// TIA Portal project "ContadoresHMI4" (V16)

(* hardware
DEVICE "S71500/ET200MP station_1"  S7-1500 station
   slot 0: "Rail_0"  Rack  6ES7 590-1***0-0AA0
   slot 1: "PLC_1"  CPU 1516-3 PN/DP  6ES7 516-3AN00-0AB0  V1.8
      slot 3: "CPU display_1"  6ES7591-1BA00-0AA0
      slot 32768: "PROFINET interface_1"  X1
         slot 32769: "Port_1"  X1 P1
         slot 32770: "Port_2"  X1 P2
      slot 33024: "PROFINET interface_2"  X2
         slot 33025: "Port_1"  X2 P1
      slot 33280: "DP interface_1"  X3
DEVICE "HMI_1"  TP700 Comfort
   slot 0: "HMI_1"  TP700 Comfort  6AV2 124-0GC01-0AX0  16.0.0.0
   slot 1: "HMI_RT_1"  TP700 Comfort  6AV2 124-0GC01-0AX0  16.0.0.0
   slot 5: "HMI_1.IE_CP_1"  PROFINET Interface  16.0.0.0
      slot 1: "PROFINET Interface_1"  PROFINET Interface
         slot 1: "Port_1"  Port
         slot 2: "Port_2"  Port
   slot 7: "HMI_1.MPI/DP_CP_1"  MPI/DP Interface  16.0.0.0
*)

// ===== PLC "PLC_1"  CPU 1516-3 PN/DP =====

VAR_GLOBAL   // PLC tag table "Default tag table"
   "ReiniciarJuego" AT %M6.0 : Bool;
   "CodigoS0J1" AT %M6.1 : Bool;
   "CodigoS1J1" AT %M6.2 : Bool;
   "CodigoS2J1" AT %M6.3 : Bool;
   "CodigoS3J1" AT %M6.4 : Bool;
   "CodigoO0J1" AT %M6.5 : Bool;
   "CodigoO1J1" AT %M6.6 : Bool;
   "CodigoO2J1" AT %M6.7 : Bool;
   "CodigoO3J1" AT %M7.0 : Bool;
   "CodigoS0J2" AT %M7.1 : Bool;
   "CodigoS1J2" AT %M7.2 : Bool;
   "CodigoS2J2" AT %M7.3 : Bool;
   "CodigoS3J2" AT %M7.4 : Bool;
   "CodigoO0J2" AT %M7.5 : Bool;
   "CodigoO1J2" AT %M7.6 : Bool;
   "CodigoO2J2" AT %M7.7 : Bool;
   "CodigoO3J2" AT %M8.0 : Bool;
   "Intento0J1" AT %M8.1 : Bool;
   "Intento1J1" AT %M8.2 : Bool;
   "Intento2J1" AT %M8.3 : Bool;
   "Intento3J1" AT %M8.4 : Bool;
   "Intento0J2" AT %M8.5 : Bool;
   "Intento1J2" AT %M8.6 : Bool;
   "Intento2J2" AT %M8.7 : Bool;
   "Intento3J2" AT %M9.0 : Bool;
   "IntentoCompletoJ1" AT %MW2 : UInt;
   "IntentoCompletoJ2" AT %MW4 : UInt;
   "Timer" AT %M9.3 : Bool;
   "Repetido" AT %M9.4 : Bool;
   "Panel1CafeJ1" AT %M9.5 : Bool;
   "Panel1RosaJ1" AT %M9.6 : Bool;
   "Panel1MoradoJ1" AT %M9.7 : Bool;
   "Panel1RojoJ1" AT %M10.0 : Bool;
   "Panel1AzulJ1" AT %M10.1 : Bool;
   "Panel1VerdeJ1" AT %M10.2 : Bool;
   "Panel1AmarilloJ1" AT %M10.3 : Bool;
   "Panel2CafeJ1" AT %M10.4 : Bool;
   "Panel2RosaJ1" AT %M10.5 : Bool;
   "Panel2MoradoJ1" AT %M10.6 : Bool;
   "Panel2RojoJ1" AT %M10.7 : Bool;
   "Panel2AzulJ1" AT %M11.0 : Bool;
   "Panel2VerdeJ1" AT %M11.1 : Bool;
   "Panel2AmarilloJ1" AT %M11.2 : Bool;
   "Panel1CafeJ2" AT %M11.3 : Bool;
   "Panel1RosaJ2" AT %M11.4 : Bool;
   "Panel1MoradoJ2" AT %M11.5 : Bool;
   "Panel1RojoJ2" AT %M11.6 : Bool;
   "Panel1AzulJ2" AT %M11.7 : Bool;
   "Panel1VerdeJ2" AT %M12.0 : Bool;
   "Panel1AmarilloJ2" AT %M12.1 : Bool;
   "Panel2CafeJ2" AT %M12.2 : Bool;
   "Panel2RosaJ2" AT %M12.3 : Bool;
   "Panel2MoradoJ2" AT %M12.4 : Bool;
   "Panel2RojoJ2" AT %M12.5 : Bool;
   "Panel2AzulJ2" AT %M12.6 : Bool;
   "Panel2VerdeJ2" AT %M12.7 : Bool;
   "Panel2AmarilloJ2" AT %M13.0 : Bool;
   "Panel1J1Activado" AT %M13.1 : Bool;
   "Panel2J1Activado" AT %M13.2 : Bool;
   "Panel1J2Activado" AT %M13.3 : Bool;
   "Panel2J2Activado" AT %M13.4 : Bool;
   "ReinicioCorrecto" AT %M13.5 : Bool;
   "Bounce1" AT %M13.6 : Bool;
   "Bounce2" AT %M13.7 : Bool;
   "Bounce3" AT %M14.0 : Bool;
   "Bounce5" AT %M14.1 : Bool;
   "Bounce6" AT %M14.2 : Bool;
   "Bounce7" AT %M14.3 : Bool;
   "Bounce8" AT %M14.4 : Bool;
   "Bounce10" AT %M14.5 : Bool;
   "MensajeCorrecto" AT %M14.6 : Bool;
   "Bounce4" AT %M14.7 : Bool;
   "Bounce9" AT %M15.0 : Bool;
   "ReiniciarContadorJ1" AT %M15.1 : Bool;
   "ReiniciarContadorJ2" AT %M15.2 : Bool;
   "ChecarIntento1J1" AT %M15.3 : Bool;
   "ChecarIntento2J1" AT %M15.4 : Bool;
   "ChecarIntento3J1" AT %M15.5 : Bool;
   "ChecarIntento4J1" AT %M15.6 : Bool;
   "ChecarIntento1J2" AT %M15.7 : Bool;
   "ChecarIntento2J2" AT %M16.0 : Bool;
   "ChecarIntento3J2" AT %M16.1 : Bool;
   "ChecarIntento4J2" AT %M16.2 : Bool;
   "ContadorCorr" AT %MW17 : UInt;
   "ContadorSimi" AT %MW20 : UInt;
   "ContadorError" AT %MW22 : UInt;
   "ContadorCorrTemp" AT %MW24 : UInt;
   "ContadorSimiTemp" AT %MW26 : UInt;
   "ReiniciarChecarCorr" AT %M28.0 : Bool;
   "ReiniciarChecarSimi" AT %M28.1 : Bool;
   "ReiniciarChecarError" AT %M28.2 : Bool;
   "ChecarIntentoCorrecto" AT %M28.3 : Bool;
   "ChecarIntento1SJ1" AT %M28.4 : Bool;
   "ChecarIntento2SJ1" AT %M28.5 : Bool;
   "ChecarIntento3SJ1" AT %M28.6 : Bool;
   "ChecarIntento4SJ1" AT %M28.7 : Bool;
   "ChecarIntento1SJ2" AT %M29.0 : Bool;
   "ChecarIntento2SJ2" AT %M29.1 : Bool;
   "ChecarIntento3SJ2" AT %M29.2 : Bool;
   "ChecarIntento4SJ2" AT %M29.3 : Bool;
   "CorrectasSimilares" AT %M29.4 : Bool;
   "IntentoCompletoCORR" AT %MW31 : UInt;
   "ReiniciarCorrSimiDisp" AT %M34.0 : Bool;
   "CondicionGanasteJ1" AT %M34.1 : Bool;
   "CondicionPerdisteJ1" AT %M34.2 : Bool;
   "CondicionGanasteJ2" AT %M34.3 : Bool;
   "CondicionPerdisteJ2" AT %M34.4 : Bool;
   "BloqueoSimilares1" AT %M34.5 : Bool;
   "BloqueoSimilares2" AT %M34.6 : Bool;
   "BloqueoSimilares3" AT %M34.7 : Bool;
   "BloqueoSimilares4" AT %M35.0 : Bool;
END_VAR

DATA_BLOCK "Var"   // DB3
{ S7_Optimized_Access := 'TRUE' }
VERSION : 0.1
   VAR
      V1 : Array[0..10, 0..10] of Int;
      CodigoSJ1 : Array[0..3] of Int;
      CodigoOJ1 : Array[0..3] of Int;
      CodigoSJ2 : Array[0..3] of Int;
      CodigoOJ2 : Array[0..3] of Int;
      VectorPrincipalJ1 : Array[0..7, 0..3] of Int;
      VectorSecundarioJ1 : Array[0..7, 0..3] of Int;
      VectorPrincipalJ2 : Array[0..7, 0..3] of Int;
      VectorSecundarioJ2 : Array[0..7, 0..3] of Int;
      VectorMensajes : Array[0..10] of Int;
      VectorMensajesReset : Array[0..10] of Int;
      VectorMensajesJ2 : Array[0..10] of Int;
      VectorMensajesResetJ2 : Array[0..10] of Int;
      VectorCorrectas : Array[0..7, 0..3] of Int;
      VectorCorrectasReset : Array[0..7, 0..3] of Int;
      CodigoSimilaresJ1 : Array[0..3] of Int;
      CodigoSimilaresJ1Temp : Array[0..3] of Int;
   END_VAR
BEGIN
END_DATA_BLOCK

// folder: System blocks/Program resources

DATA_BLOCK "ContadorCorrectas"   // DB1
{ S7_Optimized_Access := 'TRUE' }
AUTHOR : Simatic
FAMILY : IEC
NAME : UCNTR
VERSION : 1.2
// stored: InstanceOfName IEC_UCOUNTER
"IEC_UCOUNTER"
BEGIN
END_DATA_BLOCK

DATA_BLOCK "IEC_Counter_0_DB_1"   // DB2
{ S7_Optimized_Access := 'TRUE' }
AUTHOR : Simatic
FAMILY : IEC
NAME : UCNTR
VERSION : 1.2
// stored: InstanceOfName IEC_UCOUNTER
"IEC_UCOUNTER"
BEGIN
END_DATA_BLOCK

DATA_BLOCK "IEC_Timer_1_DB"   // DB4
{ S7_Optimized_Access := 'TRUE' }
AUTHOR : Simatic
FAMILY : IEC
NAME : IEC_TMR
VERSION : 1.0
// stored: InstanceOfName IEC_TIMER
"IEC_TIMER"
BEGIN
END_DATA_BLOCK

DATA_BLOCK "IEC_Timer_0_DB_1"   // DB5
{ S7_Optimized_Access := 'TRUE' }
AUTHOR : Simatic
FAMILY : IEC
NAME : IEC_TMR
VERSION : 1.0
// stored: InstanceOfName IEC_TIMER
"IEC_TIMER"
BEGIN
END_DATA_BLOCK

DATA_BLOCK "IEC_Timer_2_DB"   // DB6
{ S7_Optimized_Access := 'TRUE' }
AUTHOR : Simatic
FAMILY : IEC
NAME : IEC_TMR
VERSION : 1.0
// stored: InstanceOfName IEC_TIMER
"IEC_TIMER"
BEGIN
END_DATA_BLOCK

DATA_BLOCK "IEC_Timer_3_DB"   // DB7
{ S7_Optimized_Access := 'TRUE' }
AUTHOR : Simatic
FAMILY : IEC
NAME : IEC_TMR
VERSION : 1.0
// stored: InstanceOfName IEC_TIMER
"IEC_TIMER"
BEGIN
END_DATA_BLOCK

DATA_BLOCK "IEC_Timer_4_DB"   // DB8
{ S7_Optimized_Access := 'TRUE' }
AUTHOR : Simatic
FAMILY : IEC
NAME : IEC_TMR
VERSION : 1.0
// stored: InstanceOfName IEC_TIMER
"IEC_TIMER"
BEGIN
END_DATA_BLOCK

DATA_BLOCK "IEC_Timer_5_DB"   // DB9
{ S7_Optimized_Access := 'TRUE' }
AUTHOR : Simatic
FAMILY : IEC
NAME : IEC_TMR
VERSION : 1.0
// stored: InstanceOfName IEC_TIMER
"IEC_TIMER"
BEGIN
END_DATA_BLOCK

DATA_BLOCK "ContadorSimilares"   // DB10
{ S7_Optimized_Access := 'TRUE' }
AUTHOR : Simatic
FAMILY : IEC
NAME : UCNTR
VERSION : 1.2
// stored: InstanceOfName IEC_UCOUNTER
"IEC_UCOUNTER"
BEGIN
END_DATA_BLOCK

// folder: (top level)

ORGANIZATION_BLOCK "Main"   // OB1, LAD, ProgramCycle
TITLE = "Main Program Sweep (Cycle)"
{ S7_Optimized_Access := 'TRUE' }
VERSION : 0.1
   VAR_INPUT
      Initial_Call : Bool;   // Initial call of this OB
      Remanence : Bool;   // =True, if remanent data are available
   END_VAR
   VAR_TEMP   // added for the SCL form of the ladder/FBD networks
      _w1 : Bool;
      _w2 : Bool;
      _w3 : Bool;
      _w4 : Bool;
      _w5 : Bool;
      _w6 : Bool;
      _w7 : Bool;
      _w8 : Bool;
      _w9 : Bool;
      _w10 : Bool;
      _w11 : Bool;
      _w12 : Bool;
      _w13 : Bool;
      _w14 : Bool;
      _w15 : Bool;
      _w16 : Bool;
      _w17 : Bool;
      _w18 : Bool;
      _w19 : Bool;
      _w20 : Bool;
      _w21 : Bool;
      _w22 : Bool;
      _w23 : Bool;
      _w24 : Bool;
      _w25 : Bool;
      _w26 : Bool;
      _w27 : Bool;
      _w28 : Bool;
      _w29 : Bool;
      _w30 : Bool;
      _w31 : Bool;
      _w32 : Bool;
      _w33 : Bool;
      _w34 : Bool;
      _w35 : Bool;
      _w36 : Bool;
      _w37 : Bool;
   END_VAR
BEGIN

REGION Network 1: Reiniciar Juego
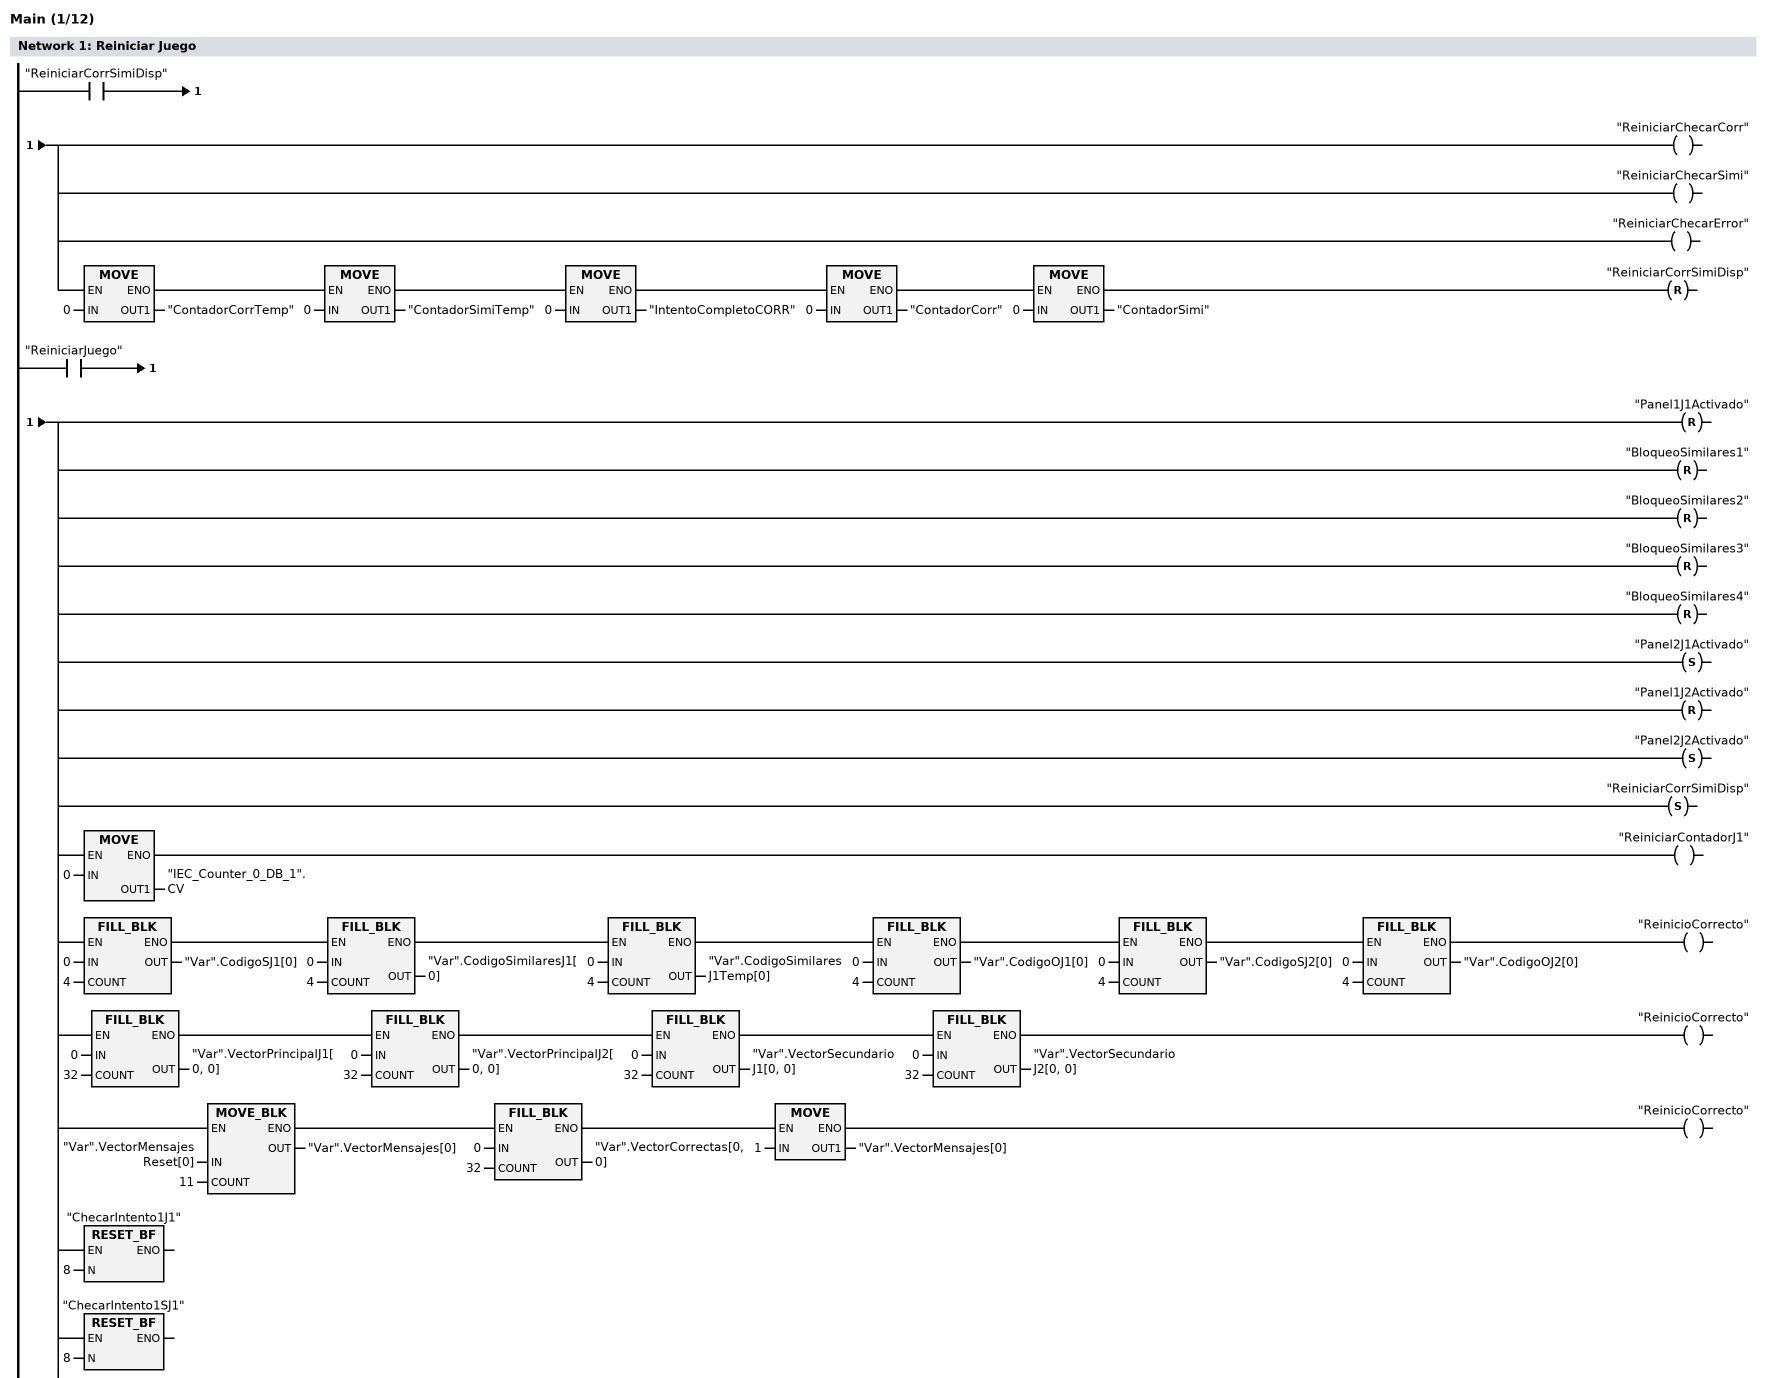
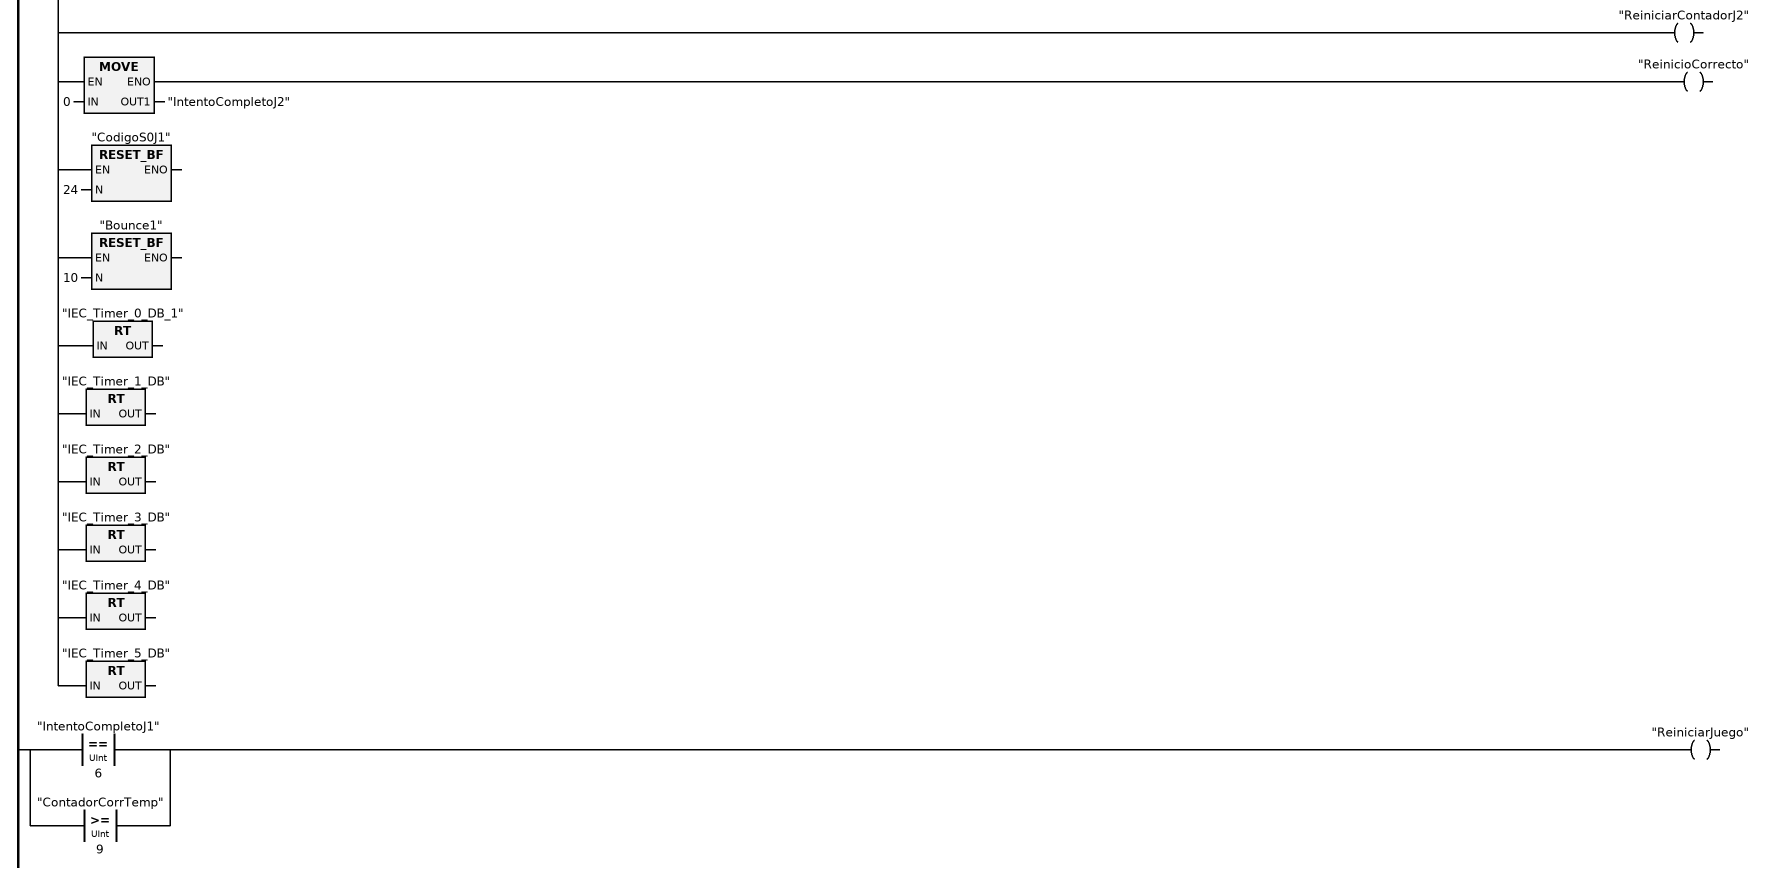
   // no SCL statement known for RBitfield: written as a call
   "ReiniciarChecarCorr" := "ReiniciarCorrSimiDisp";
   "ReiniciarChecarSimi" := "ReiniciarCorrSimiDisp";
   "ReiniciarChecarError" := "ReiniciarCorrSimiDisp";
   IF "ReiniciarCorrSimiDisp" THEN
       "ContadorCorrTemp" := 0;
       "ContadorSimiTemp" := 0;
       "IntentoCompletoCORR" := 0;
       "ContadorCorr" := 0;
       "ContadorSimi" := 0;
       "ReiniciarCorrSimiDisp" := FALSE;
   END_IF;
   IF "ReiniciarJuego" THEN
       "Panel1J1Activado" := FALSE;
       "BloqueoSimilares1" := FALSE;
       "BloqueoSimilares2" := FALSE;
       "BloqueoSimilares3" := FALSE;
       "BloqueoSimilares4" := FALSE;
       "Panel2J1Activado" := TRUE;
       "Panel1J2Activado" := FALSE;
       "Panel2J2Activado" := TRUE;
       "ReiniciarCorrSimiDisp" := TRUE;
       "IEC_Counter_0_DB_1".CV := 0;
   END_IF;
   "ReiniciarContadorJ1" := "ReiniciarJuego";
   #_w1 := "ReiniciarJuego";
   #_w2 := "ReiniciarJuego";
   IF #_w2 THEN
       FILL_BLK(IN := 0, COUNT := 4, OUT => "Var".CodigoSJ1[0]);
       FILL_BLK(IN := 0, COUNT := 4, OUT => "Var".CodigoSimilaresJ1[0]);
       FILL_BLK(IN := 0, COUNT := 4, OUT => "Var".CodigoSimilaresJ1Temp[0]);
       FILL_BLK(IN := 0, COUNT := 4, OUT => "Var".CodigoOJ1[0]);
       FILL_BLK(IN := 0, COUNT := 4, OUT => "Var".CodigoSJ2[0]);
       FILL_BLK(IN := 0, COUNT := 4, OUT => "Var".CodigoOJ2[0]);
   END_IF;
   "ReinicioCorrecto" := #_w2;
   IF #_w1 THEN
       FILL_BLK(IN := 0, COUNT := 32, OUT => "Var".VectorPrincipalJ1[0, 0]);
       FILL_BLK(IN := 0, COUNT := 32, OUT => "Var".VectorPrincipalJ2[0, 0]);
       FILL_BLK(IN := 0, COUNT := 32, OUT => "Var".VectorSecundarioJ1[0, 0]);
       FILL_BLK(IN := 0, COUNT := 32, OUT => "Var".VectorSecundarioJ2[0, 0]);
   END_IF;
   "ReinicioCorrecto" := #_w1;
   IF #_w1 THEN
       MOVE_BLK(IN := "Var".VectorMensajesReset[0], COUNT := 11, OUT => "Var".VectorMensajes[0]);
       FILL_BLK(IN := 0, COUNT := 32, OUT => "Var".VectorCorrectas[0, 0]);
       "Var".VectorMensajes[0] := 1;
   END_IF;
   "ReinicioCorrecto" := #_w1;
   IF #_w1 THEN
       RESET_BF(operand := "ChecarIntento1J1", n := 8);
       RESET_BF(operand := "ChecarIntento1SJ1", n := 8);
   END_IF;
   "ReiniciarContadorJ2" := #_w1;
   IF #_w1 THEN "IntentoCompletoJ2" := 0; END_IF;
   "ReinicioCorrecto" := #_w1;
   IF #_w1 THEN
       RESET_BF(operand := "CodigoS0J1", n := 24);
       RESET_BF(operand := "Bounce1", n := 10);
       RESET_TIMER("IEC_Timer_0_DB_1");
       RESET_TIMER("IEC_Timer_1_DB");
       RESET_TIMER("IEC_Timer_2_DB");
       RESET_TIMER("IEC_Timer_3_DB");
       RESET_TIMER("IEC_Timer_4_DB");
       RESET_TIMER("IEC_Timer_5_DB");
   END_IF;
   "ReiniciarJuego" := ("IntentoCompletoJ1" = 6) OR ("ContadorCorrTemp" >= 9);
END_REGION

REGION Network 2: Seleccionar Codigo
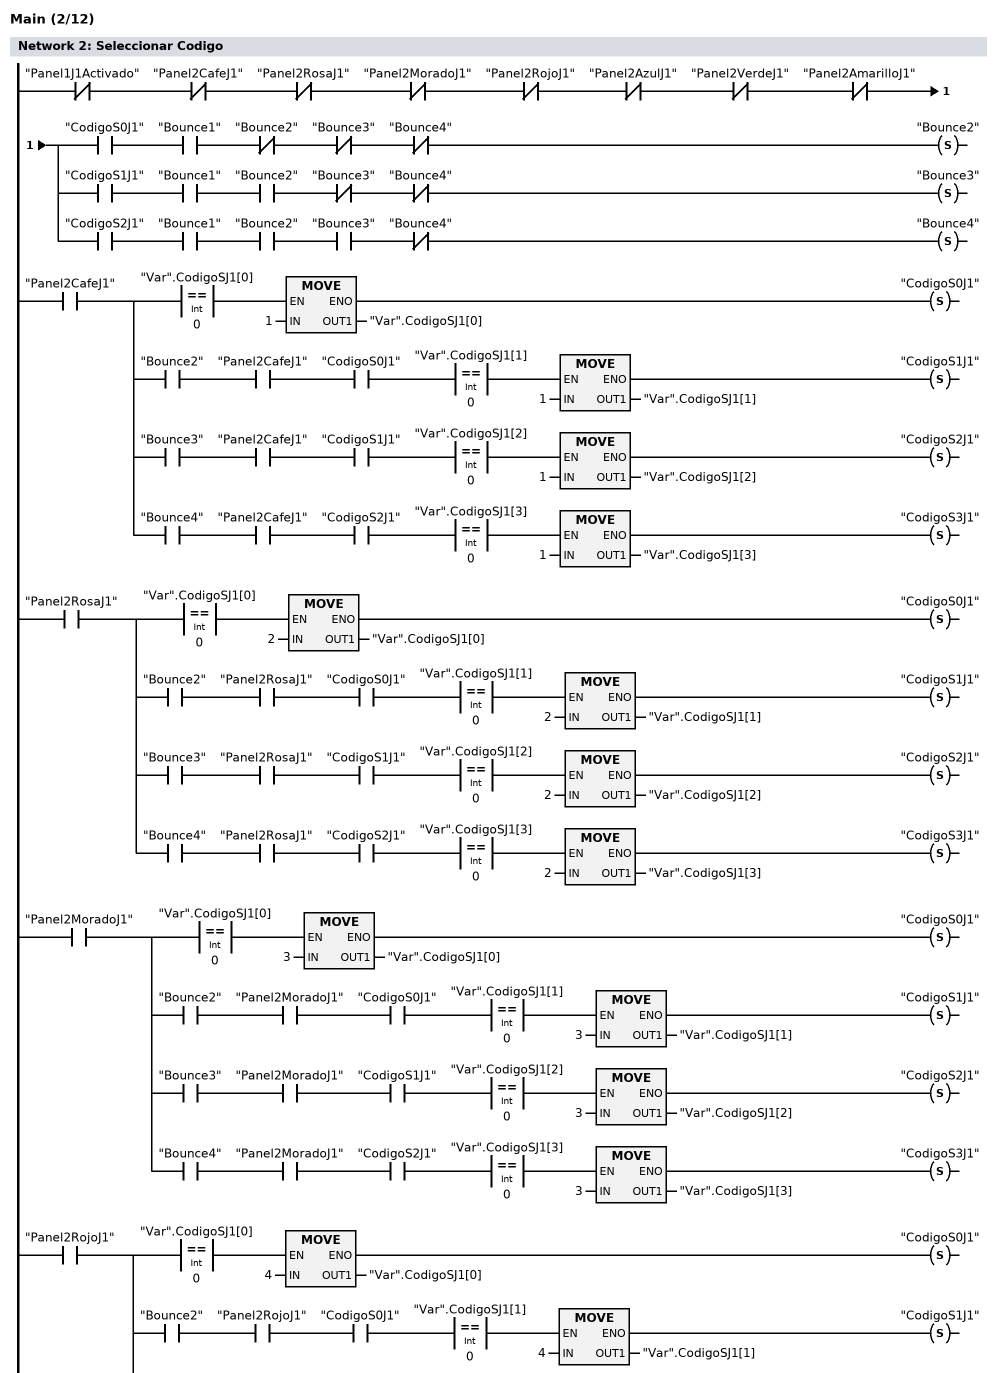
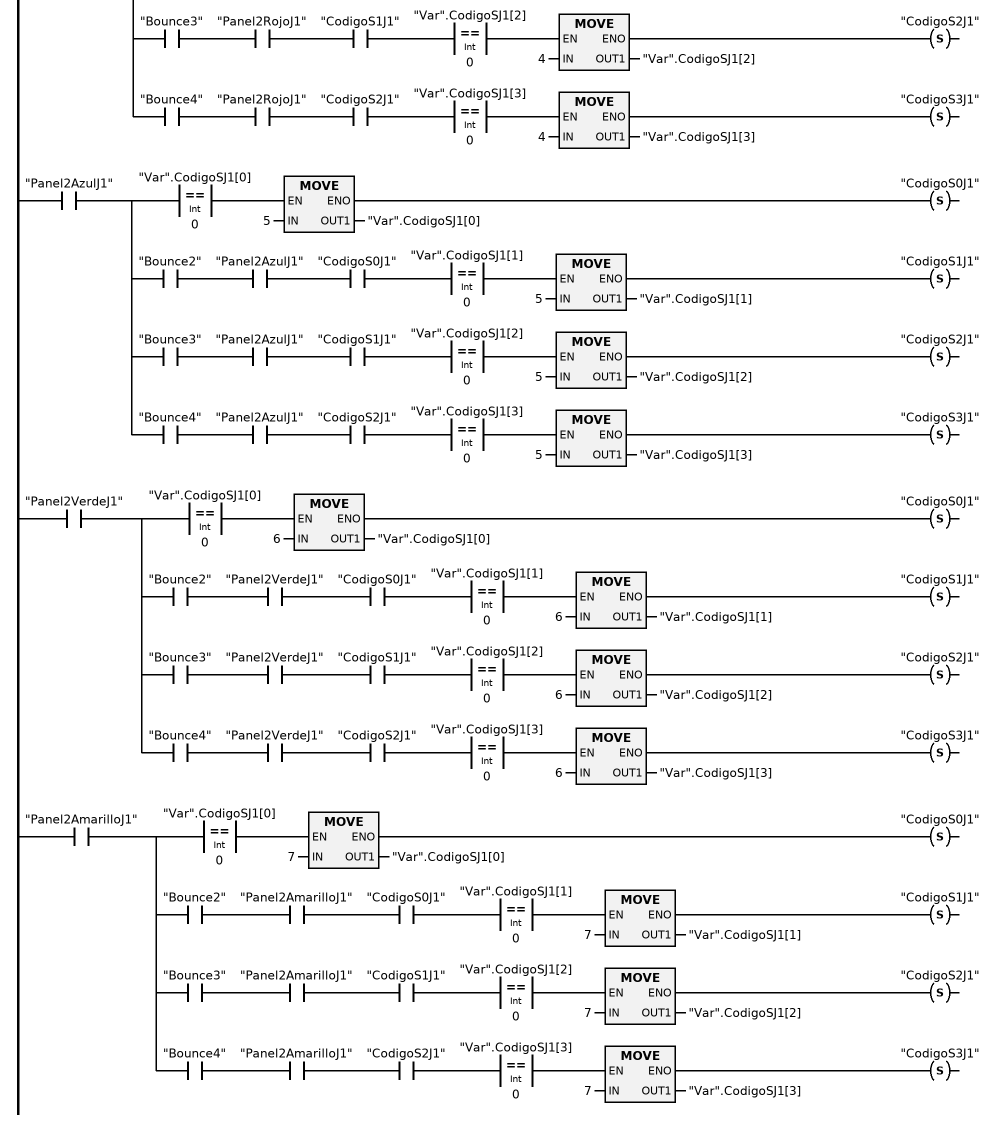
   RUNG wire#powerrail
      I_Contact( "Panel1J1Activado" )
      I_Contact( "Panel2CafeJ1" )
      I_Contact( "Panel2RosaJ1" )
      I_Contact( "Panel2MoradoJ1" )
      I_Contact( "Panel2RojoJ1" )
      I_Contact( "Panel2AzulJ1" )
      I_Contact( "Panel2VerdeJ1" )
      I_Contact( "Panel2AmarilloJ1" )
      wire#w1
      Contact( "CodigoS0J1" )
      Contact( "Bounce1" )
      I_Contact( "Bounce2" )
      I_Contact( "Bounce3" )
      I_Contact( "Bounce4" )
      S_Coil( "Bounce2" )
   END_RUNG
   RUNG wire#w1
      Contact( "CodigoS1J1" )
      Contact( "Bounce1" )
      Contact( "Bounce2" )
      I_Contact( "Bounce3" )
      I_Contact( "Bounce4" )
      S_Coil( "Bounce3" )
   END_RUNG
   RUNG wire#w1
      Contact( "CodigoS2J1" )
      Contact( "Bounce1" )
      Contact( "Bounce2" )
      Contact( "Bounce3" )
      I_Contact( "Bounce4" )
      S_Coil( "Bounce4" )
   END_RUNG
   RUNG wire#powerrail
      Contact( "Panel2CafeJ1" )
      wire#w2
      { S7_Templates := "SrcType := Int" } EQ_Contact(in1 := "Var".CodigoSJ1[0], in2 := 0)
      Move(in := 1, out1 => "Var".CodigoSJ1[0])
      S_Coil( "CodigoS0J1" )
   END_RUNG
   RUNG wire#w2
      Contact( "Bounce2" )
      Contact( "Panel2CafeJ1" )
      Contact( "CodigoS0J1" )
      { S7_Templates := "SrcType := Int" } EQ_Contact(in1 := "Var".CodigoSJ1[1], in2 := 0)
      Move(in := 1, out1 => "Var".CodigoSJ1[1])
      S_Coil( "CodigoS1J1" )
   END_RUNG
   RUNG wire#w2
      Contact( "Bounce3" )
      Contact( "Panel2CafeJ1" )
      Contact( "CodigoS1J1" )
      { S7_Templates := "SrcType := Int" } EQ_Contact(in1 := "Var".CodigoSJ1[2], in2 := 0)
      Move(in := 1, out1 => "Var".CodigoSJ1[2])
      S_Coil( "CodigoS2J1" )
   END_RUNG
   RUNG wire#w2
      Contact( "Bounce4" )
      Contact( "Panel2CafeJ1" )
      Contact( "CodigoS2J1" )
      { S7_Templates := "SrcType := Int" } EQ_Contact(in1 := "Var".CodigoSJ1[3], in2 := 0)
      Move(in := 1, out1 => "Var".CodigoSJ1[3])
      S_Coil( "CodigoS3J1" )
   END_RUNG
   RUNG wire#powerrail
      Contact( "Panel2RosaJ1" )
      wire#w3
      { S7_Templates := "SrcType := Int" } EQ_Contact(in1 := "Var".CodigoSJ1[0], in2 := 0)
      Move(in := 2, out1 => "Var".CodigoSJ1[0])
      S_Coil( "CodigoS0J1" )
   END_RUNG
   RUNG wire#w3
      Contact( "Bounce2" )
      Contact( "Panel2RosaJ1" )
      Contact( "CodigoS0J1" )
      { S7_Templates := "SrcType := Int" } EQ_Contact(in1 := "Var".CodigoSJ1[1], in2 := 0)
      Move(in := 2, out1 => "Var".CodigoSJ1[1])
      S_Coil( "CodigoS1J1" )
   END_RUNG
   RUNG wire#w3
      Contact( "Bounce3" )
      Contact( "Panel2RosaJ1" )
      Contact( "CodigoS1J1" )
      { S7_Templates := "SrcType := Int" } EQ_Contact(in1 := "Var".CodigoSJ1[2], in2 := 0)
      Move(in := 2, out1 => "Var".CodigoSJ1[2])
      S_Coil( "CodigoS2J1" )
   END_RUNG
   RUNG wire#w3
      Contact( "Bounce4" )
      Contact( "Panel2RosaJ1" )
      Contact( "CodigoS2J1" )
      { S7_Templates := "SrcType := Int" } EQ_Contact(in1 := "Var".CodigoSJ1[3], in2 := 0)
      Move(in := 2, out1 => "Var".CodigoSJ1[3])
      S_Coil( "CodigoS3J1" )
   END_RUNG
   RUNG wire#powerrail
      Contact( "Panel2MoradoJ1" )
      wire#w4
      { S7_Templates := "SrcType := Int" } EQ_Contact(in1 := "Var".CodigoSJ1[0], in2 := 0)
      Move(in := 3, out1 => "Var".CodigoSJ1[0])
      S_Coil( "CodigoS0J1" )
   END_RUNG
   RUNG wire#w4
      Contact( "Bounce2" )
      Contact( "Panel2MoradoJ1" )
      Contact( "CodigoS0J1" )
      { S7_Templates := "SrcType := Int" } EQ_Contact(in1 := "Var".CodigoSJ1[1], in2 := 0)
      Move(in := 3, out1 => "Var".CodigoSJ1[1])
      S_Coil( "CodigoS1J1" )
   END_RUNG
   RUNG wire#w4
      Contact( "Bounce3" )
      Contact( "Panel2MoradoJ1" )
      Contact( "CodigoS1J1" )
      { S7_Templates := "SrcType := Int" } EQ_Contact(in1 := "Var".CodigoSJ1[2], in2 := 0)
      Move(in := 3, out1 => "Var".CodigoSJ1[2])
      S_Coil( "CodigoS2J1" )
   END_RUNG
   RUNG wire#w4
      Contact( "Bounce4" )
      Contact( "Panel2MoradoJ1" )
      Contact( "CodigoS2J1" )
      { S7_Templates := "SrcType := Int" } EQ_Contact(in1 := "Var".CodigoSJ1[3], in2 := 0)
      Move(in := 3, out1 => "Var".CodigoSJ1[3])
      S_Coil( "CodigoS3J1" )
   END_RUNG
   RUNG wire#powerrail
      Contact( "Panel2RojoJ1" )
      wire#w5
      { S7_Templates := "SrcType := Int" } EQ_Contact(in1 := "Var".CodigoSJ1[0], in2 := 0)
      Move(in := 4, out1 => "Var".CodigoSJ1[0])
      S_Coil( "CodigoS0J1" )
   END_RUNG
   RUNG wire#w5
      Contact( "Bounce2" )
      Contact( "Panel2RojoJ1" )
      Contact( "CodigoS0J1" )
      { S7_Templates := "SrcType := Int" } EQ_Contact(in1 := "Var".CodigoSJ1[1], in2 := 0)
      Move(in := 4, out1 => "Var".CodigoSJ1[1])
      S_Coil( "CodigoS1J1" )
   END_RUNG
   RUNG wire#w5
      Contact( "Bounce3" )
      Contact( "Panel2RojoJ1" )
      Contact( "CodigoS1J1" )
      { S7_Templates := "SrcType := Int" } EQ_Contact(in1 := "Var".CodigoSJ1[2], in2 := 0)
      Move(in := 4, out1 => "Var".CodigoSJ1[2])
      S_Coil( "CodigoS2J1" )
   END_RUNG
   RUNG wire#w5
      Contact( "Bounce4" )
      Contact( "Panel2RojoJ1" )
      Contact( "CodigoS2J1" )
      { S7_Templates := "SrcType := Int" } EQ_Contact(in1 := "Var".CodigoSJ1[3], in2 := 0)
      Move(in := 4, out1 => "Var".CodigoSJ1[3])
      S_Coil( "CodigoS3J1" )
   END_RUNG
   RUNG wire#powerrail
      Contact( "Panel2AzulJ1" )
      wire#w6
      { S7_Templates := "SrcType := Int" } EQ_Contact(in1 := "Var".CodigoSJ1[0], in2 := 0)
      Move(in := 5, out1 => "Var".CodigoSJ1[0])
      S_Coil( "CodigoS0J1" )
   END_RUNG
   RUNG wire#w6
      Contact( "Bounce2" )
      Contact( "Panel2AzulJ1" )
      Contact( "CodigoS0J1" )
      { S7_Templates := "SrcType := Int" } EQ_Contact(in1 := "Var".CodigoSJ1[1], in2 := 0)
      Move(in := 5, out1 => "Var".CodigoSJ1[1])
      S_Coil( "CodigoS1J1" )
   END_RUNG
   RUNG wire#w6
      Contact( "Bounce3" )
      Contact( "Panel2AzulJ1" )
      Contact( "CodigoS1J1" )
      { S7_Templates := "SrcType := Int" } EQ_Contact(in1 := "Var".CodigoSJ1[2], in2 := 0)
      Move(in := 5, out1 => "Var".CodigoSJ1[2])
      S_Coil( "CodigoS2J1" )
   END_RUNG
   RUNG wire#w6
      Contact( "Bounce4" )
      Contact( "Panel2AzulJ1" )
      Contact( "CodigoS2J1" )
      { S7_Templates := "SrcType := Int" } EQ_Contact(in1 := "Var".CodigoSJ1[3], in2 := 0)
      Move(in := 5, out1 => "Var".CodigoSJ1[3])
      S_Coil( "CodigoS3J1" )
   END_RUNG
   RUNG wire#powerrail
      Contact( "Panel2VerdeJ1" )
      wire#w7
      { S7_Templates := "SrcType := Int" } EQ_Contact(in1 := "Var".CodigoSJ1[0], in2 := 0)
      Move(in := 6, out1 => "Var".CodigoSJ1[0])
      S_Coil( "CodigoS0J1" )
   END_RUNG
   RUNG wire#w7
      Contact( "Bounce2" )
      Contact( "Panel2VerdeJ1" )
      Contact( "CodigoS0J1" )
      { S7_Templates := "SrcType := Int" } EQ_Contact(in1 := "Var".CodigoSJ1[1], in2 := 0)
      Move(in := 6, out1 => "Var".CodigoSJ1[1])
      S_Coil( "CodigoS1J1" )
   END_RUNG
   RUNG wire#w7
      Contact( "Bounce3" )
      Contact( "Panel2VerdeJ1" )
      Contact( "CodigoS1J1" )
      { S7_Templates := "SrcType := Int" } EQ_Contact(in1 := "Var".CodigoSJ1[2], in2 := 0)
      Move(in := 6, out1 => "Var".CodigoSJ1[2])
      S_Coil( "CodigoS2J1" )
   END_RUNG
   RUNG wire#w7
      Contact( "Bounce4" )
      Contact( "Panel2VerdeJ1" )
      Contact( "CodigoS2J1" )
      { S7_Templates := "SrcType := Int" } EQ_Contact(in1 := "Var".CodigoSJ1[3], in2 := 0)
      Move(in := 6, out1 => "Var".CodigoSJ1[3])
      S_Coil( "CodigoS3J1" )
   END_RUNG
   RUNG wire#powerrail
      Contact( "Panel2AmarilloJ1" )
      wire#w8
      { S7_Templates := "SrcType := Int" } EQ_Contact(in1 := "Var".CodigoSJ1[0], in2 := 0)
      Move(in := 7, out1 => "Var".CodigoSJ1[0])
      S_Coil( "CodigoS0J1" )
   END_RUNG
   RUNG wire#w8
      Contact( "Bounce2" )
      Contact( "Panel2AmarilloJ1" )
      Contact( "CodigoS0J1" )
      { S7_Templates := "SrcType := Int" } EQ_Contact(in1 := "Var".CodigoSJ1[1], in2 := 0)
      Move(in := 7, out1 => "Var".CodigoSJ1[1])
      S_Coil( "CodigoS1J1" )
   END_RUNG
   RUNG wire#w8
      Contact( "Bounce3" )
      Contact( "Panel2AmarilloJ1" )
      Contact( "CodigoS1J1" )
      { S7_Templates := "SrcType := Int" } EQ_Contact(in1 := "Var".CodigoSJ1[2], in2 := 0)
      Move(in := 7, out1 => "Var".CodigoSJ1[2])
      S_Coil( "CodigoS2J1" )
   END_RUNG
   RUNG wire#w8
      Contact( "Bounce4" )
      Contact( "Panel2AmarilloJ1" )
      Contact( "CodigoS2J1" )
      { S7_Templates := "SrcType := Int" } EQ_Contact(in1 := "Var".CodigoSJ1[3], in2 := 0)
      Move(in := 7, out1 => "Var".CodigoSJ1[3])
      S_Coil( "CodigoS3J1" )
   END_RUNG
   // the same network as SCL:
   #_w1 := NOT "Panel1J1Activado" AND NOT "Panel2CafeJ1" AND NOT "Panel2RosaJ1" AND NOT "Panel2MoradoJ1" AND NOT "Panel2RojoJ1" AND NOT "Panel2AzulJ1" AND NOT "Panel2VerdeJ1" AND NOT "Panel2AmarilloJ1";
   IF #_w1 AND "CodigoS0J1" AND "Bounce1" AND NOT "Bounce2" AND NOT "Bounce3" AND NOT "Bounce4" THEN
       "Bounce2" := TRUE;
   END_IF;
   IF #_w1 AND "CodigoS1J1" AND "Bounce1" AND "Bounce2" AND NOT "Bounce3" AND NOT "Bounce4" THEN
       "Bounce3" := TRUE;
   END_IF;
   IF #_w1 AND "CodigoS2J1" AND "Bounce1" AND "Bounce2" AND "Bounce3" AND NOT "Bounce4" THEN
       "Bounce4" := TRUE;
   END_IF;
   #_w2 := "Panel2CafeJ1" AND ("Var".CodigoSJ1[0] = 0);
   IF #_w2 THEN
       "Var".CodigoSJ1[0] := 1;
       "CodigoS0J1" := TRUE;
   END_IF;
   #_w3 := "Panel2CafeJ1" AND "Bounce2" AND "Panel2CafeJ1" AND "CodigoS0J1" AND ("Var".CodigoSJ1[1] = 0);
   IF #_w3 THEN
       "Var".CodigoSJ1[1] := 1;
       "CodigoS1J1" := TRUE;
   END_IF;
   #_w4 := "Panel2CafeJ1" AND "Bounce3" AND "Panel2CafeJ1" AND "CodigoS1J1" AND ("Var".CodigoSJ1[2] = 0);
   IF #_w4 THEN
       "Var".CodigoSJ1[2] := 1;
       "CodigoS2J1" := TRUE;
   END_IF;
   #_w5 := "Panel2CafeJ1" AND "Bounce4" AND "Panel2CafeJ1" AND "CodigoS2J1" AND ("Var".CodigoSJ1[3] = 0);
   IF #_w5 THEN
       "Var".CodigoSJ1[3] := 1;
       "CodigoS3J1" := TRUE;
   END_IF;
   #_w6 := "Panel2RosaJ1" AND ("Var".CodigoSJ1[0] = 0);
   IF #_w6 THEN
       "Var".CodigoSJ1[0] := 2;
       "CodigoS0J1" := TRUE;
   END_IF;
   #_w7 := "Panel2RosaJ1" AND "Bounce2" AND "Panel2RosaJ1" AND "CodigoS0J1" AND ("Var".CodigoSJ1[1] = 0);
   IF #_w7 THEN
       "Var".CodigoSJ1[1] := 2;
       "CodigoS1J1" := TRUE;
   END_IF;
   #_w8 := "Panel2RosaJ1" AND "Bounce3" AND "Panel2RosaJ1" AND "CodigoS1J1" AND ("Var".CodigoSJ1[2] = 0);
   IF #_w8 THEN
       "Var".CodigoSJ1[2] := 2;
       "CodigoS2J1" := TRUE;
   END_IF;
   #_w9 := "Panel2RosaJ1" AND "Bounce4" AND "Panel2RosaJ1" AND "CodigoS2J1" AND ("Var".CodigoSJ1[3] = 0);
   IF #_w9 THEN
       "Var".CodigoSJ1[3] := 2;
       "CodigoS3J1" := TRUE;
   END_IF;
   #_w10 := "Panel2MoradoJ1" AND ("Var".CodigoSJ1[0] = 0);
   IF #_w10 THEN
       "Var".CodigoSJ1[0] := 3;
       "CodigoS0J1" := TRUE;
   END_IF;
   #_w11 := "Panel2MoradoJ1" AND "Bounce2" AND "Panel2MoradoJ1" AND "CodigoS0J1" AND ("Var".CodigoSJ1[1] = 0);
   IF #_w11 THEN
       "Var".CodigoSJ1[1] := 3;
       "CodigoS1J1" := TRUE;
   END_IF;
   #_w12 := "Panel2MoradoJ1" AND "Bounce3" AND "Panel2MoradoJ1" AND "CodigoS1J1" AND ("Var".CodigoSJ1[2] = 0);
   IF #_w12 THEN
       "Var".CodigoSJ1[2] := 3;
       "CodigoS2J1" := TRUE;
   END_IF;
   #_w13 := "Panel2MoradoJ1" AND "Bounce4" AND "Panel2MoradoJ1" AND "CodigoS2J1" AND ("Var".CodigoSJ1[3] = 0);
   IF #_w13 THEN
       "Var".CodigoSJ1[3] := 3;
       "CodigoS3J1" := TRUE;
   END_IF;
   #_w14 := "Panel2RojoJ1" AND ("Var".CodigoSJ1[0] = 0);
   IF #_w14 THEN
       "Var".CodigoSJ1[0] := 4;
       "CodigoS0J1" := TRUE;
   END_IF;
   #_w15 := "Panel2RojoJ1" AND "Bounce2" AND "Panel2RojoJ1" AND "CodigoS0J1" AND ("Var".CodigoSJ1[1] = 0);
   IF #_w15 THEN
       "Var".CodigoSJ1[1] := 4;
       "CodigoS1J1" := TRUE;
   END_IF;
   #_w16 := "Panel2RojoJ1" AND "Bounce3" AND "Panel2RojoJ1" AND "CodigoS1J1" AND ("Var".CodigoSJ1[2] = 0);
   IF #_w16 THEN
       "Var".CodigoSJ1[2] := 4;
       "CodigoS2J1" := TRUE;
   END_IF;
   #_w17 := "Panel2RojoJ1" AND "Bounce4" AND "Panel2RojoJ1" AND "CodigoS2J1" AND ("Var".CodigoSJ1[3] = 0);
   IF #_w17 THEN
       "Var".CodigoSJ1[3] := 4;
       "CodigoS3J1" := TRUE;
   END_IF;
   #_w18 := "Panel2AzulJ1" AND ("Var".CodigoSJ1[0] = 0);
   IF #_w18 THEN
       "Var".CodigoSJ1[0] := 5;
       "CodigoS0J1" := TRUE;
   END_IF;
   #_w19 := "Panel2AzulJ1" AND "Bounce2" AND "Panel2AzulJ1" AND "CodigoS0J1" AND ("Var".CodigoSJ1[1] = 0);
   IF #_w19 THEN
       "Var".CodigoSJ1[1] := 5;
       "CodigoS1J1" := TRUE;
   END_IF;
   #_w20 := "Panel2AzulJ1" AND "Bounce3" AND "Panel2AzulJ1" AND "CodigoS1J1" AND ("Var".CodigoSJ1[2] = 0);
   IF #_w20 THEN
       "Var".CodigoSJ1[2] := 5;
       "CodigoS2J1" := TRUE;
   END_IF;
   #_w21 := "Panel2AzulJ1" AND "Bounce4" AND "Panel2AzulJ1" AND "CodigoS2J1" AND ("Var".CodigoSJ1[3] = 0);
   IF #_w21 THEN
       "Var".CodigoSJ1[3] := 5;
       "CodigoS3J1" := TRUE;
   END_IF;
   #_w22 := "Panel2VerdeJ1" AND ("Var".CodigoSJ1[0] = 0);
   IF #_w22 THEN
       "Var".CodigoSJ1[0] := 6;
       "CodigoS0J1" := TRUE;
   END_IF;
   #_w23 := "Panel2VerdeJ1" AND "Bounce2" AND "Panel2VerdeJ1" AND "CodigoS0J1" AND ("Var".CodigoSJ1[1] = 0);
   IF #_w23 THEN
       "Var".CodigoSJ1[1] := 6;
       "CodigoS1J1" := TRUE;
   END_IF;
   #_w24 := "Panel2VerdeJ1" AND "Bounce3" AND "Panel2VerdeJ1" AND "CodigoS1J1" AND ("Var".CodigoSJ1[2] = 0);
   IF #_w24 THEN
       "Var".CodigoSJ1[2] := 6;
       "CodigoS2J1" := TRUE;
   END_IF;
   #_w25 := "Panel2VerdeJ1" AND "Bounce4" AND "Panel2VerdeJ1" AND "CodigoS2J1" AND ("Var".CodigoSJ1[3] = 0);
   IF #_w25 THEN
       "Var".CodigoSJ1[3] := 6;
       "CodigoS3J1" := TRUE;
   END_IF;
   #_w26 := "Panel2AmarilloJ1" AND ("Var".CodigoSJ1[0] = 0);
   IF #_w26 THEN
       "Var".CodigoSJ1[0] := 7;
       "CodigoS0J1" := TRUE;
   END_IF;
   #_w27 := "Panel2AmarilloJ1" AND "Bounce2" AND "Panel2AmarilloJ1" AND "CodigoS0J1" AND ("Var".CodigoSJ1[1] = 0);
   IF #_w27 THEN
       "Var".CodigoSJ1[1] := 7;
       "CodigoS1J1" := TRUE;
   END_IF;
   #_w28 := "Panel2AmarilloJ1" AND "Bounce3" AND "Panel2AmarilloJ1" AND "CodigoS1J1" AND ("Var".CodigoSJ1[2] = 0);
   IF #_w28 THEN
       "Var".CodigoSJ1[2] := 7;
       "CodigoS2J1" := TRUE;
   END_IF;
   #_w29 := "Panel2AmarilloJ1" AND "Bounce4" AND "Panel2AmarilloJ1" AND "CodigoS2J1" AND ("Var".CodigoSJ1[3] = 0);
   IF #_w29 THEN
       "Var".CodigoSJ1[3] := 7;
       "CodigoS3J1" := TRUE;
   END_IF;
END_REGION

REGION Network 3: Clave Secreta
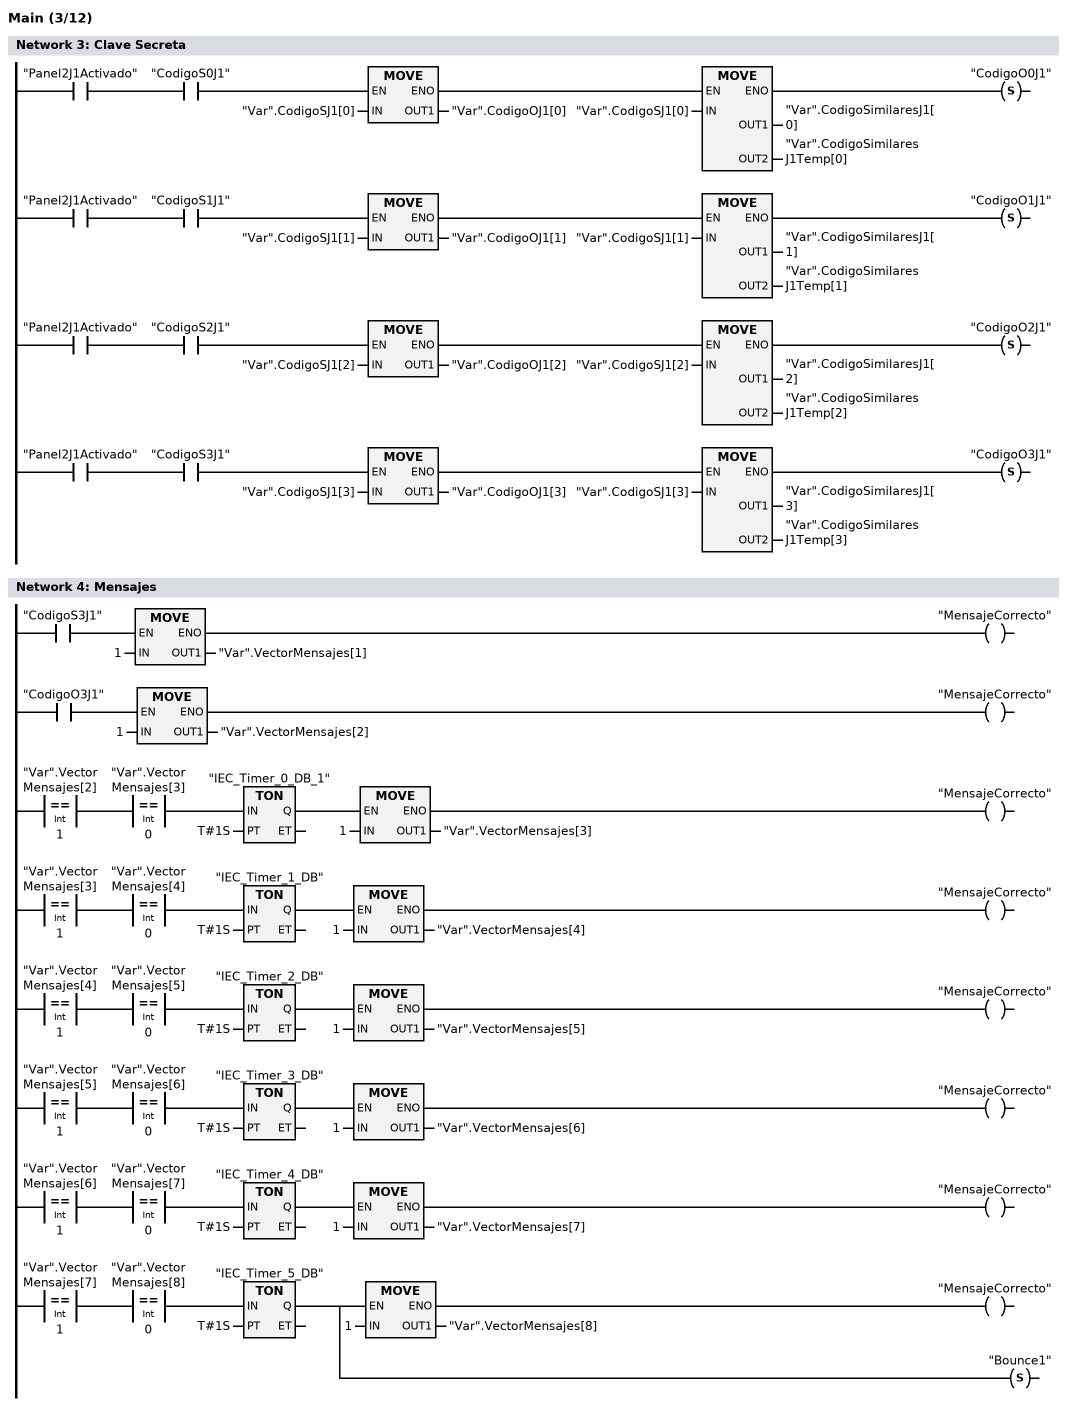
   RUNG wire#powerrail
      Contact( "Panel2J1Activado" )
      Contact( "CodigoS0J1" )
      Move(in := "Var".CodigoSJ1[0], out1 => "Var".CodigoOJ1[0])
      Move(in := "Var".CodigoSJ1[0], out1 => "Var".CodigoSimilaresJ1[0], out2 => "Var".CodigoSimilaresJ1Temp[0])
      S_Coil( "CodigoO0J1" )
   END_RUNG
   RUNG wire#powerrail
      Contact( "Panel2J1Activado" )
      Contact( "CodigoS1J1" )
      Move(in := "Var".CodigoSJ1[1], out1 => "Var".CodigoOJ1[1])
      Move(in := "Var".CodigoSJ1[1], out1 => "Var".CodigoSimilaresJ1[1], out2 => "Var".CodigoSimilaresJ1Temp[1])
      S_Coil( "CodigoO1J1" )
   END_RUNG
   RUNG wire#powerrail
      Contact( "Panel2J1Activado" )
      Contact( "CodigoS2J1" )
      Move(in := "Var".CodigoSJ1[2], out1 => "Var".CodigoOJ1[2])
      Move(in := "Var".CodigoSJ1[2], out1 => "Var".CodigoSimilaresJ1[2], out2 => "Var".CodigoSimilaresJ1Temp[2])
      S_Coil( "CodigoO2J1" )
   END_RUNG
   RUNG wire#powerrail
      Contact( "Panel2J1Activado" )
      Contact( "CodigoS3J1" )
      Move(in := "Var".CodigoSJ1[3], out1 => "Var".CodigoOJ1[3])
      Move(in := "Var".CodigoSJ1[3], out1 => "Var".CodigoSimilaresJ1[3], out2 => "Var".CodigoSimilaresJ1Temp[3])
      S_Coil( "CodigoO3J1" )
   END_RUNG
   // the same network as SCL:
   IF "Panel2J1Activado" AND "CodigoS0J1" THEN
       "Var".CodigoOJ1[0] := "Var".CodigoSJ1[0];
       "Var".CodigoSimilaresJ1[0] := "Var".CodigoSJ1[0];
       "Var".CodigoSimilaresJ1Temp[0] := "Var".CodigoSJ1[0];
       "CodigoO0J1" := TRUE;
   END_IF;
   IF "Panel2J1Activado" AND "CodigoS1J1" THEN
       "Var".CodigoOJ1[1] := "Var".CodigoSJ1[1];
       "Var".CodigoSimilaresJ1[1] := "Var".CodigoSJ1[1];
       "Var".CodigoSimilaresJ1Temp[1] := "Var".CodigoSJ1[1];
       "CodigoO1J1" := TRUE;
   END_IF;
   IF "Panel2J1Activado" AND "CodigoS2J1" THEN
       "Var".CodigoOJ1[2] := "Var".CodigoSJ1[2];
       "Var".CodigoSimilaresJ1[2] := "Var".CodigoSJ1[2];
       "Var".CodigoSimilaresJ1Temp[2] := "Var".CodigoSJ1[2];
       "CodigoO2J1" := TRUE;
   END_IF;
   IF "Panel2J1Activado" AND "CodigoS3J1" THEN
       "Var".CodigoOJ1[3] := "Var".CodigoSJ1[3];
       "Var".CodigoSimilaresJ1[3] := "Var".CodigoSJ1[3];
       "Var".CodigoSimilaresJ1Temp[3] := "Var".CodigoSJ1[3];
       "CodigoO3J1" := TRUE;
   END_IF;
END_REGION

REGION Network 4: Mensajes
   IF "CodigoS3J1" THEN "Var".VectorMensajes[1] := 1; END_IF;
   "MensajeCorrecto" := "CodigoS3J1";
   IF "CodigoO3J1" THEN "Var".VectorMensajes[2] := 1; END_IF;
   "MensajeCorrecto" := "CodigoO3J1";
   "IEC_Timer_0_DB_1".TON(IN := ("Var".VectorMensajes[2] = 1) AND ("Var".VectorMensajes[3] = 0), PT := T#1S);
   IF "IEC_Timer_0_DB_1".Q THEN "Var".VectorMensajes[3] := 1; END_IF;
   "MensajeCorrecto" := "IEC_Timer_0_DB_1".Q;
   "IEC_Timer_1_DB".TON(IN := ("Var".VectorMensajes[3] = 1) AND ("Var".VectorMensajes[4] = 0), PT := T#1S);
   IF "IEC_Timer_1_DB".Q THEN "Var".VectorMensajes[4] := 1; END_IF;
   "MensajeCorrecto" := "IEC_Timer_1_DB".Q;
   "IEC_Timer_2_DB".TON(IN := ("Var".VectorMensajes[4] = 1) AND ("Var".VectorMensajes[5] = 0), PT := T#1S);
   IF "IEC_Timer_2_DB".Q THEN "Var".VectorMensajes[5] := 1; END_IF;
   "MensajeCorrecto" := "IEC_Timer_2_DB".Q;
   "IEC_Timer_3_DB".TON(IN := ("Var".VectorMensajes[5] = 1) AND ("Var".VectorMensajes[6] = 0), PT := T#1S);
   IF "IEC_Timer_3_DB".Q THEN "Var".VectorMensajes[6] := 1; END_IF;
   "MensajeCorrecto" := "IEC_Timer_3_DB".Q;
   "IEC_Timer_4_DB".TON(IN := ("Var".VectorMensajes[6] = 1) AND ("Var".VectorMensajes[7] = 0), PT := T#1S);
   IF "IEC_Timer_4_DB".Q THEN "Var".VectorMensajes[7] := 1; END_IF;
   "MensajeCorrecto" := "IEC_Timer_4_DB".Q;
   "IEC_Timer_5_DB".TON(IN := ("Var".VectorMensajes[7] = 1) AND ("Var".VectorMensajes[8] = 0), PT := T#1S);
   IF "IEC_Timer_5_DB".Q THEN "Var".VectorMensajes[8] := 1; END_IF;
   "MensajeCorrecto" := "IEC_Timer_5_DB".Q;
   IF "IEC_Timer_5_DB".Q THEN "Bounce1" := TRUE; END_IF;
END_REGION

REGION Network 5: ActivarOtroPanel
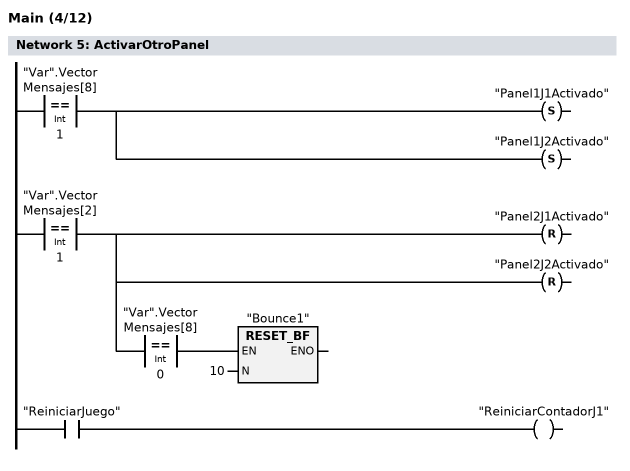
   // no SCL statement known for RBitfield: written as a call
   IF "Var".VectorMensajes[8] = 1 THEN
       "Panel1J1Activado" := TRUE;
       "Panel1J2Activado" := TRUE;
   END_IF;
   #_w1 := "Var".VectorMensajes[2] = 1;
   IF #_w1 THEN
       "Panel2J1Activado" := FALSE;
       "Panel2J2Activado" := FALSE;
   END_IF;
   IF #_w1 AND ("Var".VectorMensajes[8] = 0) THEN RESET_BF(operand := "Bounce1", n := 10); END_IF;
   "ReiniciarContadorJ1" := "ReiniciarJuego";
END_REGION

REGION Network 6: Seleccionar Intentos
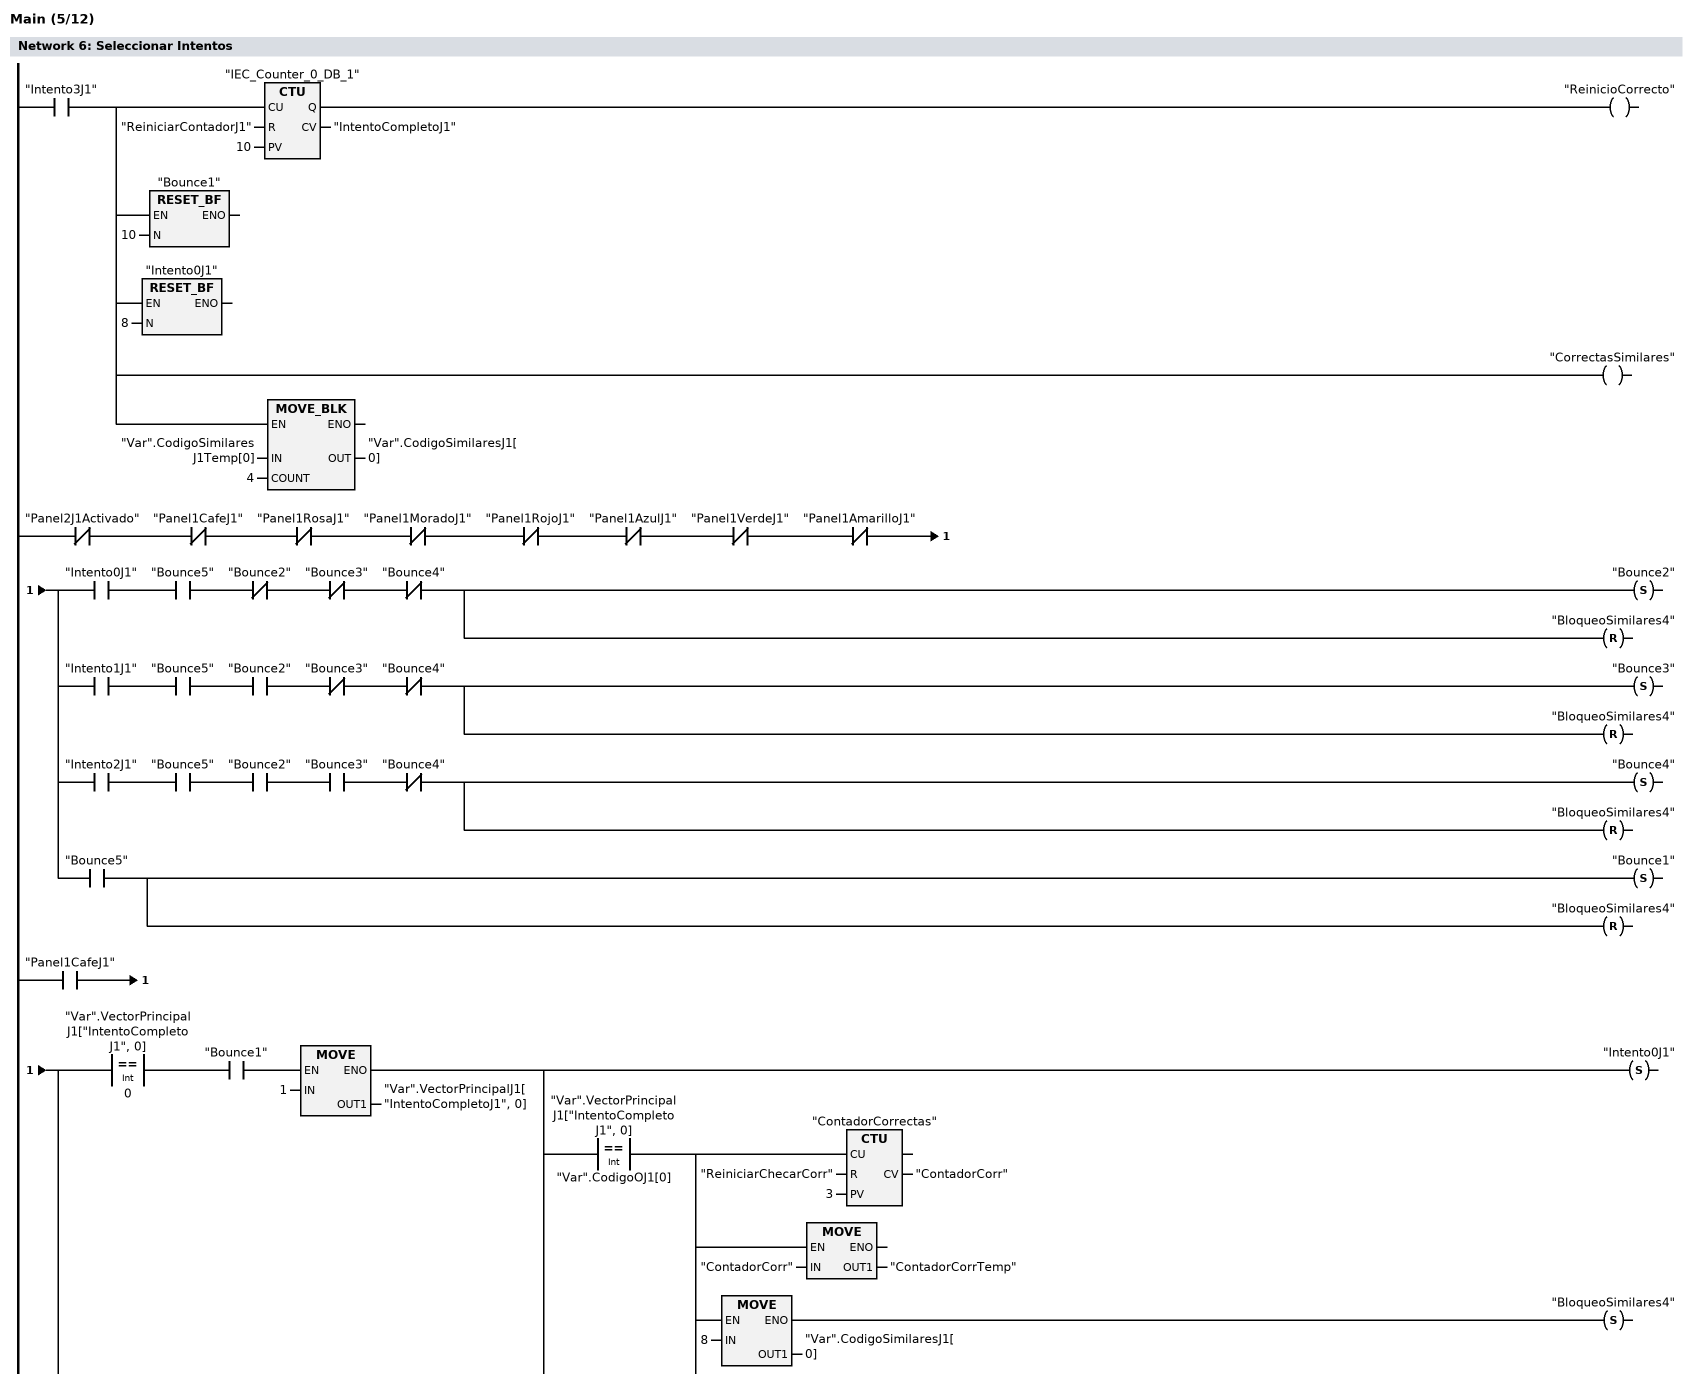
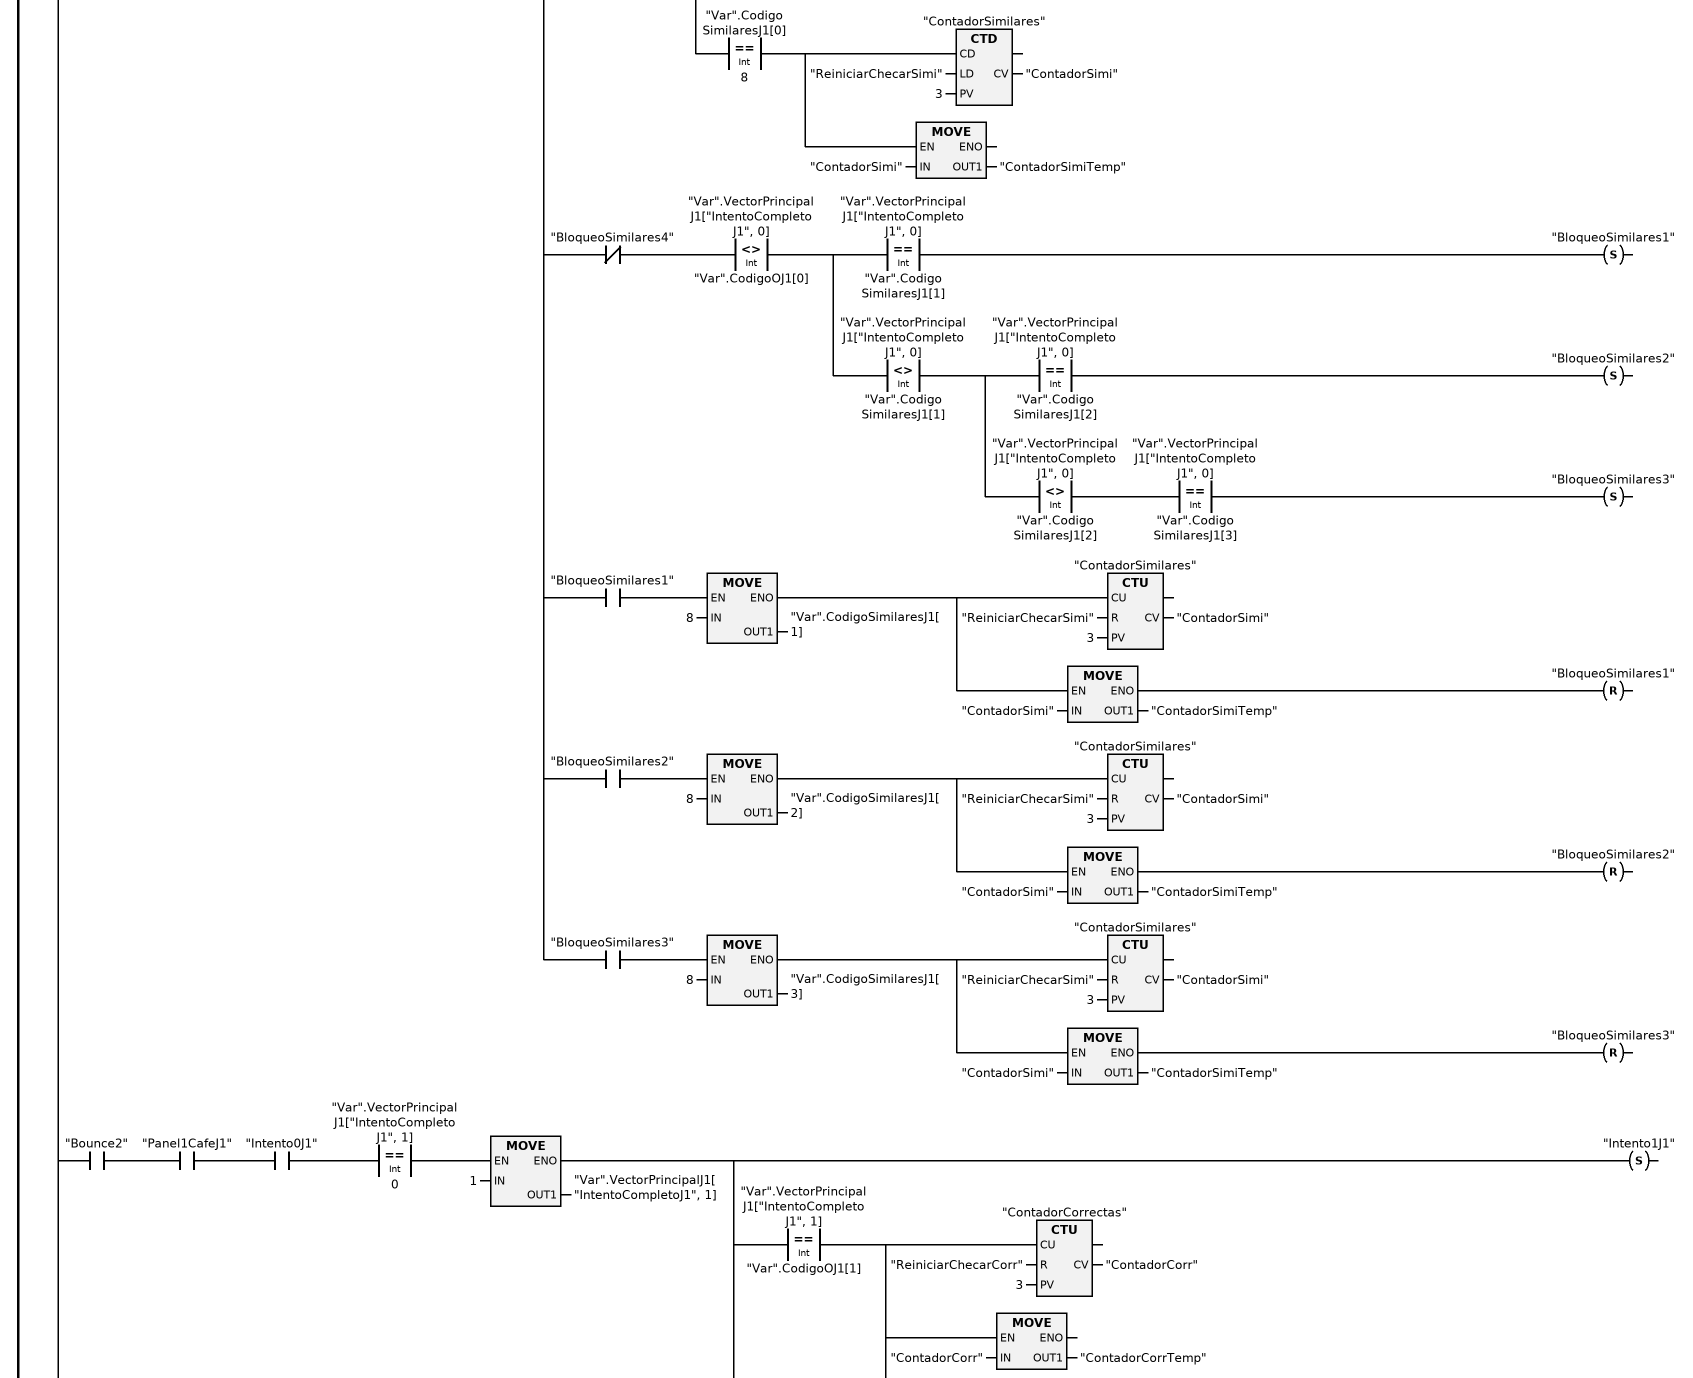
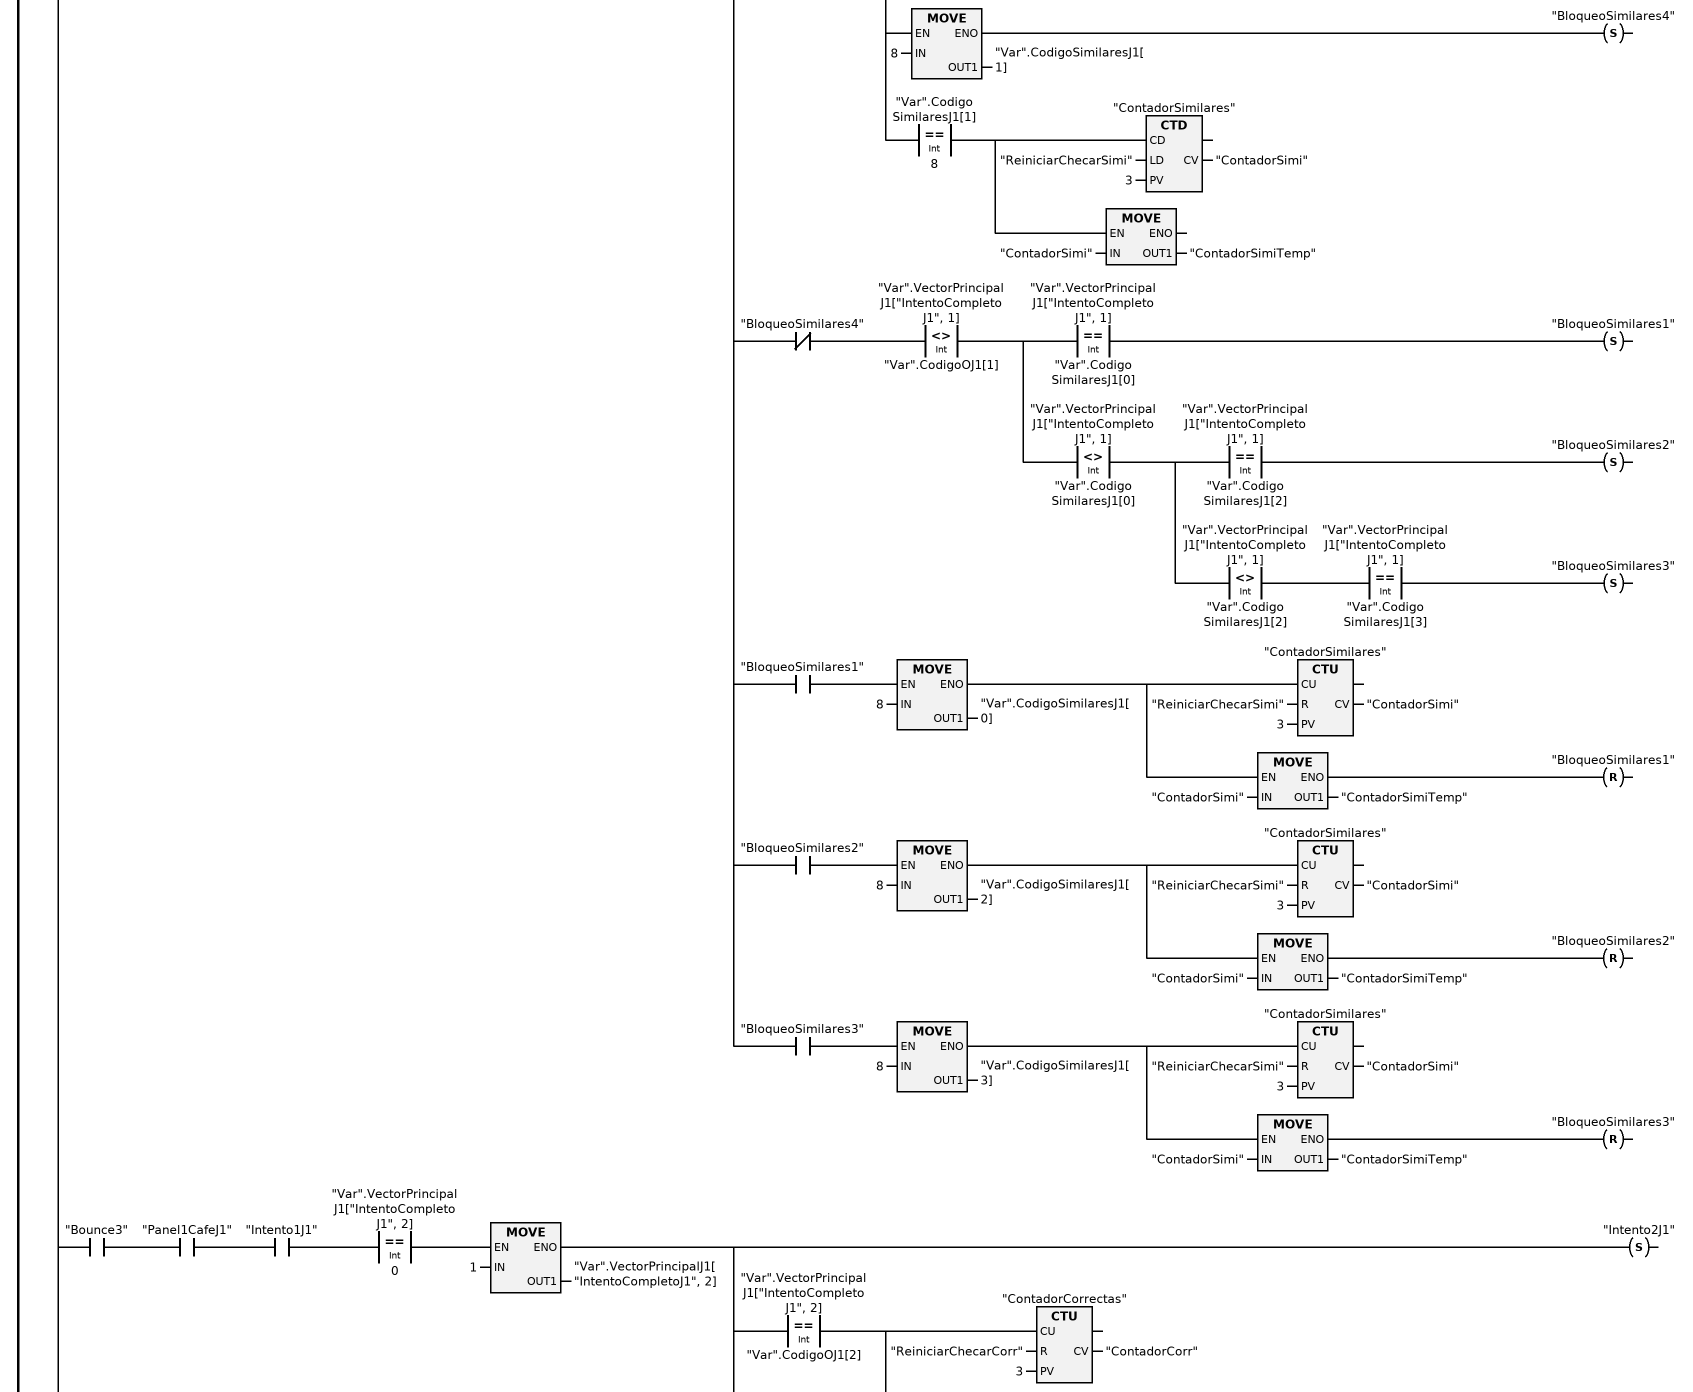
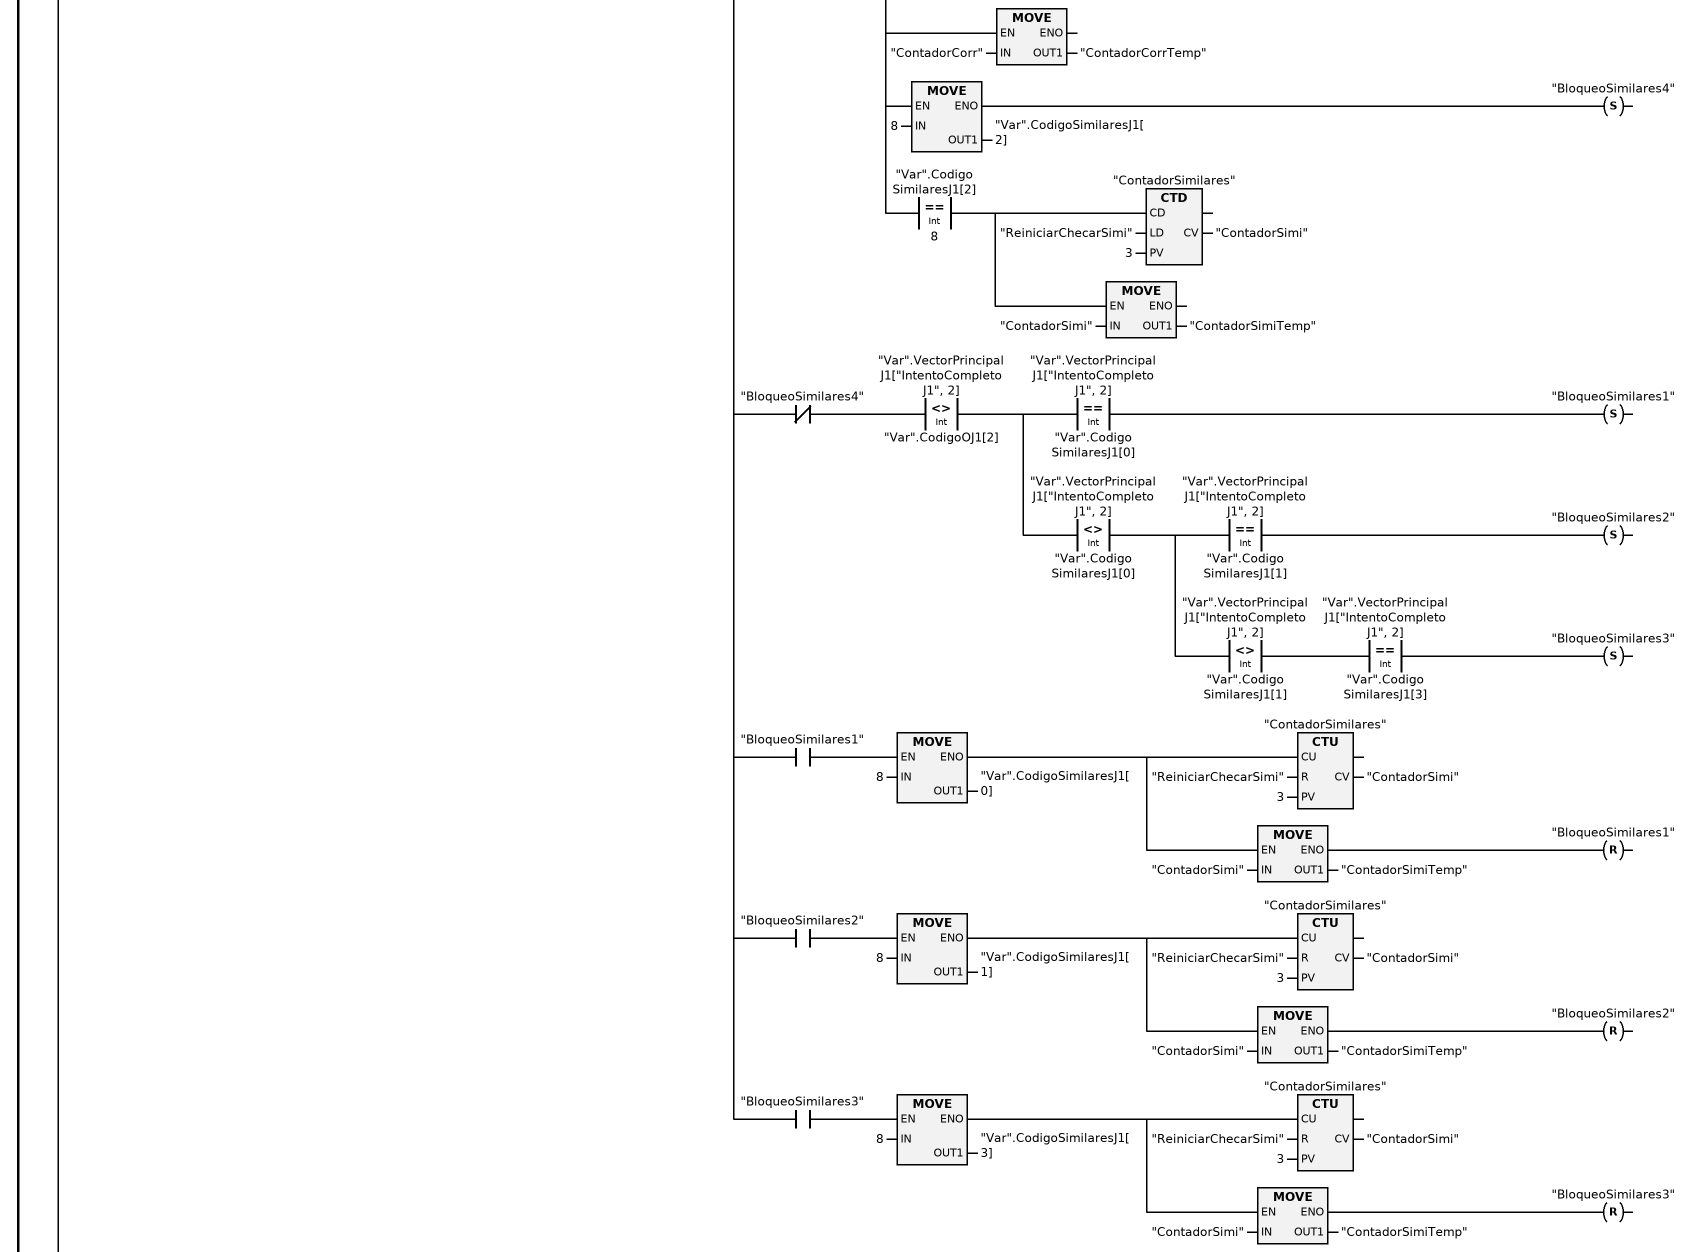
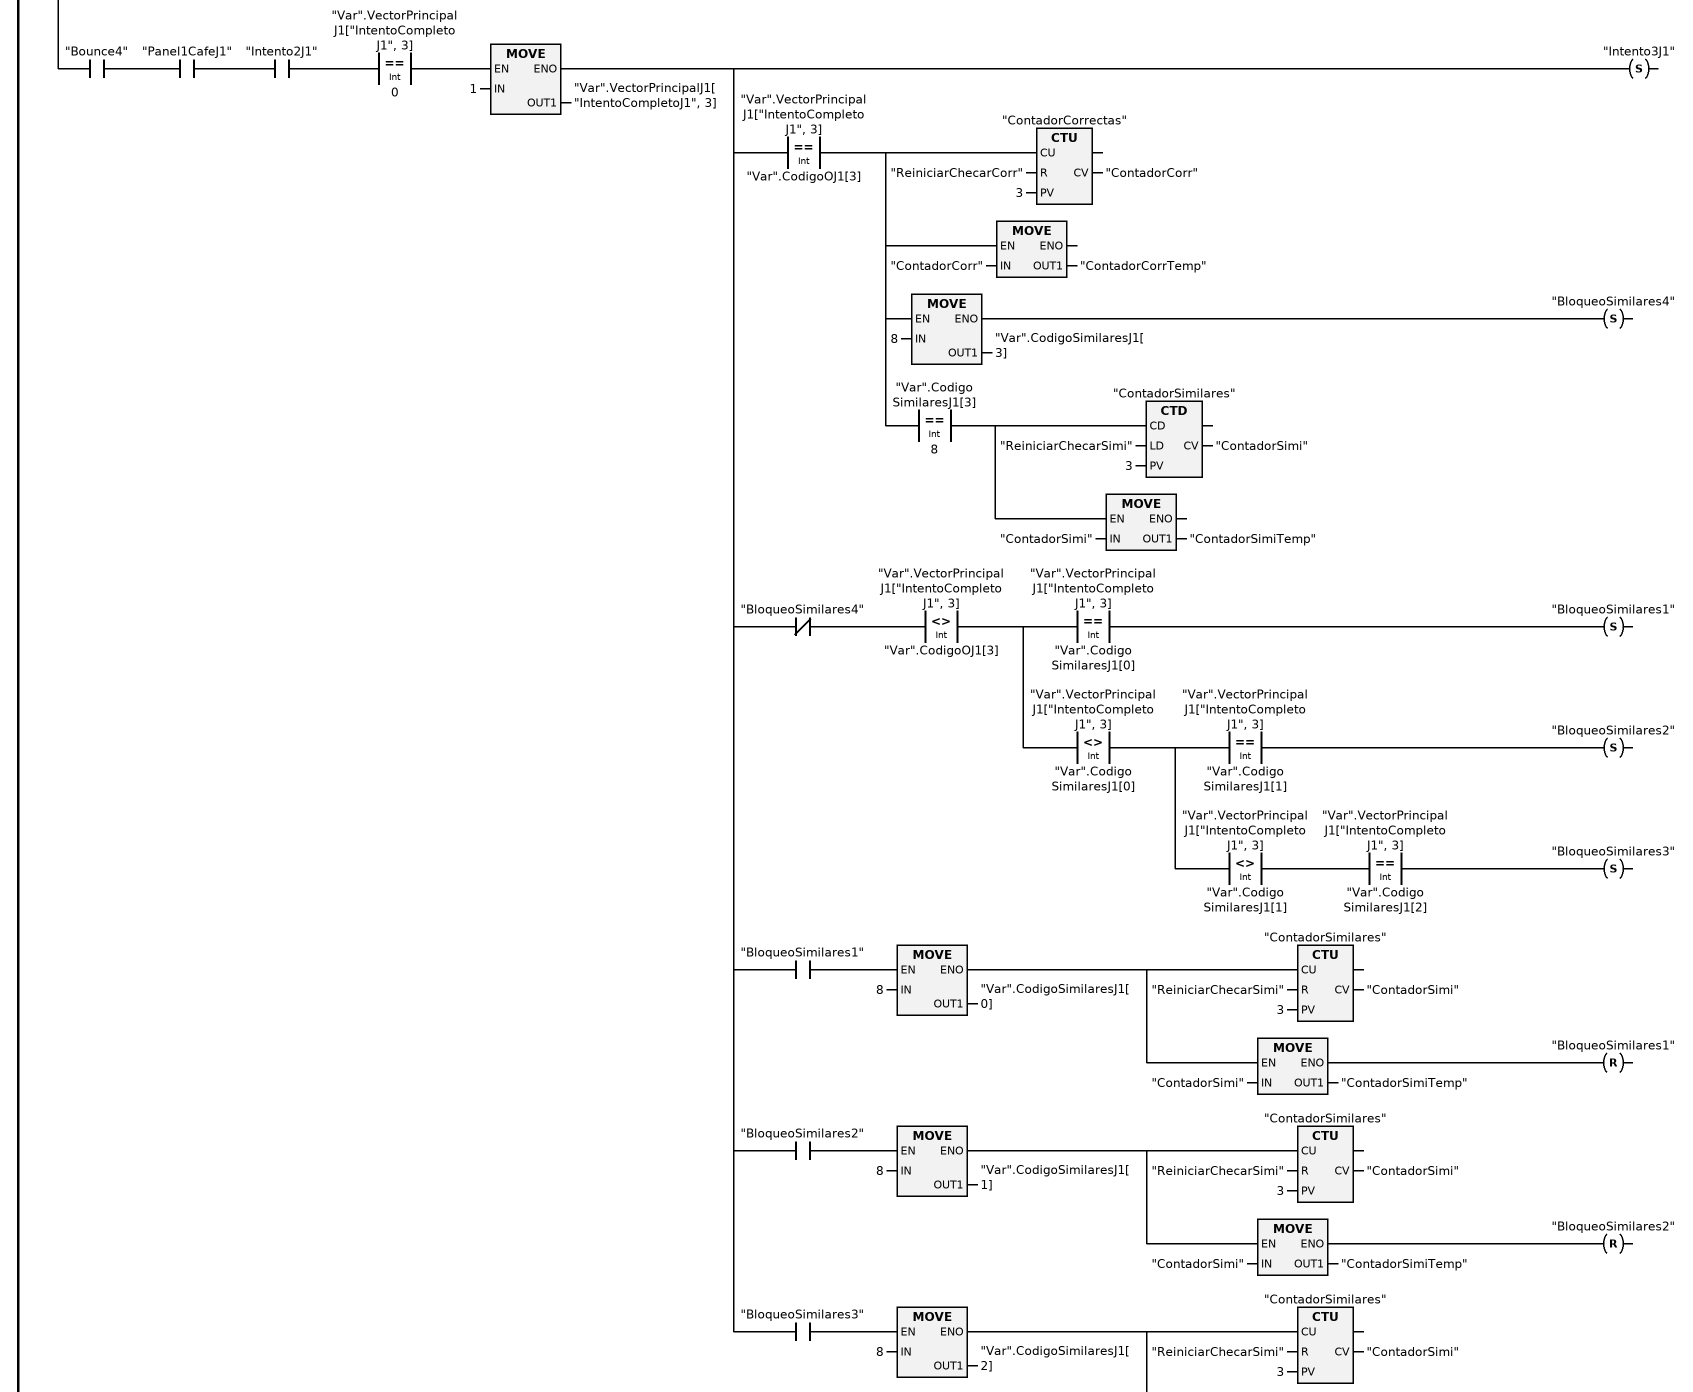
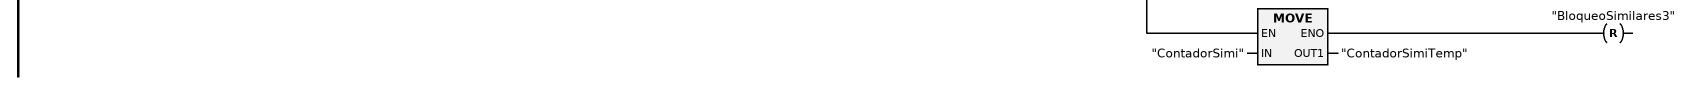
   // no SCL statement known for RBitfield: written as a call
   "IEC_Counter_0_DB_1".CTU(CU := "Intento3J1", R := "ReiniciarContadorJ1", PV := 10, CV => "IntentoCompletoJ1");
   "ReinicioCorrecto" := "IEC_Counter_0_DB_1".Q;
   #_w1 := "Intento3J1";
   IF #_w1 THEN
       RESET_BF(operand := "Bounce1", n := 10);
       RESET_BF(operand := "Intento0J1", n := 8);
   END_IF;
   "CorrectasSimilares" := #_w1;
   IF #_w1 THEN
       MOVE_BLK(IN := "Var".CodigoSimilaresJ1Temp[0], COUNT := 4, OUT => "Var".CodigoSimilaresJ1[0]);
   END_IF;
   #_w2 := NOT "Panel2J1Activado" AND NOT "Panel1CafeJ1" AND NOT "Panel1RosaJ1" AND NOT "Panel1MoradoJ1" AND NOT "Panel1RojoJ1" AND NOT "Panel1AzulJ1" AND NOT "Panel1VerdeJ1" AND NOT "Panel1AmarilloJ1";
   #_w3 := #_w2 AND "Intento0J1" AND "Bounce5" AND NOT "Bounce2" AND NOT "Bounce3" AND NOT "Bounce4";
   IF #_w3 THEN
       "Bounce2" := TRUE;
       "BloqueoSimilares4" := FALSE;
   END_IF;
   #_w4 := #_w2 AND "Intento1J1" AND "Bounce5" AND "Bounce2" AND NOT "Bounce3" AND NOT "Bounce4";
   IF #_w4 THEN
       "Bounce3" := TRUE;
       "BloqueoSimilares4" := FALSE;
   END_IF;
   #_w5 := #_w2 AND "Intento2J1" AND "Bounce5" AND "Bounce2" AND "Bounce3" AND NOT "Bounce4";
   IF #_w5 THEN
       "Bounce4" := TRUE;
       "BloqueoSimilares4" := FALSE;
   END_IF;
   IF #_w2 AND "Bounce5" THEN
       "Bounce1" := TRUE;
       "BloqueoSimilares4" := FALSE;
   END_IF;
   #_w6 := "Panel1CafeJ1" AND ("Var".VectorPrincipalJ1["IntentoCompletoJ1", 0] = 0) AND "Bounce1";
   IF #_w6 THEN
       "Var".VectorPrincipalJ1["IntentoCompletoJ1", 0] := 1;
       "Intento0J1" := TRUE;
   END_IF;
   #_w7 := #_w6 AND ("Var".VectorPrincipalJ1["IntentoCompletoJ1", 0] = "Var".CodigoOJ1[0]);
   "ContadorCorrectas".CTU(CU := #_w7, R := "ReiniciarChecarCorr", PV := 3, CV => "ContadorCorr");
   IF #_w7 THEN
       "ContadorCorrTemp" := "ContadorCorr";
       "Var".CodigoSimilaresJ1[0] := 8;
       "BloqueoSimilares4" := TRUE;
   END_IF;
   #_w8 := #_w7 AND ("Var".CodigoSimilaresJ1[0] = 8);
   "ContadorSimilares".CTD(CD := #_w8, LD := "ReiniciarChecarSimi", PV := 3, CV => "ContadorSimi");
   IF #_w8 THEN "ContadorSimiTemp" := "ContadorSimi"; END_IF;
   #_w9 := #_w6 AND NOT "BloqueoSimilares4" AND ("Var".VectorPrincipalJ1["IntentoCompletoJ1", 0] <> "Var".CodigoOJ1[0]);
   IF #_w9 AND ("Var".VectorPrincipalJ1["IntentoCompletoJ1", 0] = "Var".CodigoSimilaresJ1[1]) THEN
       "BloqueoSimilares1" := TRUE;
   END_IF;
   #_w10 := #_w9 AND ("Var".VectorPrincipalJ1["IntentoCompletoJ1", 0] <> "Var".CodigoSimilaresJ1[1]);
   IF #_w10 AND ("Var".VectorPrincipalJ1["IntentoCompletoJ1", 0] = "Var".CodigoSimilaresJ1[2]) THEN
       "BloqueoSimilares2" := TRUE;
   END_IF;
   IF #_w10 AND ("Var".VectorPrincipalJ1["IntentoCompletoJ1", 0] <> "Var".CodigoSimilaresJ1[2]) AND ("Var".VectorPrincipalJ1["IntentoCompletoJ1", 0] = "Var".CodigoSimilaresJ1[3]) THEN
       "BloqueoSimilares3" := TRUE;
   END_IF;
   #_w11 := #_w6 AND "BloqueoSimilares1";
   IF #_w11 THEN "Var".CodigoSimilaresJ1[1] := 8; END_IF;
   "ContadorSimilares".CTU(CU := #_w11, R := "ReiniciarChecarSimi", PV := 3, CV => "ContadorSimi");
   IF #_w11 THEN
       "ContadorSimiTemp" := "ContadorSimi";
       "BloqueoSimilares1" := FALSE;
   END_IF;
   #_w12 := #_w6 AND "BloqueoSimilares2";
   IF #_w12 THEN "Var".CodigoSimilaresJ1[2] := 8; END_IF;
   "ContadorSimilares".CTU(CU := #_w12, R := "ReiniciarChecarSimi", PV := 3, CV => "ContadorSimi");
   IF #_w12 THEN
       "ContadorSimiTemp" := "ContadorSimi";
       "BloqueoSimilares2" := FALSE;
   END_IF;
   #_w13 := #_w6 AND "BloqueoSimilares3";
   IF #_w13 THEN "Var".CodigoSimilaresJ1[3] := 8; END_IF;
   "ContadorSimilares".CTU(CU := #_w13, R := "ReiniciarChecarSimi", PV := 3, CV => "ContadorSimi");
   IF #_w13 THEN
       "ContadorSimiTemp" := "ContadorSimi";
       "BloqueoSimilares3" := FALSE;
   END_IF;
   #_w14 := "Panel1CafeJ1" AND "Bounce2" AND "Panel1CafeJ1" AND "Intento0J1" AND ("Var".VectorPrincipalJ1["IntentoCompletoJ1", 1] = 0);
   IF #_w14 THEN
       "Var".VectorPrincipalJ1["IntentoCompletoJ1", 1] := 1;
       "Intento1J1" := TRUE;
   END_IF;
   #_w15 := #_w14 AND ("Var".VectorPrincipalJ1["IntentoCompletoJ1", 1] = "Var".CodigoOJ1[1]);
   "ContadorCorrectas".CTU(CU := #_w15, R := "ReiniciarChecarCorr", PV := 3, CV => "ContadorCorr");
   IF #_w15 THEN
       "ContadorCorrTemp" := "ContadorCorr";
       "Var".CodigoSimilaresJ1[1] := 8;
       "BloqueoSimilares4" := TRUE;
   END_IF;
   #_w16 := #_w15 AND ("Var".CodigoSimilaresJ1[1] = 8);
   "ContadorSimilares".CTD(CD := #_w16, LD := "ReiniciarChecarSimi", PV := 3, CV => "ContadorSimi");
   IF #_w16 THEN "ContadorSimiTemp" := "ContadorSimi"; END_IF;
   #_w17 := #_w14 AND NOT "BloqueoSimilares4" AND ("Var".VectorPrincipalJ1["IntentoCompletoJ1", 1] <> "Var".CodigoOJ1[1]);
   IF #_w17 AND ("Var".VectorPrincipalJ1["IntentoCompletoJ1", 1] = "Var".CodigoSimilaresJ1[0]) THEN
       "BloqueoSimilares1" := TRUE;
   END_IF;
   #_w18 := #_w17 AND ("Var".VectorPrincipalJ1["IntentoCompletoJ1", 1] <> "Var".CodigoSimilaresJ1[0]);
   IF #_w18 AND ("Var".VectorPrincipalJ1["IntentoCompletoJ1", 1] = "Var".CodigoSimilaresJ1[2]) THEN
       "BloqueoSimilares2" := TRUE;
   END_IF;
   IF #_w18 AND ("Var".VectorPrincipalJ1["IntentoCompletoJ1", 1] <> "Var".CodigoSimilaresJ1[2]) AND ("Var".VectorPrincipalJ1["IntentoCompletoJ1", 1] = "Var".CodigoSimilaresJ1[3]) THEN
       "BloqueoSimilares3" := TRUE;
   END_IF;
   #_w19 := #_w14 AND "BloqueoSimilares1";
   IF #_w19 THEN "Var".CodigoSimilaresJ1[0] := 8; END_IF;
   "ContadorSimilares".CTU(CU := #_w19, R := "ReiniciarChecarSimi", PV := 3, CV => "ContadorSimi");
   IF #_w19 THEN
       "ContadorSimiTemp" := "ContadorSimi";
       "BloqueoSimilares1" := FALSE;
   END_IF;
   #_w20 := #_w14 AND "BloqueoSimilares2";
   IF #_w20 THEN "Var".CodigoSimilaresJ1[2] := 8; END_IF;
   "ContadorSimilares".CTU(CU := #_w20, R := "ReiniciarChecarSimi", PV := 3, CV => "ContadorSimi");
   IF #_w20 THEN
       "ContadorSimiTemp" := "ContadorSimi";
       "BloqueoSimilares2" := FALSE;
   END_IF;
   #_w21 := #_w14 AND "BloqueoSimilares3";
   IF #_w21 THEN "Var".CodigoSimilaresJ1[3] := 8; END_IF;
   "ContadorSimilares".CTU(CU := #_w21, R := "ReiniciarChecarSimi", PV := 3, CV => "ContadorSimi");
   IF #_w21 THEN
       "ContadorSimiTemp" := "ContadorSimi";
       "BloqueoSimilares3" := FALSE;
   END_IF;
   #_w22 := "Panel1CafeJ1" AND "Bounce3" AND "Panel1CafeJ1" AND "Intento1J1" AND ("Var".VectorPrincipalJ1["IntentoCompletoJ1", 2] = 0);
   IF #_w22 THEN
       "Var".VectorPrincipalJ1["IntentoCompletoJ1", 2] := 1;
       "Intento2J1" := TRUE;
   END_IF;
   #_w23 := #_w22 AND ("Var".VectorPrincipalJ1["IntentoCompletoJ1", 2] = "Var".CodigoOJ1[2]);
   "ContadorCorrectas".CTU(CU := #_w23, R := "ReiniciarChecarCorr", PV := 3, CV => "ContadorCorr");
   IF #_w23 THEN
       "ContadorCorrTemp" := "ContadorCorr";
       "Var".CodigoSimilaresJ1[2] := 8;
       "BloqueoSimilares4" := TRUE;
   END_IF;
   #_w24 := #_w23 AND ("Var".CodigoSimilaresJ1[2] = 8);
   "ContadorSimilares".CTD(CD := #_w24, LD := "ReiniciarChecarSimi", PV := 3, CV => "ContadorSimi");
   IF #_w24 THEN "ContadorSimiTemp" := "ContadorSimi"; END_IF;
   #_w25 := #_w22 AND NOT "BloqueoSimilares4" AND ("Var".VectorPrincipalJ1["IntentoCompletoJ1", 2] <> "Var".CodigoOJ1[2]);
   IF #_w25 AND ("Var".VectorPrincipalJ1["IntentoCompletoJ1", 2] = "Var".CodigoSimilaresJ1[0]) THEN
       "BloqueoSimilares1" := TRUE;
   END_IF;
   #_w26 := #_w25 AND ("Var".VectorPrincipalJ1["IntentoCompletoJ1", 2] <> "Var".CodigoSimilaresJ1[0]);
   IF #_w26 AND ("Var".VectorPrincipalJ1["IntentoCompletoJ1", 2] = "Var".CodigoSimilaresJ1[1]) THEN
       "BloqueoSimilares2" := TRUE;
   END_IF;
   IF #_w26 AND ("Var".VectorPrincipalJ1["IntentoCompletoJ1", 2] <> "Var".CodigoSimilaresJ1[1]) AND ("Var".VectorPrincipalJ1["IntentoCompletoJ1", 2] = "Var".CodigoSimilaresJ1[3]) THEN
       "BloqueoSimilares3" := TRUE;
   END_IF;
   #_w27 := #_w22 AND "BloqueoSimilares1";
   IF #_w27 THEN "Var".CodigoSimilaresJ1[0] := 8; END_IF;
   "ContadorSimilares".CTU(CU := #_w27, R := "ReiniciarChecarSimi", PV := 3, CV => "ContadorSimi");
   IF #_w27 THEN
       "ContadorSimiTemp" := "ContadorSimi";
       "BloqueoSimilares1" := FALSE;
   END_IF;
   #_w28 := #_w22 AND "BloqueoSimilares2";
   IF #_w28 THEN "Var".CodigoSimilaresJ1[1] := 8; END_IF;
   "ContadorSimilares".CTU(CU := #_w28, R := "ReiniciarChecarSimi", PV := 3, CV => "ContadorSimi");
   IF #_w28 THEN
       "ContadorSimiTemp" := "ContadorSimi";
       "BloqueoSimilares2" := FALSE;
   END_IF;
   #_w29 := #_w22 AND "BloqueoSimilares3";
   IF #_w29 THEN "Var".CodigoSimilaresJ1[3] := 8; END_IF;
   "ContadorSimilares".CTU(CU := #_w29, R := "ReiniciarChecarSimi", PV := 3, CV => "ContadorSimi");
   IF #_w29 THEN
       "ContadorSimiTemp" := "ContadorSimi";
       "BloqueoSimilares3" := FALSE;
   END_IF;
   #_w30 := "Panel1CafeJ1" AND "Bounce4" AND "Panel1CafeJ1" AND "Intento2J1" AND ("Var".VectorPrincipalJ1["IntentoCompletoJ1", 3] = 0);
   IF #_w30 THEN
       "Var".VectorPrincipalJ1["IntentoCompletoJ1", 3] := 1;
       "Intento3J1" := TRUE;
   END_IF;
   #_w31 := #_w30 AND ("Var".VectorPrincipalJ1["IntentoCompletoJ1", 3] = "Var".CodigoOJ1[3]);
   "ContadorCorrectas".CTU(CU := #_w31, R := "ReiniciarChecarCorr", PV := 3, CV => "ContadorCorr");
   IF #_w31 THEN
       "ContadorCorrTemp" := "ContadorCorr";
       "Var".CodigoSimilaresJ1[3] := 8;
       "BloqueoSimilares4" := TRUE;
   END_IF;
   #_w32 := #_w31 AND ("Var".CodigoSimilaresJ1[3] = 8);
   "ContadorSimilares".CTD(CD := #_w32, LD := "ReiniciarChecarSimi", PV := 3, CV => "ContadorSimi");
   IF #_w32 THEN "ContadorSimiTemp" := "ContadorSimi"; END_IF;
   #_w33 := #_w30 AND NOT "BloqueoSimilares4" AND ("Var".VectorPrincipalJ1["IntentoCompletoJ1", 3] <> "Var".CodigoOJ1[3]);
   IF #_w33 AND ("Var".VectorPrincipalJ1["IntentoCompletoJ1", 3] = "Var".CodigoSimilaresJ1[0]) THEN
       "BloqueoSimilares1" := TRUE;
   END_IF;
   #_w34 := #_w33 AND ("Var".VectorPrincipalJ1["IntentoCompletoJ1", 3] <> "Var".CodigoSimilaresJ1[0]);
   IF #_w34 AND ("Var".VectorPrincipalJ1["IntentoCompletoJ1", 3] = "Var".CodigoSimilaresJ1[1]) THEN
       "BloqueoSimilares2" := TRUE;
   END_IF;
   IF #_w34 AND ("Var".VectorPrincipalJ1["IntentoCompletoJ1", 3] <> "Var".CodigoSimilaresJ1[1]) AND ("Var".VectorPrincipalJ1["IntentoCompletoJ1", 3] = "Var".CodigoSimilaresJ1[2]) THEN
       "BloqueoSimilares3" := TRUE;
   END_IF;
   #_w35 := #_w30 AND "BloqueoSimilares1";
   IF #_w35 THEN "Var".CodigoSimilaresJ1[0] := 8; END_IF;
   "ContadorSimilares".CTU(CU := #_w35, R := "ReiniciarChecarSimi", PV := 3, CV => "ContadorSimi");
   IF #_w35 THEN
       "ContadorSimiTemp" := "ContadorSimi";
       "BloqueoSimilares1" := FALSE;
   END_IF;
   #_w36 := #_w30 AND "BloqueoSimilares2";
   IF #_w36 THEN "Var".CodigoSimilaresJ1[1] := 8; END_IF;
   "ContadorSimilares".CTU(CU := #_w36, R := "ReiniciarChecarSimi", PV := 3, CV => "ContadorSimi");
   IF #_w36 THEN
       "ContadorSimiTemp" := "ContadorSimi";
       "BloqueoSimilares2" := FALSE;
   END_IF;
   #_w37 := #_w30 AND "BloqueoSimilares3";
   IF #_w37 THEN "Var".CodigoSimilaresJ1[2] := 8; END_IF;
   "ContadorSimilares".CTU(CU := #_w37, R := "ReiniciarChecarSimi", PV := 3, CV => "ContadorSimi");
   IF #_w37 THEN
       "ContadorSimiTemp" := "ContadorSimi";
       "BloqueoSimilares3" := FALSE;
   END_IF;
END_REGION

REGION Network 7: Rosa
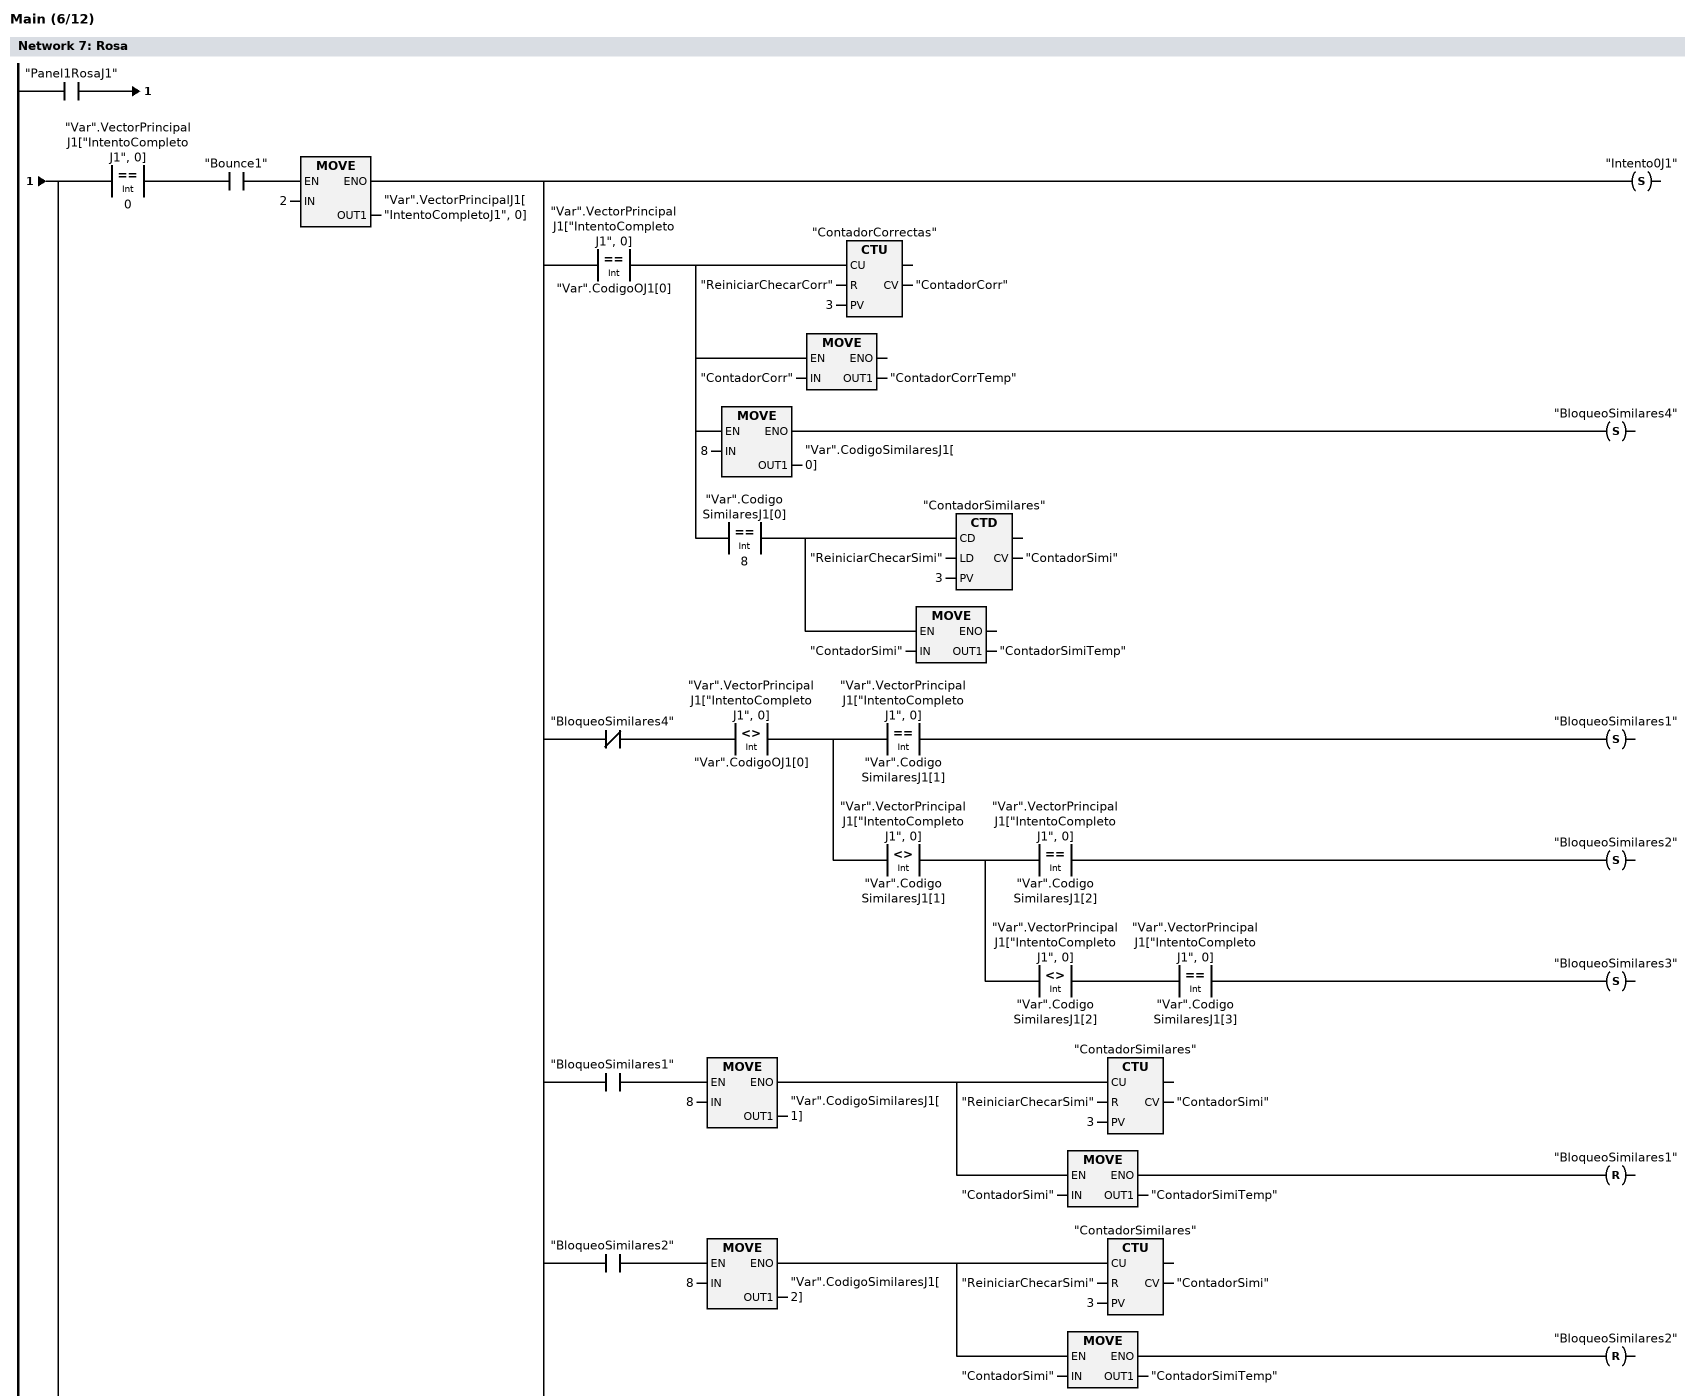
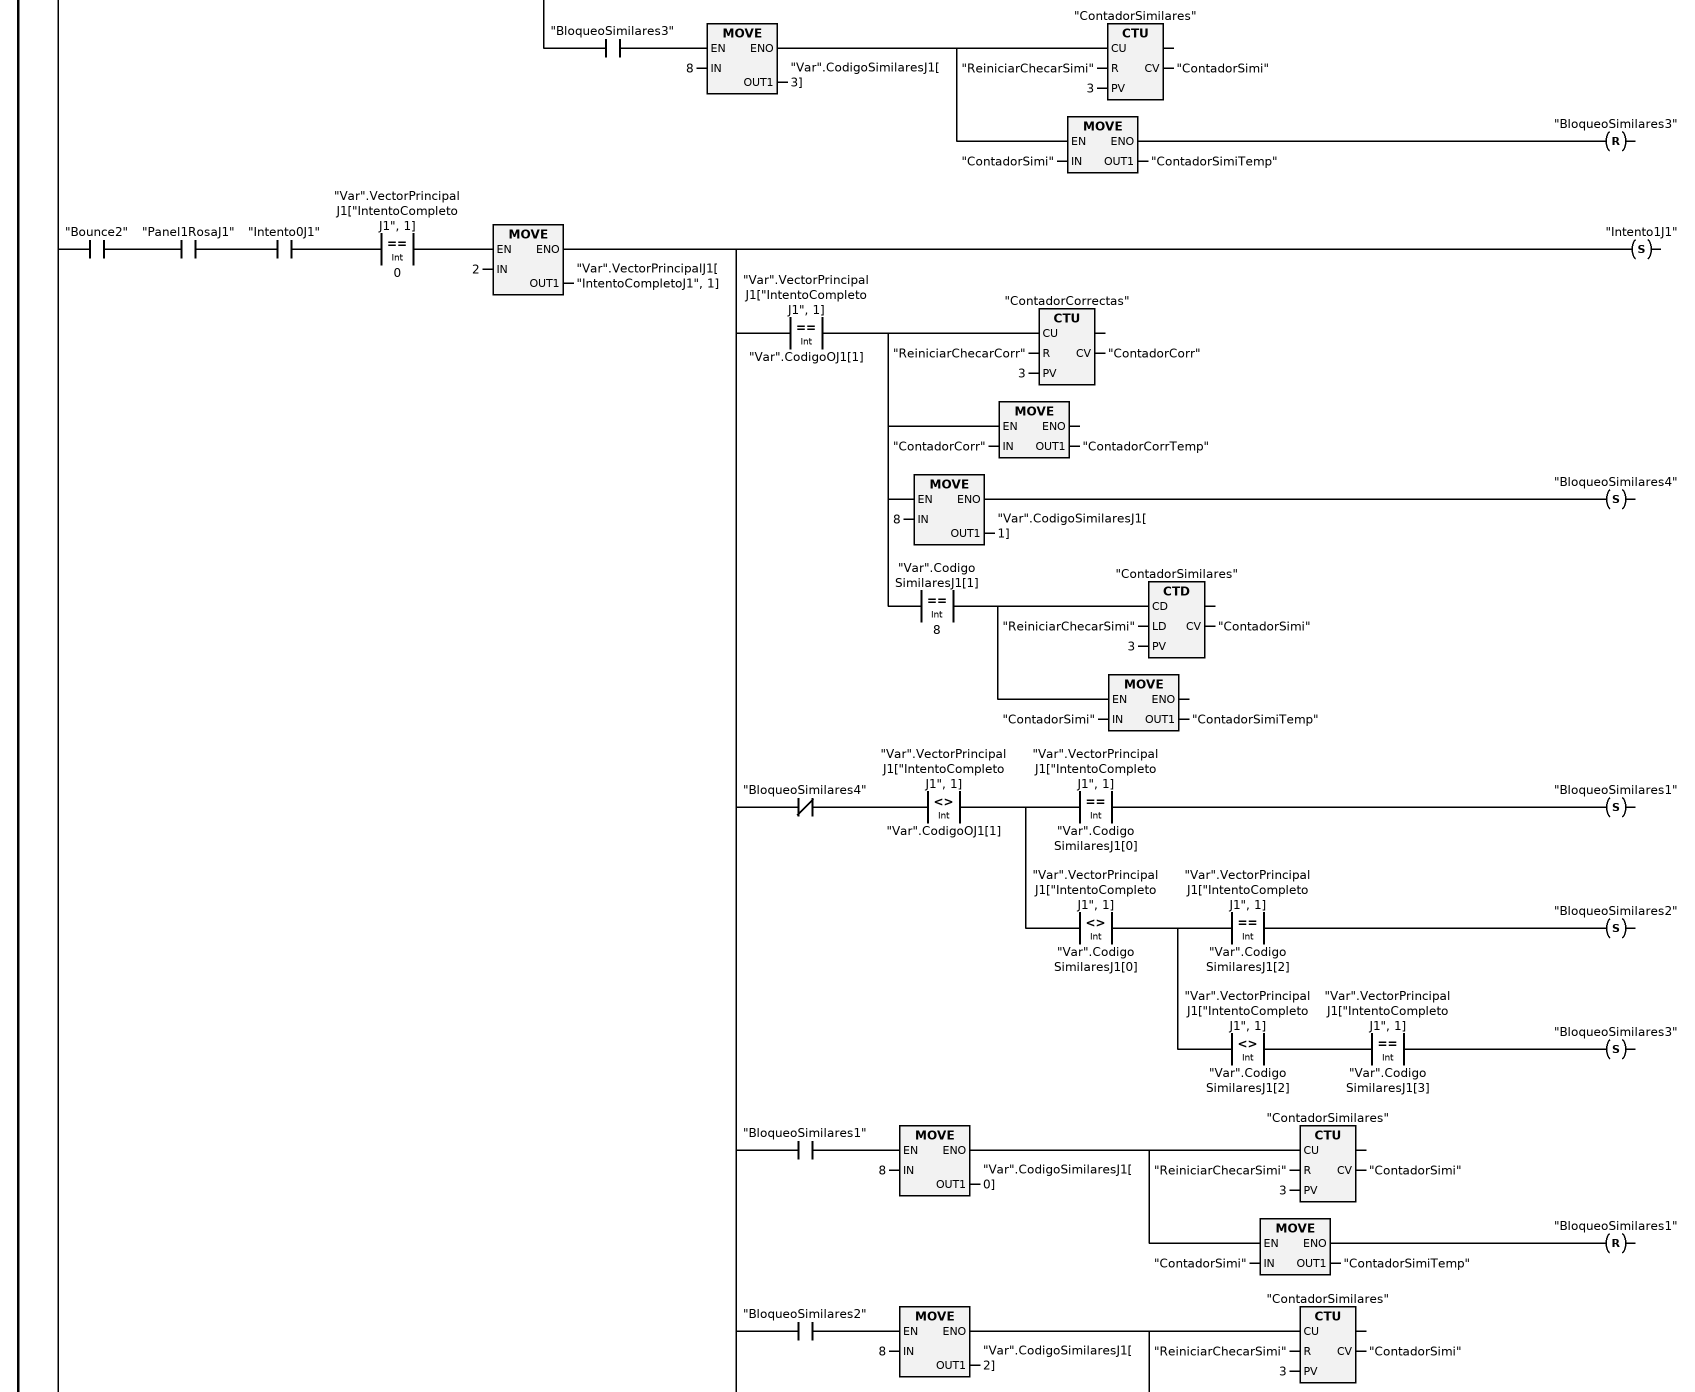
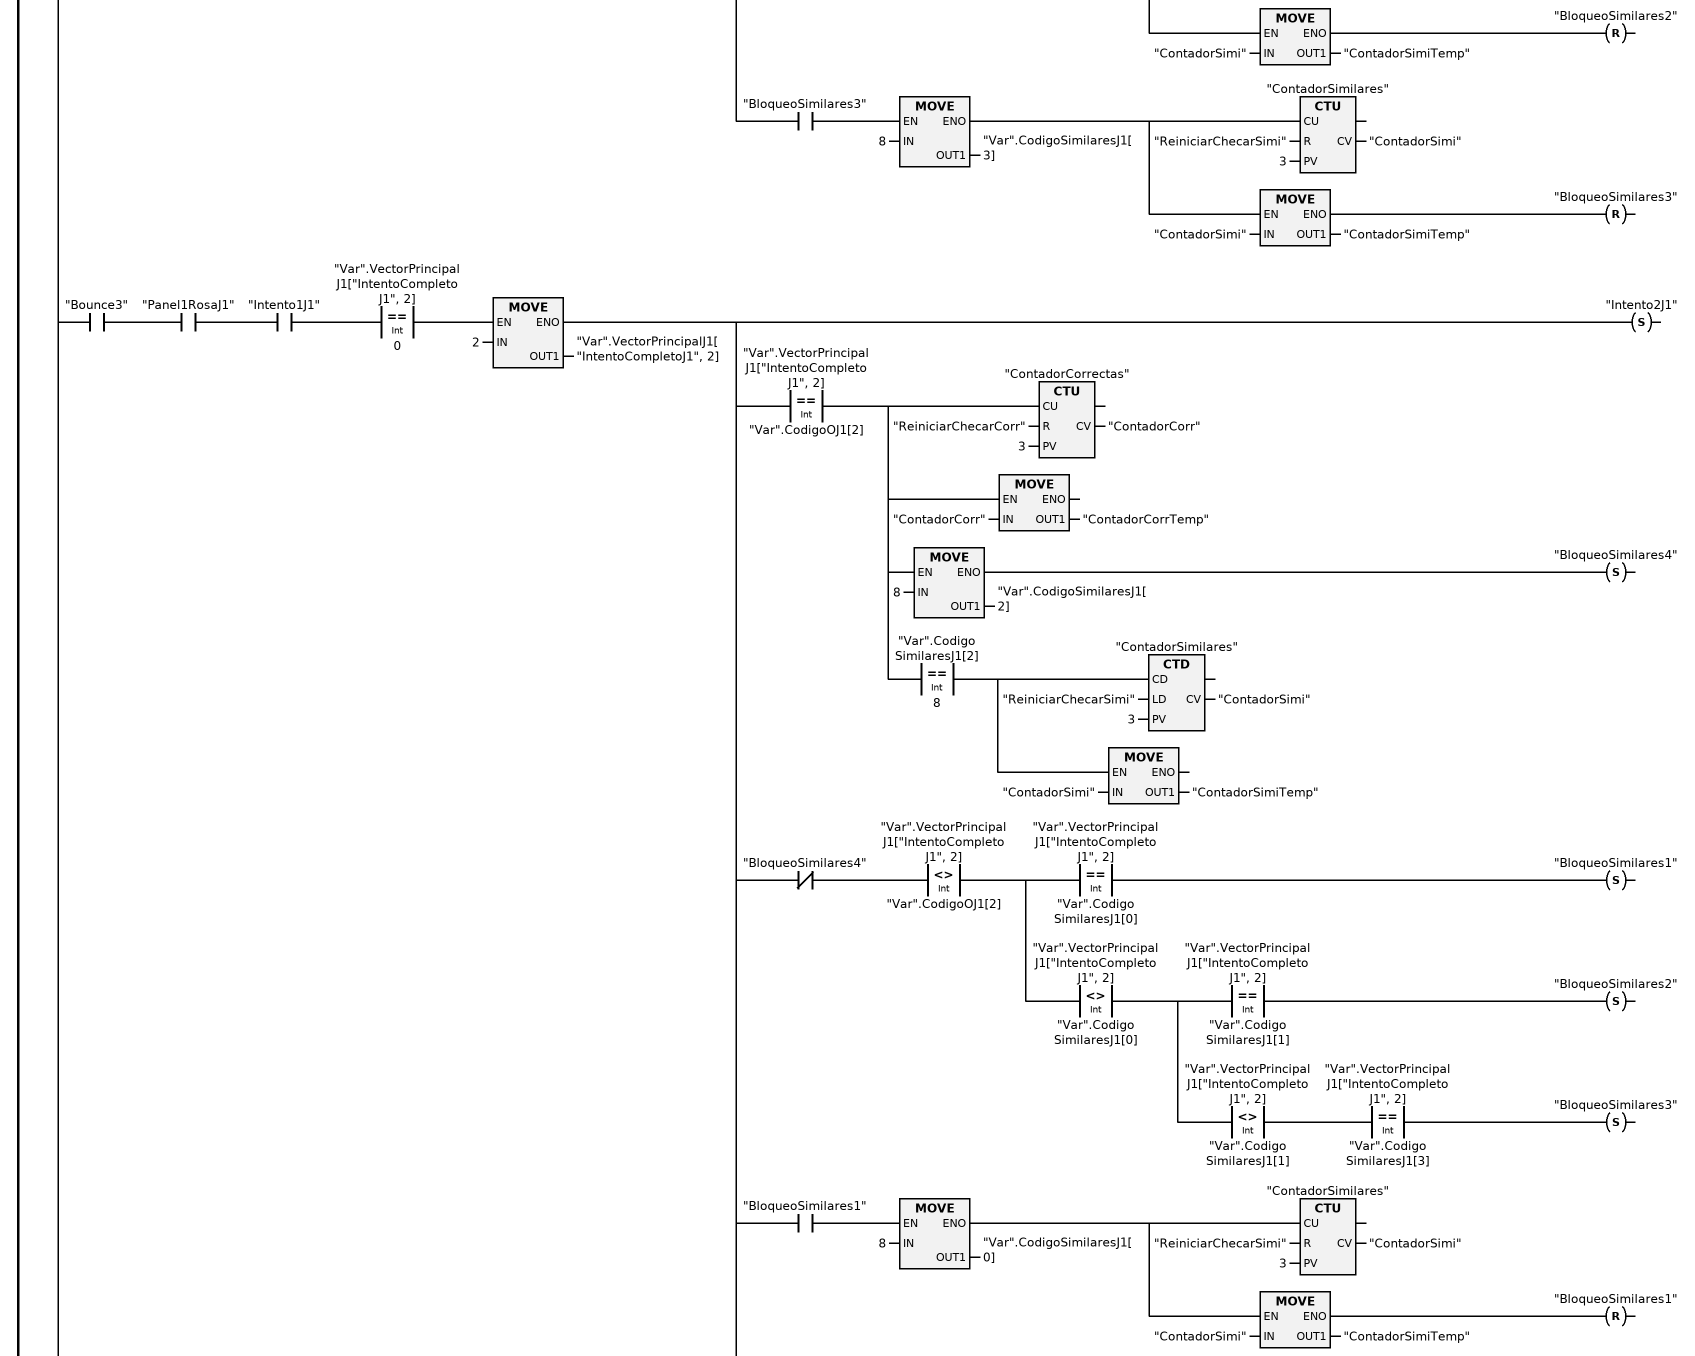
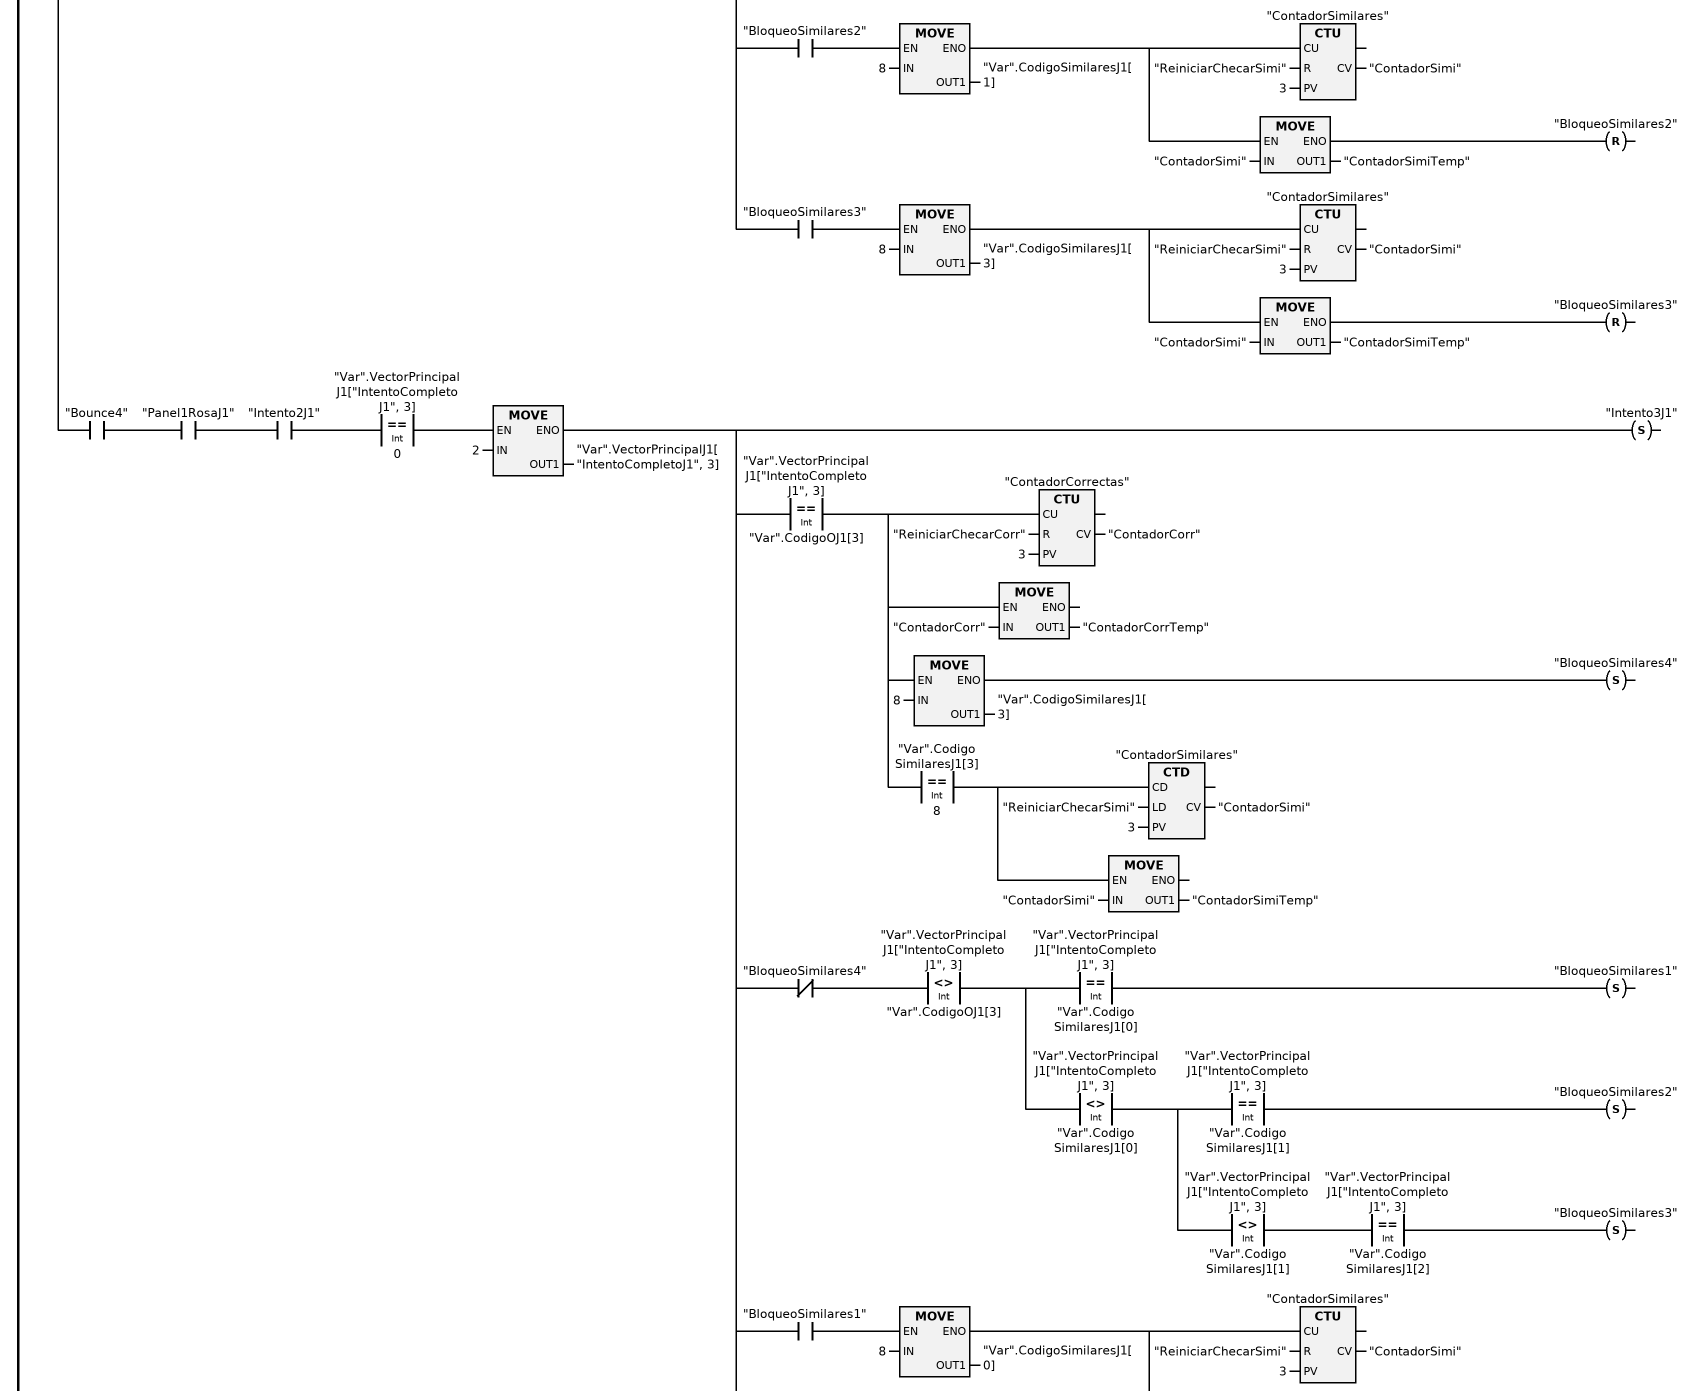
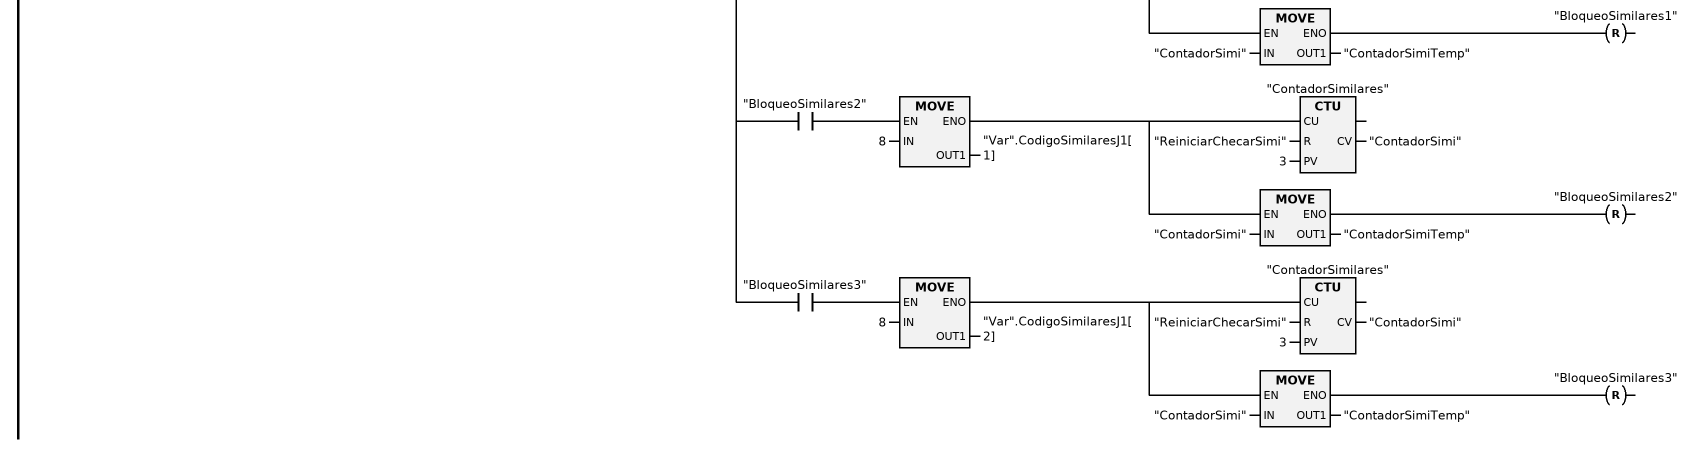
   #_w1 := "Panel1RosaJ1" AND ("Var".VectorPrincipalJ1["IntentoCompletoJ1", 0] = 0) AND "Bounce1";
   IF #_w1 THEN
       "Var".VectorPrincipalJ1["IntentoCompletoJ1", 0] := 2;
       "Intento0J1" := TRUE;
   END_IF;
   #_w2 := #_w1 AND ("Var".VectorPrincipalJ1["IntentoCompletoJ1", 0] = "Var".CodigoOJ1[0]);
   "ContadorCorrectas".CTU(CU := #_w2, R := "ReiniciarChecarCorr", PV := 3, CV => "ContadorCorr");
   IF #_w2 THEN
       "ContadorCorrTemp" := "ContadorCorr";
       "Var".CodigoSimilaresJ1[0] := 8;
       "BloqueoSimilares4" := TRUE;
   END_IF;
   #_w3 := #_w2 AND ("Var".CodigoSimilaresJ1[0] = 8);
   "ContadorSimilares".CTD(CD := #_w3, LD := "ReiniciarChecarSimi", PV := 3, CV => "ContadorSimi");
   IF #_w3 THEN "ContadorSimiTemp" := "ContadorSimi"; END_IF;
   #_w4 := #_w1 AND NOT "BloqueoSimilares4" AND ("Var".VectorPrincipalJ1["IntentoCompletoJ1", 0] <> "Var".CodigoOJ1[0]);
   IF #_w4 AND ("Var".VectorPrincipalJ1["IntentoCompletoJ1", 0] = "Var".CodigoSimilaresJ1[1]) THEN
       "BloqueoSimilares1" := TRUE;
   END_IF;
   #_w5 := #_w4 AND ("Var".VectorPrincipalJ1["IntentoCompletoJ1", 0] <> "Var".CodigoSimilaresJ1[1]);
   IF #_w5 AND ("Var".VectorPrincipalJ1["IntentoCompletoJ1", 0] = "Var".CodigoSimilaresJ1[2]) THEN
       "BloqueoSimilares2" := TRUE;
   END_IF;
   IF #_w5 AND ("Var".VectorPrincipalJ1["IntentoCompletoJ1", 0] <> "Var".CodigoSimilaresJ1[2]) AND ("Var".VectorPrincipalJ1["IntentoCompletoJ1", 0] = "Var".CodigoSimilaresJ1[3]) THEN
       "BloqueoSimilares3" := TRUE;
   END_IF;
   #_w6 := #_w1 AND "BloqueoSimilares1";
   IF #_w6 THEN "Var".CodigoSimilaresJ1[1] := 8; END_IF;
   "ContadorSimilares".CTU(CU := #_w6, R := "ReiniciarChecarSimi", PV := 3, CV => "ContadorSimi");
   IF #_w6 THEN
       "ContadorSimiTemp" := "ContadorSimi";
       "BloqueoSimilares1" := FALSE;
   END_IF;
   #_w7 := #_w1 AND "BloqueoSimilares2";
   IF #_w7 THEN "Var".CodigoSimilaresJ1[2] := 8; END_IF;
   "ContadorSimilares".CTU(CU := #_w7, R := "ReiniciarChecarSimi", PV := 3, CV => "ContadorSimi");
   IF #_w7 THEN
       "ContadorSimiTemp" := "ContadorSimi";
       "BloqueoSimilares2" := FALSE;
   END_IF;
   #_w8 := #_w1 AND "BloqueoSimilares3";
   IF #_w8 THEN "Var".CodigoSimilaresJ1[3] := 8; END_IF;
   "ContadorSimilares".CTU(CU := #_w8, R := "ReiniciarChecarSimi", PV := 3, CV => "ContadorSimi");
   IF #_w8 THEN
       "ContadorSimiTemp" := "ContadorSimi";
       "BloqueoSimilares3" := FALSE;
   END_IF;
   #_w9 := "Panel1RosaJ1" AND "Bounce2" AND "Panel1RosaJ1" AND "Intento0J1" AND ("Var".VectorPrincipalJ1["IntentoCompletoJ1", 1] = 0);
   IF #_w9 THEN
       "Var".VectorPrincipalJ1["IntentoCompletoJ1", 1] := 2;
       "Intento1J1" := TRUE;
   END_IF;
   #_w10 := #_w9 AND ("Var".VectorPrincipalJ1["IntentoCompletoJ1", 1] = "Var".CodigoOJ1[1]);
   "ContadorCorrectas".CTU(CU := #_w10, R := "ReiniciarChecarCorr", PV := 3, CV => "ContadorCorr");
   IF #_w10 THEN
       "ContadorCorrTemp" := "ContadorCorr";
       "Var".CodigoSimilaresJ1[1] := 8;
       "BloqueoSimilares4" := TRUE;
   END_IF;
   #_w11 := #_w10 AND ("Var".CodigoSimilaresJ1[1] = 8);
   "ContadorSimilares".CTD(CD := #_w11, LD := "ReiniciarChecarSimi", PV := 3, CV => "ContadorSimi");
   IF #_w11 THEN "ContadorSimiTemp" := "ContadorSimi"; END_IF;
   #_w12 := #_w9 AND NOT "BloqueoSimilares4" AND ("Var".VectorPrincipalJ1["IntentoCompletoJ1", 1] <> "Var".CodigoOJ1[1]);
   IF #_w12 AND ("Var".VectorPrincipalJ1["IntentoCompletoJ1", 1] = "Var".CodigoSimilaresJ1[0]) THEN
       "BloqueoSimilares1" := TRUE;
   END_IF;
   #_w13 := #_w12 AND ("Var".VectorPrincipalJ1["IntentoCompletoJ1", 1] <> "Var".CodigoSimilaresJ1[0]);
   IF #_w13 AND ("Var".VectorPrincipalJ1["IntentoCompletoJ1", 1] = "Var".CodigoSimilaresJ1[2]) THEN
       "BloqueoSimilares2" := TRUE;
   END_IF;
   IF #_w13 AND ("Var".VectorPrincipalJ1["IntentoCompletoJ1", 1] <> "Var".CodigoSimilaresJ1[2]) AND ("Var".VectorPrincipalJ1["IntentoCompletoJ1", 1] = "Var".CodigoSimilaresJ1[3]) THEN
       "BloqueoSimilares3" := TRUE;
   END_IF;
   #_w14 := #_w9 AND "BloqueoSimilares1";
   IF #_w14 THEN "Var".CodigoSimilaresJ1[0] := 8; END_IF;
   "ContadorSimilares".CTU(CU := #_w14, R := "ReiniciarChecarSimi", PV := 3, CV => "ContadorSimi");
   IF #_w14 THEN
       "ContadorSimiTemp" := "ContadorSimi";
       "BloqueoSimilares1" := FALSE;
   END_IF;
   #_w15 := #_w9 AND "BloqueoSimilares2";
   IF #_w15 THEN "Var".CodigoSimilaresJ1[2] := 8; END_IF;
   "ContadorSimilares".CTU(CU := #_w15, R := "ReiniciarChecarSimi", PV := 3, CV => "ContadorSimi");
   IF #_w15 THEN
       "ContadorSimiTemp" := "ContadorSimi";
       "BloqueoSimilares2" := FALSE;
   END_IF;
   #_w16 := #_w9 AND "BloqueoSimilares3";
   IF #_w16 THEN "Var".CodigoSimilaresJ1[3] := 8; END_IF;
   "ContadorSimilares".CTU(CU := #_w16, R := "ReiniciarChecarSimi", PV := 3, CV => "ContadorSimi");
   IF #_w16 THEN
       "ContadorSimiTemp" := "ContadorSimi";
       "BloqueoSimilares3" := FALSE;
   END_IF;
   #_w17 := "Panel1RosaJ1" AND "Bounce3" AND "Panel1RosaJ1" AND "Intento1J1" AND ("Var".VectorPrincipalJ1["IntentoCompletoJ1", 2] = 0);
   IF #_w17 THEN
       "Var".VectorPrincipalJ1["IntentoCompletoJ1", 2] := 2;
       "Intento2J1" := TRUE;
   END_IF;
   #_w18 := #_w17 AND ("Var".VectorPrincipalJ1["IntentoCompletoJ1", 2] = "Var".CodigoOJ1[2]);
   "ContadorCorrectas".CTU(CU := #_w18, R := "ReiniciarChecarCorr", PV := 3, CV => "ContadorCorr");
   IF #_w18 THEN
       "ContadorCorrTemp" := "ContadorCorr";
       "Var".CodigoSimilaresJ1[2] := 8;
       "BloqueoSimilares4" := TRUE;
   END_IF;
   #_w19 := #_w18 AND ("Var".CodigoSimilaresJ1[2] = 8);
   "ContadorSimilares".CTD(CD := #_w19, LD := "ReiniciarChecarSimi", PV := 3, CV => "ContadorSimi");
   IF #_w19 THEN "ContadorSimiTemp" := "ContadorSimi"; END_IF;
   #_w20 := #_w17 AND NOT "BloqueoSimilares4" AND ("Var".VectorPrincipalJ1["IntentoCompletoJ1", 2] <> "Var".CodigoOJ1[2]);
   IF #_w20 AND ("Var".VectorPrincipalJ1["IntentoCompletoJ1", 2] = "Var".CodigoSimilaresJ1[0]) THEN
       "BloqueoSimilares1" := TRUE;
   END_IF;
   #_w21 := #_w20 AND ("Var".VectorPrincipalJ1["IntentoCompletoJ1", 2] <> "Var".CodigoSimilaresJ1[0]);
   IF #_w21 AND ("Var".VectorPrincipalJ1["IntentoCompletoJ1", 2] = "Var".CodigoSimilaresJ1[1]) THEN
       "BloqueoSimilares2" := TRUE;
   END_IF;
   IF #_w21 AND ("Var".VectorPrincipalJ1["IntentoCompletoJ1", 2] <> "Var".CodigoSimilaresJ1[1]) AND ("Var".VectorPrincipalJ1["IntentoCompletoJ1", 2] = "Var".CodigoSimilaresJ1[3]) THEN
       "BloqueoSimilares3" := TRUE;
   END_IF;
   #_w22 := #_w17 AND "BloqueoSimilares1";
   IF #_w22 THEN "Var".CodigoSimilaresJ1[0] := 8; END_IF;
   "ContadorSimilares".CTU(CU := #_w22, R := "ReiniciarChecarSimi", PV := 3, CV => "ContadorSimi");
   IF #_w22 THEN
       "ContadorSimiTemp" := "ContadorSimi";
       "BloqueoSimilares1" := FALSE;
   END_IF;
   #_w23 := #_w17 AND "BloqueoSimilares2";
   IF #_w23 THEN "Var".CodigoSimilaresJ1[1] := 8; END_IF;
   "ContadorSimilares".CTU(CU := #_w23, R := "ReiniciarChecarSimi", PV := 3, CV => "ContadorSimi");
   IF #_w23 THEN
       "ContadorSimiTemp" := "ContadorSimi";
       "BloqueoSimilares2" := FALSE;
   END_IF;
   #_w24 := #_w17 AND "BloqueoSimilares3";
   IF #_w24 THEN "Var".CodigoSimilaresJ1[3] := 8; END_IF;
   "ContadorSimilares".CTU(CU := #_w24, R := "ReiniciarChecarSimi", PV := 3, CV => "ContadorSimi");
   IF #_w24 THEN
       "ContadorSimiTemp" := "ContadorSimi";
       "BloqueoSimilares3" := FALSE;
   END_IF;
   #_w25 := "Panel1RosaJ1" AND "Bounce4" AND "Panel1RosaJ1" AND "Intento2J1" AND ("Var".VectorPrincipalJ1["IntentoCompletoJ1", 3] = 0);
   IF #_w25 THEN
       "Var".VectorPrincipalJ1["IntentoCompletoJ1", 3] := 2;
       "Intento3J1" := TRUE;
   END_IF;
   #_w26 := #_w25 AND ("Var".VectorPrincipalJ1["IntentoCompletoJ1", 3] = "Var".CodigoOJ1[3]);
   "ContadorCorrectas".CTU(CU := #_w26, R := "ReiniciarChecarCorr", PV := 3, CV => "ContadorCorr");
   IF #_w26 THEN
       "ContadorCorrTemp" := "ContadorCorr";
       "Var".CodigoSimilaresJ1[3] := 8;
       "BloqueoSimilares4" := TRUE;
   END_IF;
   #_w27 := #_w26 AND ("Var".CodigoSimilaresJ1[3] = 8);
   "ContadorSimilares".CTD(CD := #_w27, LD := "ReiniciarChecarSimi", PV := 3, CV => "ContadorSimi");
   IF #_w27 THEN "ContadorSimiTemp" := "ContadorSimi"; END_IF;
   #_w28 := #_w25 AND NOT "BloqueoSimilares4" AND ("Var".VectorPrincipalJ1["IntentoCompletoJ1", 3] <> "Var".CodigoOJ1[3]);
   IF #_w28 AND ("Var".VectorPrincipalJ1["IntentoCompletoJ1", 3] = "Var".CodigoSimilaresJ1[0]) THEN
       "BloqueoSimilares1" := TRUE;
   END_IF;
   #_w29 := #_w28 AND ("Var".VectorPrincipalJ1["IntentoCompletoJ1", 3] <> "Var".CodigoSimilaresJ1[0]);
   IF #_w29 AND ("Var".VectorPrincipalJ1["IntentoCompletoJ1", 3] = "Var".CodigoSimilaresJ1[1]) THEN
       "BloqueoSimilares2" := TRUE;
   END_IF;
   IF #_w29 AND ("Var".VectorPrincipalJ1["IntentoCompletoJ1", 3] <> "Var".CodigoSimilaresJ1[1]) AND ("Var".VectorPrincipalJ1["IntentoCompletoJ1", 3] = "Var".CodigoSimilaresJ1[2]) THEN
       "BloqueoSimilares3" := TRUE;
   END_IF;
   #_w30 := #_w25 AND "BloqueoSimilares1";
   IF #_w30 THEN "Var".CodigoSimilaresJ1[0] := 8; END_IF;
   "ContadorSimilares".CTU(CU := #_w30, R := "ReiniciarChecarSimi", PV := 3, CV => "ContadorSimi");
   IF #_w30 THEN
       "ContadorSimiTemp" := "ContadorSimi";
       "BloqueoSimilares1" := FALSE;
   END_IF;
   #_w31 := #_w25 AND "BloqueoSimilares2";
   IF #_w31 THEN "Var".CodigoSimilaresJ1[1] := 8; END_IF;
   "ContadorSimilares".CTU(CU := #_w31, R := "ReiniciarChecarSimi", PV := 3, CV => "ContadorSimi");
   IF #_w31 THEN
       "ContadorSimiTemp" := "ContadorSimi";
       "BloqueoSimilares2" := FALSE;
   END_IF;
   #_w32 := #_w25 AND "BloqueoSimilares3";
   IF #_w32 THEN "Var".CodigoSimilaresJ1[2] := 8; END_IF;
   "ContadorSimilares".CTU(CU := #_w32, R := "ReiniciarChecarSimi", PV := 3, CV => "ContadorSimi");
   IF #_w32 THEN
       "ContadorSimiTemp" := "ContadorSimi";
       "BloqueoSimilares3" := FALSE;
   END_IF;
END_REGION

REGION Network 8: Morado
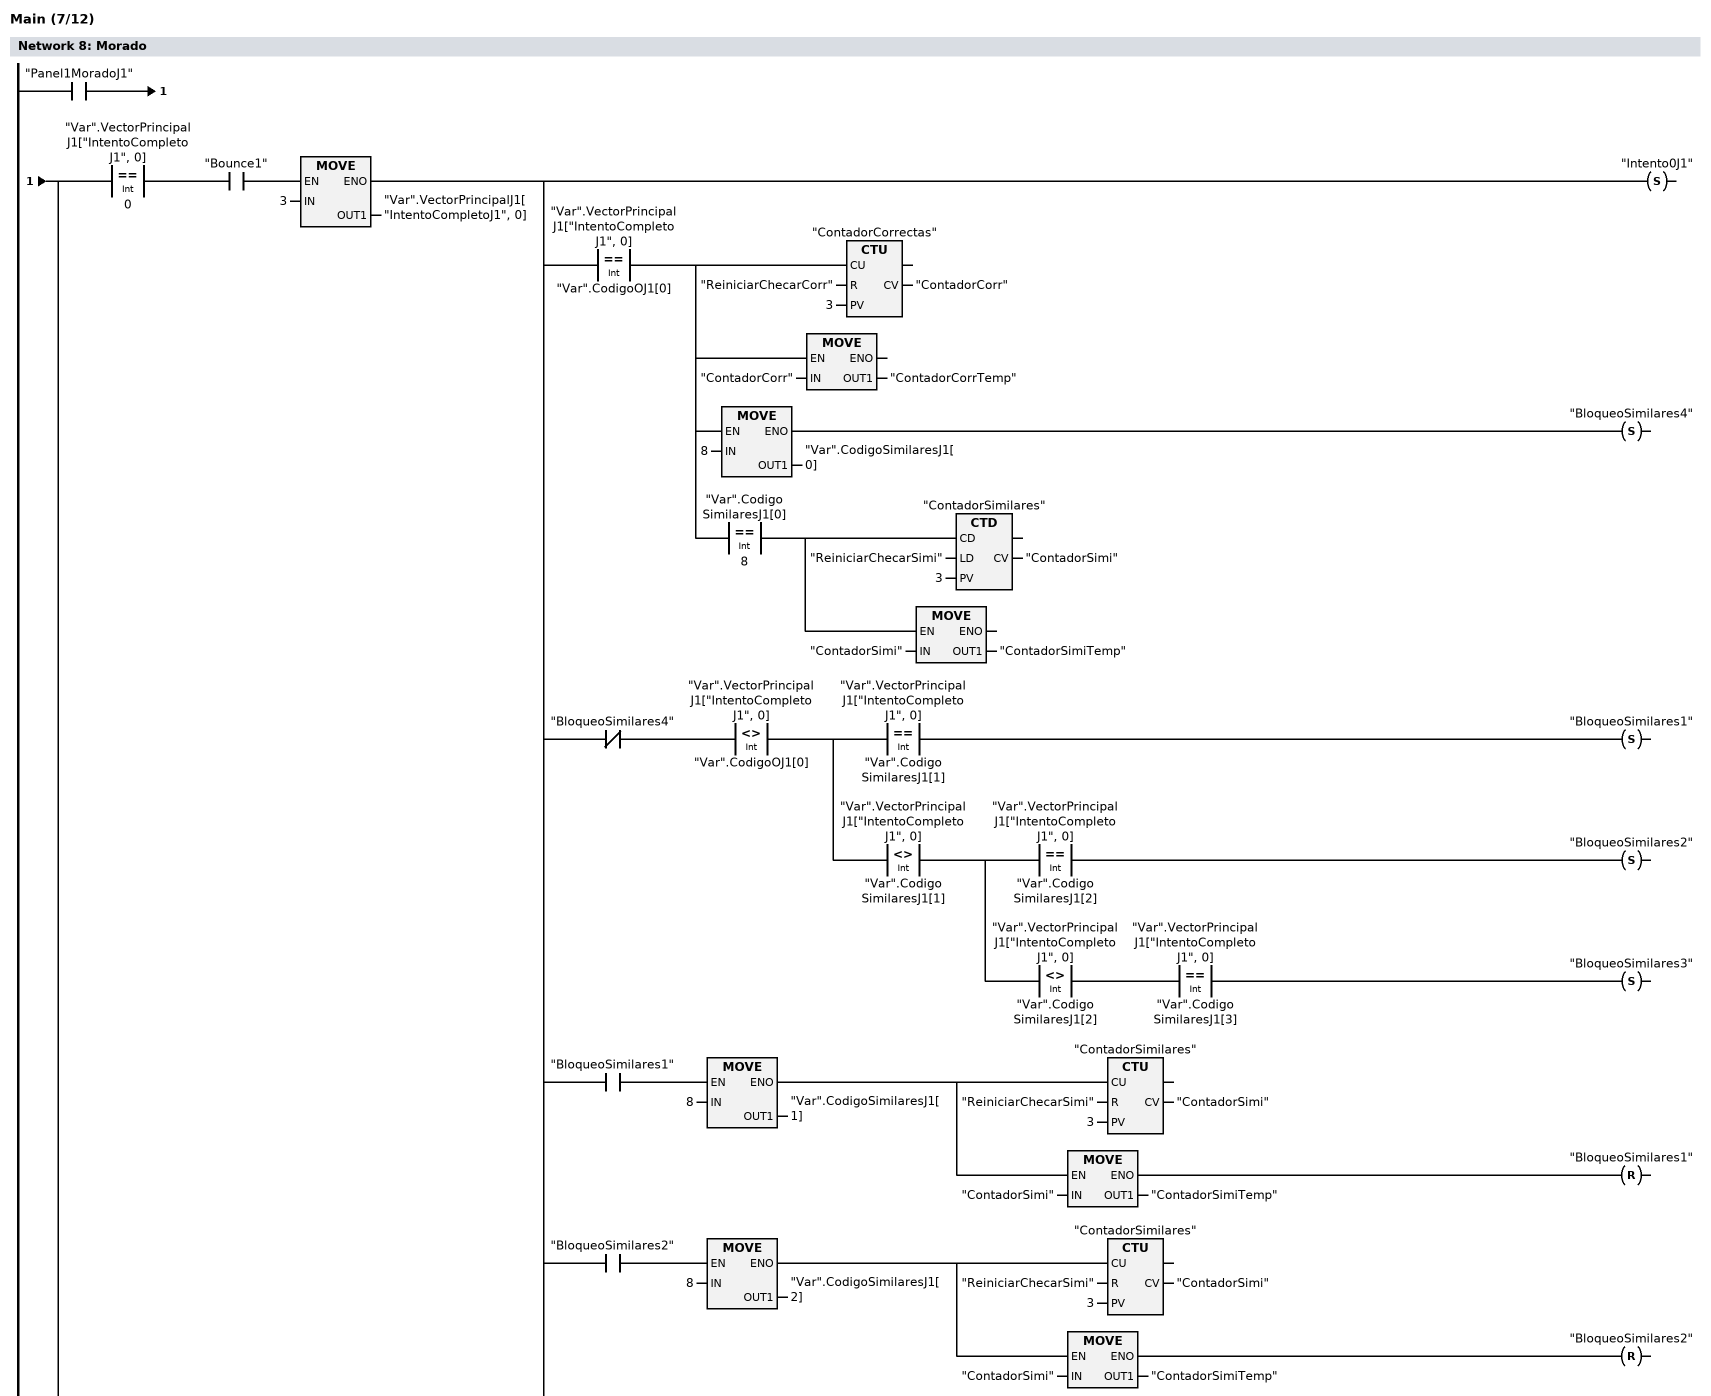
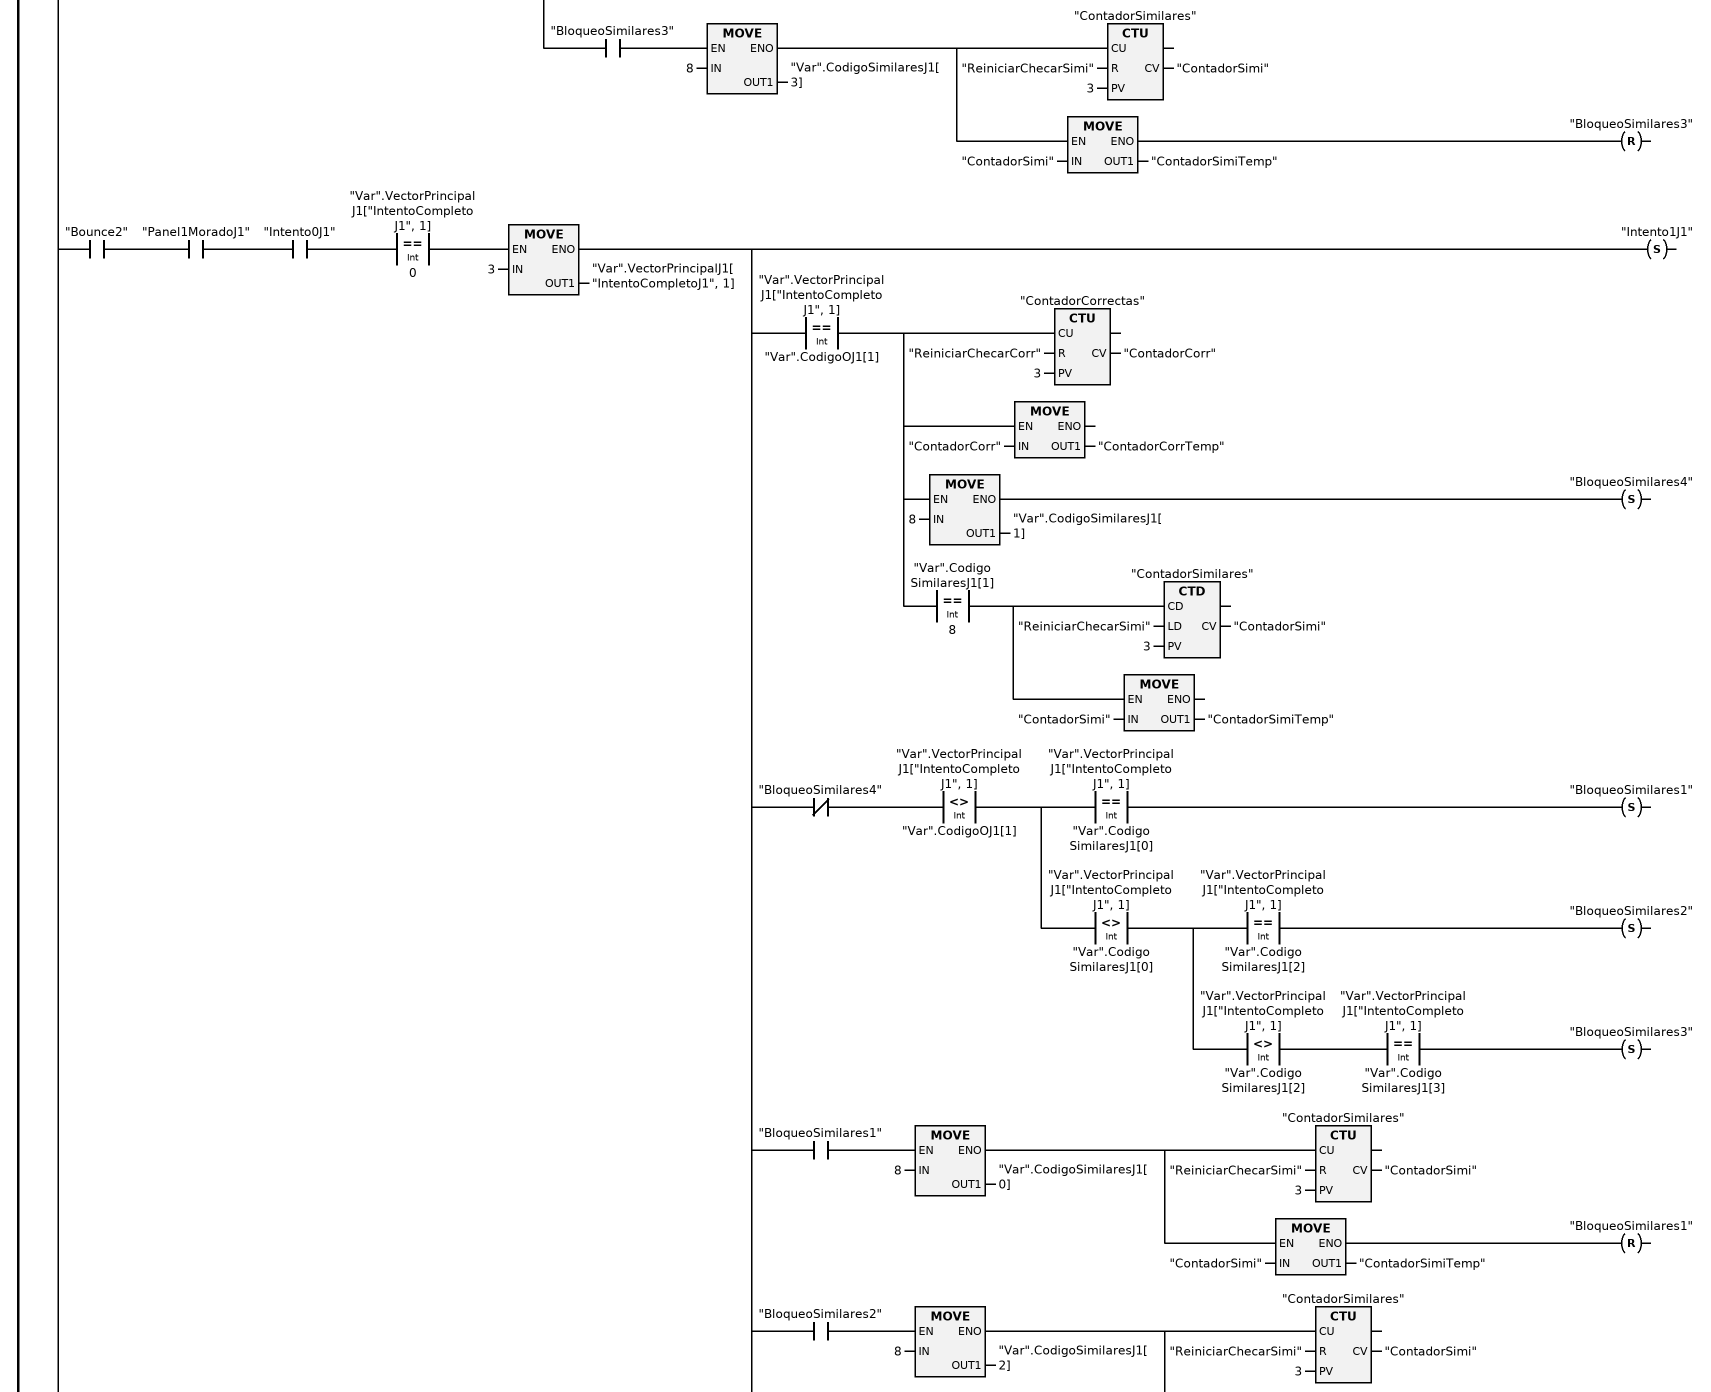
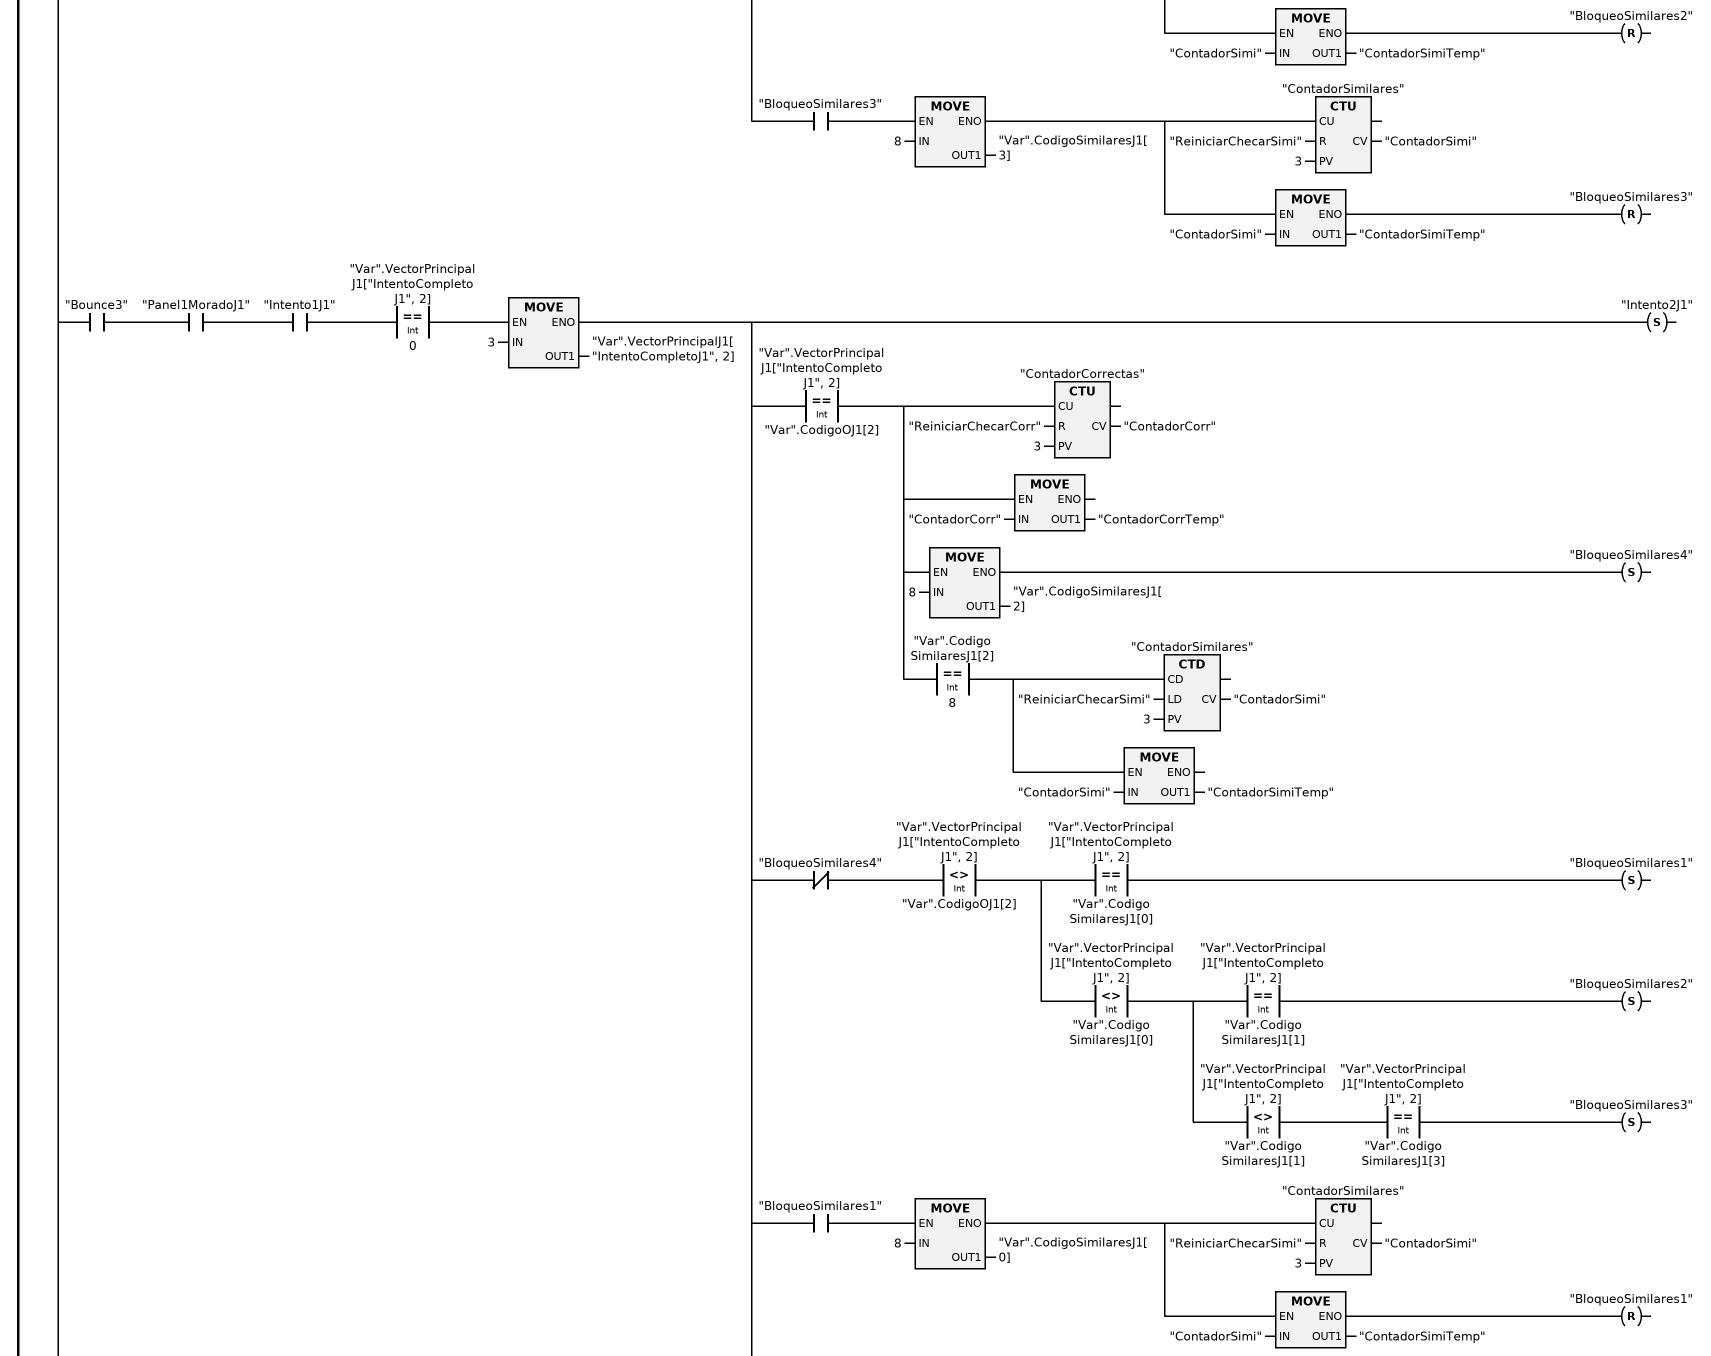
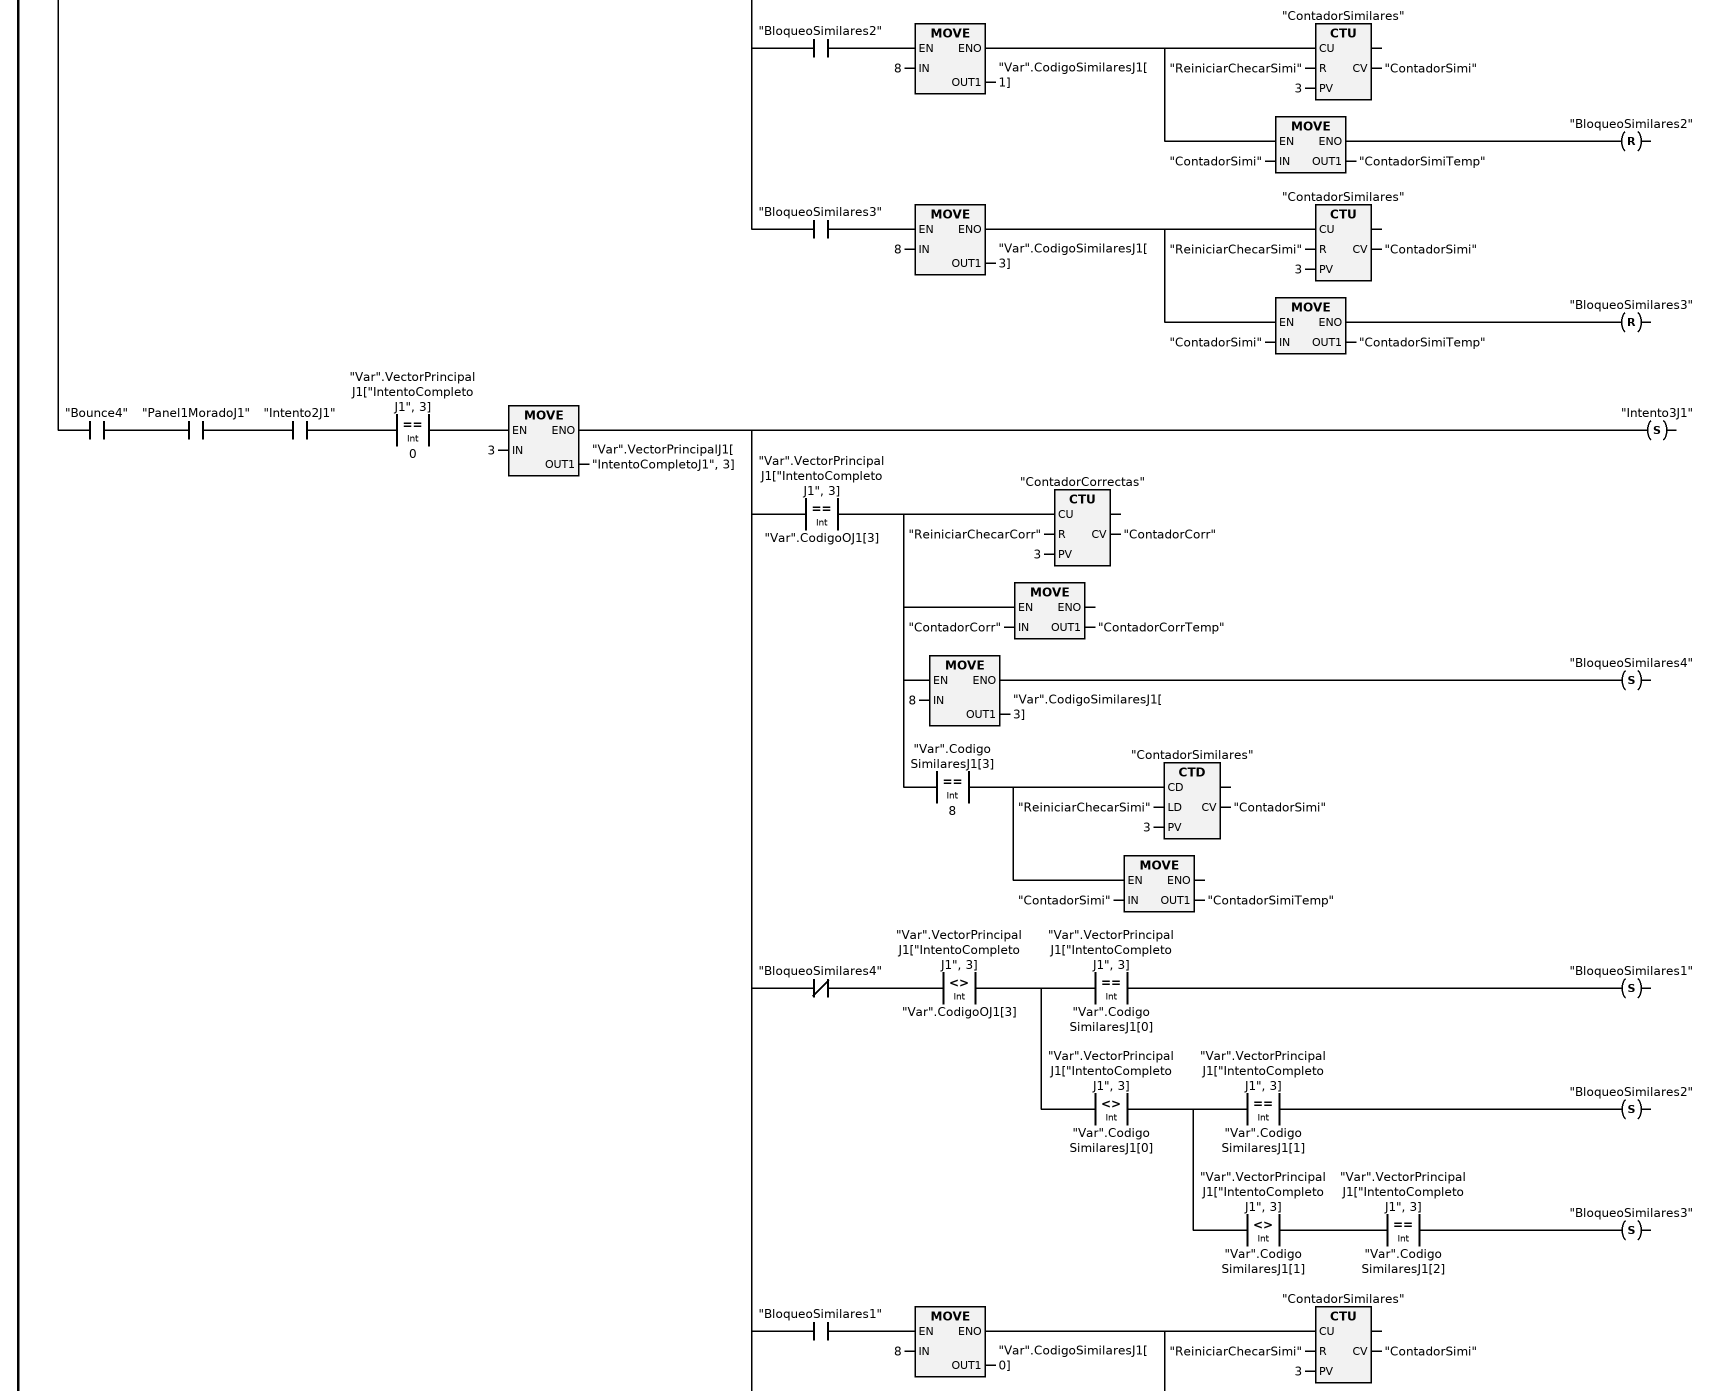
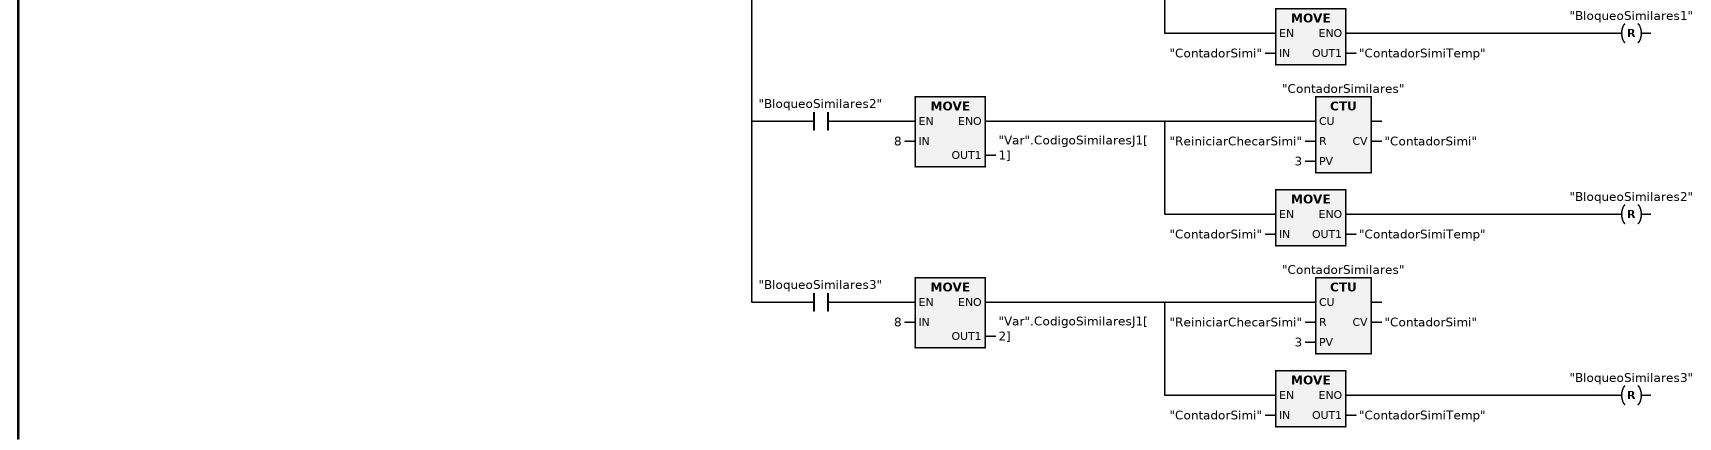
   #_w1 := "Panel1MoradoJ1" AND ("Var".VectorPrincipalJ1["IntentoCompletoJ1", 0] = 0) AND "Bounce1";
   IF #_w1 THEN
       "Var".VectorPrincipalJ1["IntentoCompletoJ1", 0] := 3;
       "Intento0J1" := TRUE;
   END_IF;
   #_w2 := #_w1 AND ("Var".VectorPrincipalJ1["IntentoCompletoJ1", 0] = "Var".CodigoOJ1[0]);
   "ContadorCorrectas".CTU(CU := #_w2, R := "ReiniciarChecarCorr", PV := 3, CV => "ContadorCorr");
   IF #_w2 THEN
       "ContadorCorrTemp" := "ContadorCorr";
       "Var".CodigoSimilaresJ1[0] := 8;
       "BloqueoSimilares4" := TRUE;
   END_IF;
   #_w3 := #_w2 AND ("Var".CodigoSimilaresJ1[0] = 8);
   "ContadorSimilares".CTD(CD := #_w3, LD := "ReiniciarChecarSimi", PV := 3, CV => "ContadorSimi");
   IF #_w3 THEN "ContadorSimiTemp" := "ContadorSimi"; END_IF;
   #_w4 := #_w1 AND NOT "BloqueoSimilares4" AND ("Var".VectorPrincipalJ1["IntentoCompletoJ1", 0] <> "Var".CodigoOJ1[0]);
   IF #_w4 AND ("Var".VectorPrincipalJ1["IntentoCompletoJ1", 0] = "Var".CodigoSimilaresJ1[1]) THEN
       "BloqueoSimilares1" := TRUE;
   END_IF;
   #_w5 := #_w4 AND ("Var".VectorPrincipalJ1["IntentoCompletoJ1", 0] <> "Var".CodigoSimilaresJ1[1]);
   IF #_w5 AND ("Var".VectorPrincipalJ1["IntentoCompletoJ1", 0] = "Var".CodigoSimilaresJ1[2]) THEN
       "BloqueoSimilares2" := TRUE;
   END_IF;
   IF #_w5 AND ("Var".VectorPrincipalJ1["IntentoCompletoJ1", 0] <> "Var".CodigoSimilaresJ1[2]) AND ("Var".VectorPrincipalJ1["IntentoCompletoJ1", 0] = "Var".CodigoSimilaresJ1[3]) THEN
       "BloqueoSimilares3" := TRUE;
   END_IF;
   #_w6 := #_w1 AND "BloqueoSimilares1";
   IF #_w6 THEN "Var".CodigoSimilaresJ1[1] := 8; END_IF;
   "ContadorSimilares".CTU(CU := #_w6, R := "ReiniciarChecarSimi", PV := 3, CV => "ContadorSimi");
   IF #_w6 THEN
       "ContadorSimiTemp" := "ContadorSimi";
       "BloqueoSimilares1" := FALSE;
   END_IF;
   #_w7 := #_w1 AND "BloqueoSimilares2";
   IF #_w7 THEN "Var".CodigoSimilaresJ1[2] := 8; END_IF;
   "ContadorSimilares".CTU(CU := #_w7, R := "ReiniciarChecarSimi", PV := 3, CV => "ContadorSimi");
   IF #_w7 THEN
       "ContadorSimiTemp" := "ContadorSimi";
       "BloqueoSimilares2" := FALSE;
   END_IF;
   #_w8 := #_w1 AND "BloqueoSimilares3";
   IF #_w8 THEN "Var".CodigoSimilaresJ1[3] := 8; END_IF;
   "ContadorSimilares".CTU(CU := #_w8, R := "ReiniciarChecarSimi", PV := 3, CV => "ContadorSimi");
   IF #_w8 THEN
       "ContadorSimiTemp" := "ContadorSimi";
       "BloqueoSimilares3" := FALSE;
   END_IF;
   #_w9 := "Panel1MoradoJ1" AND "Bounce2" AND "Panel1MoradoJ1" AND "Intento0J1" AND ("Var".VectorPrincipalJ1["IntentoCompletoJ1", 1] = 0);
   IF #_w9 THEN
       "Var".VectorPrincipalJ1["IntentoCompletoJ1", 1] := 3;
       "Intento1J1" := TRUE;
   END_IF;
   #_w10 := #_w9 AND ("Var".VectorPrincipalJ1["IntentoCompletoJ1", 1] = "Var".CodigoOJ1[1]);
   "ContadorCorrectas".CTU(CU := #_w10, R := "ReiniciarChecarCorr", PV := 3, CV => "ContadorCorr");
   IF #_w10 THEN
       "ContadorCorrTemp" := "ContadorCorr";
       "Var".CodigoSimilaresJ1[1] := 8;
       "BloqueoSimilares4" := TRUE;
   END_IF;
   #_w11 := #_w10 AND ("Var".CodigoSimilaresJ1[1] = 8);
   "ContadorSimilares".CTD(CD := #_w11, LD := "ReiniciarChecarSimi", PV := 3, CV => "ContadorSimi");
   IF #_w11 THEN "ContadorSimiTemp" := "ContadorSimi"; END_IF;
   #_w12 := #_w9 AND NOT "BloqueoSimilares4" AND ("Var".VectorPrincipalJ1["IntentoCompletoJ1", 1] <> "Var".CodigoOJ1[1]);
   IF #_w12 AND ("Var".VectorPrincipalJ1["IntentoCompletoJ1", 1] = "Var".CodigoSimilaresJ1[0]) THEN
       "BloqueoSimilares1" := TRUE;
   END_IF;
   #_w13 := #_w12 AND ("Var".VectorPrincipalJ1["IntentoCompletoJ1", 1] <> "Var".CodigoSimilaresJ1[0]);
   IF #_w13 AND ("Var".VectorPrincipalJ1["IntentoCompletoJ1", 1] = "Var".CodigoSimilaresJ1[2]) THEN
       "BloqueoSimilares2" := TRUE;
   END_IF;
   IF #_w13 AND ("Var".VectorPrincipalJ1["IntentoCompletoJ1", 1] <> "Var".CodigoSimilaresJ1[2]) AND ("Var".VectorPrincipalJ1["IntentoCompletoJ1", 1] = "Var".CodigoSimilaresJ1[3]) THEN
       "BloqueoSimilares3" := TRUE;
   END_IF;
   #_w14 := #_w9 AND "BloqueoSimilares1";
   IF #_w14 THEN "Var".CodigoSimilaresJ1[0] := 8; END_IF;
   "ContadorSimilares".CTU(CU := #_w14, R := "ReiniciarChecarSimi", PV := 3, CV => "ContadorSimi");
   IF #_w14 THEN
       "ContadorSimiTemp" := "ContadorSimi";
       "BloqueoSimilares1" := FALSE;
   END_IF;
   #_w15 := #_w9 AND "BloqueoSimilares2";
   IF #_w15 THEN "Var".CodigoSimilaresJ1[2] := 8; END_IF;
   "ContadorSimilares".CTU(CU := #_w15, R := "ReiniciarChecarSimi", PV := 3, CV => "ContadorSimi");
   IF #_w15 THEN
       "ContadorSimiTemp" := "ContadorSimi";
       "BloqueoSimilares2" := FALSE;
   END_IF;
   #_w16 := #_w9 AND "BloqueoSimilares3";
   IF #_w16 THEN "Var".CodigoSimilaresJ1[3] := 8; END_IF;
   "ContadorSimilares".CTU(CU := #_w16, R := "ReiniciarChecarSimi", PV := 3, CV => "ContadorSimi");
   IF #_w16 THEN
       "ContadorSimiTemp" := "ContadorSimi";
       "BloqueoSimilares3" := FALSE;
   END_IF;
   #_w17 := "Panel1MoradoJ1" AND "Bounce3" AND "Panel1MoradoJ1" AND "Intento1J1" AND ("Var".VectorPrincipalJ1["IntentoCompletoJ1", 2] = 0);
   IF #_w17 THEN
       "Var".VectorPrincipalJ1["IntentoCompletoJ1", 2] := 3;
       "Intento2J1" := TRUE;
   END_IF;
   #_w18 := #_w17 AND ("Var".VectorPrincipalJ1["IntentoCompletoJ1", 2] = "Var".CodigoOJ1[2]);
   "ContadorCorrectas".CTU(CU := #_w18, R := "ReiniciarChecarCorr", PV := 3, CV => "ContadorCorr");
   IF #_w18 THEN
       "ContadorCorrTemp" := "ContadorCorr";
       "Var".CodigoSimilaresJ1[2] := 8;
       "BloqueoSimilares4" := TRUE;
   END_IF;
   #_w19 := #_w18 AND ("Var".CodigoSimilaresJ1[2] = 8);
   "ContadorSimilares".CTD(CD := #_w19, LD := "ReiniciarChecarSimi", PV := 3, CV => "ContadorSimi");
   IF #_w19 THEN "ContadorSimiTemp" := "ContadorSimi"; END_IF;
   #_w20 := #_w17 AND NOT "BloqueoSimilares4" AND ("Var".VectorPrincipalJ1["IntentoCompletoJ1", 2] <> "Var".CodigoOJ1[2]);
   IF #_w20 AND ("Var".VectorPrincipalJ1["IntentoCompletoJ1", 2] = "Var".CodigoSimilaresJ1[0]) THEN
       "BloqueoSimilares1" := TRUE;
   END_IF;
   #_w21 := #_w20 AND ("Var".VectorPrincipalJ1["IntentoCompletoJ1", 2] <> "Var".CodigoSimilaresJ1[0]);
   IF #_w21 AND ("Var".VectorPrincipalJ1["IntentoCompletoJ1", 2] = "Var".CodigoSimilaresJ1[1]) THEN
       "BloqueoSimilares2" := TRUE;
   END_IF;
   IF #_w21 AND ("Var".VectorPrincipalJ1["IntentoCompletoJ1", 2] <> "Var".CodigoSimilaresJ1[1]) AND ("Var".VectorPrincipalJ1["IntentoCompletoJ1", 2] = "Var".CodigoSimilaresJ1[3]) THEN
       "BloqueoSimilares3" := TRUE;
   END_IF;
   #_w22 := #_w17 AND "BloqueoSimilares1";
   IF #_w22 THEN "Var".CodigoSimilaresJ1[0] := 8; END_IF;
   "ContadorSimilares".CTU(CU := #_w22, R := "ReiniciarChecarSimi", PV := 3, CV => "ContadorSimi");
   IF #_w22 THEN
       "ContadorSimiTemp" := "ContadorSimi";
       "BloqueoSimilares1" := FALSE;
   END_IF;
   #_w23 := #_w17 AND "BloqueoSimilares2";
   IF #_w23 THEN "Var".CodigoSimilaresJ1[1] := 8; END_IF;
   "ContadorSimilares".CTU(CU := #_w23, R := "ReiniciarChecarSimi", PV := 3, CV => "ContadorSimi");
   IF #_w23 THEN
       "ContadorSimiTemp" := "ContadorSimi";
       "BloqueoSimilares2" := FALSE;
   END_IF;
   #_w24 := #_w17 AND "BloqueoSimilares3";
   IF #_w24 THEN "Var".CodigoSimilaresJ1[3] := 8; END_IF;
   "ContadorSimilares".CTU(CU := #_w24, R := "ReiniciarChecarSimi", PV := 3, CV => "ContadorSimi");
   IF #_w24 THEN
       "ContadorSimiTemp" := "ContadorSimi";
       "BloqueoSimilares3" := FALSE;
   END_IF;
   #_w25 := "Panel1MoradoJ1" AND "Bounce4" AND "Panel1MoradoJ1" AND "Intento2J1" AND ("Var".VectorPrincipalJ1["IntentoCompletoJ1", 3] = 0);
   IF #_w25 THEN
       "Var".VectorPrincipalJ1["IntentoCompletoJ1", 3] := 3;
       "Intento3J1" := TRUE;
   END_IF;
   #_w26 := #_w25 AND ("Var".VectorPrincipalJ1["IntentoCompletoJ1", 3] = "Var".CodigoOJ1[3]);
   "ContadorCorrectas".CTU(CU := #_w26, R := "ReiniciarChecarCorr", PV := 3, CV => "ContadorCorr");
   IF #_w26 THEN
       "ContadorCorrTemp" := "ContadorCorr";
       "Var".CodigoSimilaresJ1[3] := 8;
       "BloqueoSimilares4" := TRUE;
   END_IF;
   #_w27 := #_w26 AND ("Var".CodigoSimilaresJ1[3] = 8);
   "ContadorSimilares".CTD(CD := #_w27, LD := "ReiniciarChecarSimi", PV := 3, CV => "ContadorSimi");
   IF #_w27 THEN "ContadorSimiTemp" := "ContadorSimi"; END_IF;
   #_w28 := #_w25 AND NOT "BloqueoSimilares4" AND ("Var".VectorPrincipalJ1["IntentoCompletoJ1", 3] <> "Var".CodigoOJ1[3]);
   IF #_w28 AND ("Var".VectorPrincipalJ1["IntentoCompletoJ1", 3] = "Var".CodigoSimilaresJ1[0]) THEN
       "BloqueoSimilares1" := TRUE;
   END_IF;
   #_w29 := #_w28 AND ("Var".VectorPrincipalJ1["IntentoCompletoJ1", 3] <> "Var".CodigoSimilaresJ1[0]);
   IF #_w29 AND ("Var".VectorPrincipalJ1["IntentoCompletoJ1", 3] = "Var".CodigoSimilaresJ1[1]) THEN
       "BloqueoSimilares2" := TRUE;
   END_IF;
   IF #_w29 AND ("Var".VectorPrincipalJ1["IntentoCompletoJ1", 3] <> "Var".CodigoSimilaresJ1[1]) AND ("Var".VectorPrincipalJ1["IntentoCompletoJ1", 3] = "Var".CodigoSimilaresJ1[2]) THEN
       "BloqueoSimilares3" := TRUE;
   END_IF;
   #_w30 := #_w25 AND "BloqueoSimilares1";
   IF #_w30 THEN "Var".CodigoSimilaresJ1[0] := 8; END_IF;
   "ContadorSimilares".CTU(CU := #_w30, R := "ReiniciarChecarSimi", PV := 3, CV => "ContadorSimi");
   IF #_w30 THEN
       "ContadorSimiTemp" := "ContadorSimi";
       "BloqueoSimilares1" := FALSE;
   END_IF;
   #_w31 := #_w25 AND "BloqueoSimilares2";
   IF #_w31 THEN "Var".CodigoSimilaresJ1[1] := 8; END_IF;
   "ContadorSimilares".CTU(CU := #_w31, R := "ReiniciarChecarSimi", PV := 3, CV => "ContadorSimi");
   IF #_w31 THEN
       "ContadorSimiTemp" := "ContadorSimi";
       "BloqueoSimilares2" := FALSE;
   END_IF;
   #_w32 := #_w25 AND "BloqueoSimilares3";
   IF #_w32 THEN "Var".CodigoSimilaresJ1[2] := 8; END_IF;
   "ContadorSimilares".CTU(CU := #_w32, R := "ReiniciarChecarSimi", PV := 3, CV => "ContadorSimi");
   IF #_w32 THEN
       "ContadorSimiTemp" := "ContadorSimi";
       "BloqueoSimilares3" := FALSE;
   END_IF;
END_REGION

REGION Network 9: Rojo
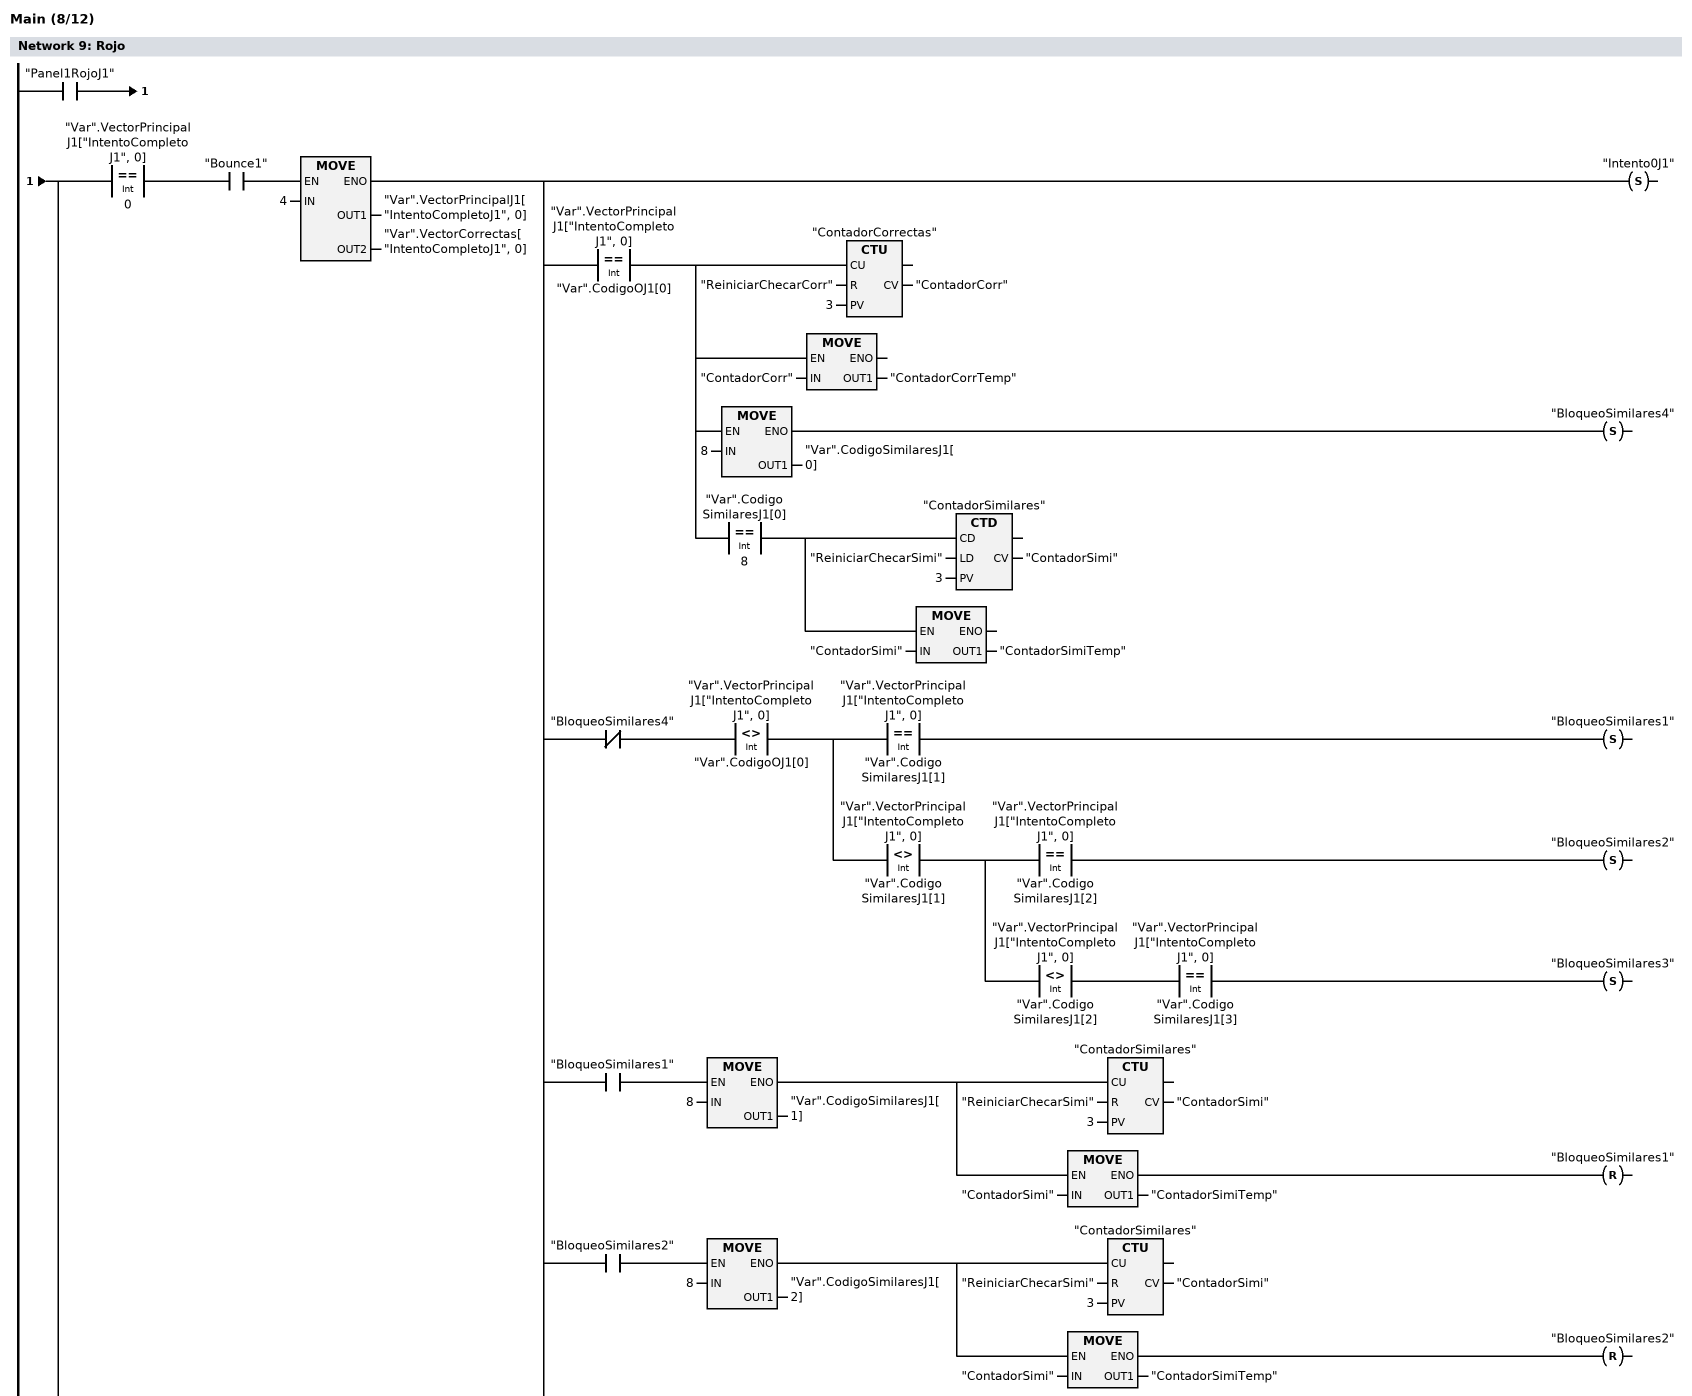
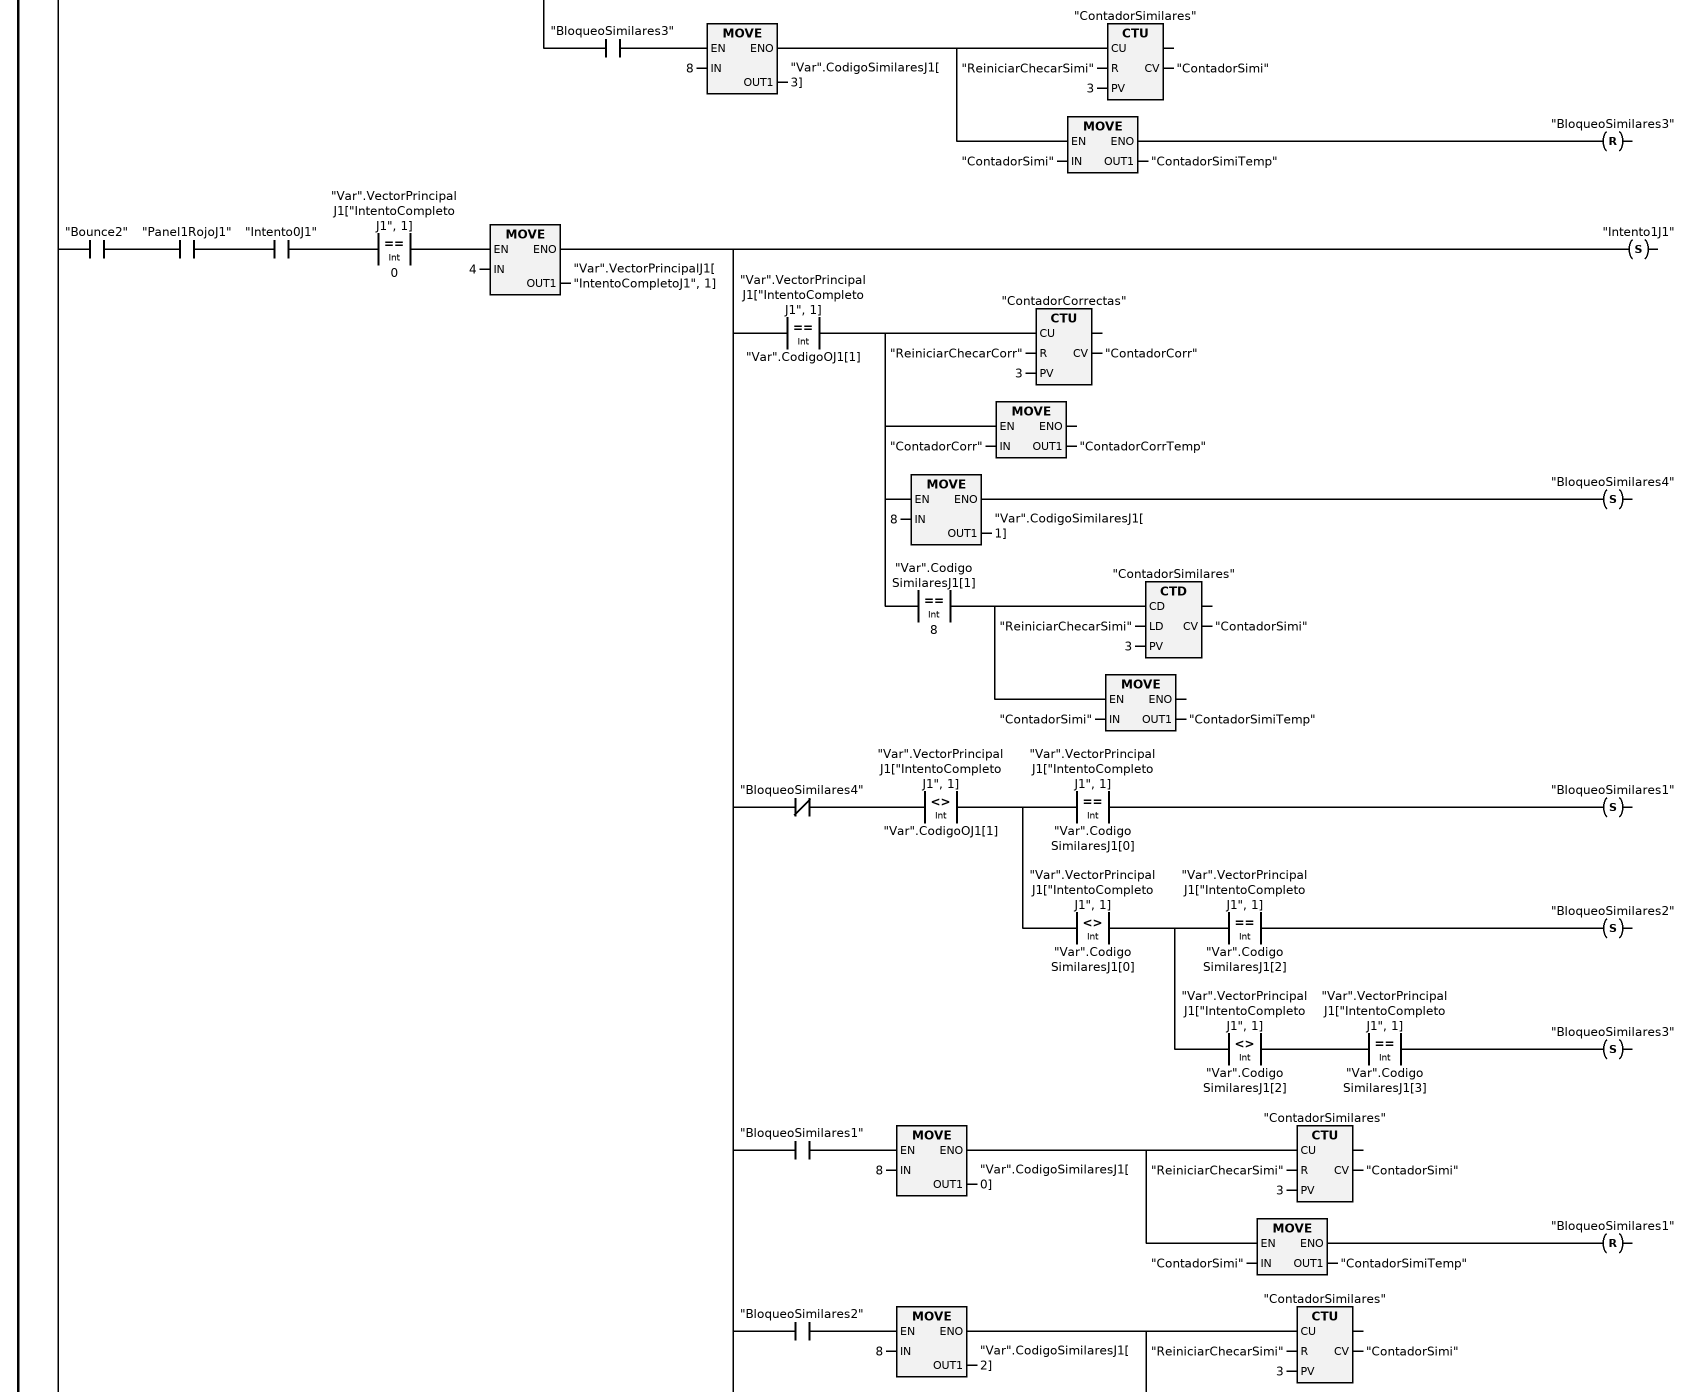
